// TIA Portal project "MSIL_TESTER_REV3_12JAN23" (V15)

(* hardware
DEVICE "S7-1200 station_1"  S7-1200 Station
   slot 0: "Rack_0"  S7-1200 Rack  Rack  V1.0
   slot 1: "PLC_1"  CPU 1214C DC/DC/DC  6ES7 214-1AG40-0XB0  V4.2
   slot 2: "DI 16/DQ 16x24VDC_1"  6ES7 223-1BL32-0XB0  V2.0
   slot 3: "DQ 8x24VDC _1"  SM 1222 DQ8 x 24VDC  6ES7 222-1BF32-0XB0  V2.0
DEVICE "GSD device_1"  GSD.Device.PN
   slot 0: "Rack"  Rack  V1.0
   slot 0: "cv-x400"  CV-X4XX  CV-X4XX  5.1
      slot 0: "CV-X4XX"  CV-X4XX  5.1
      slot 1: "Interface"  Interface
         slot 1: "Port 1"  Port 1
   slot 1: "Command and Result Status_1"  Command and Result Status
      slot 0: "Command and Result Status"  Command and Result Status
   slot 2: "Trg Ready Status_1"  Trg Ready Status
      slot 0: "Trg Ready Status"  Trg Ready Status
   slot 3: "Trg Ack Status_1"  Trg Ack Status
      slot 0: "Trg Ack Status"  Trg Ack Status
   slot 4: "Miscellaneous Status_1"  Miscellaneous Status
      slot 0: "Miscellaneous Status"  Miscellaneous Status
   slot 5: "Tool Judge Value_1"  Tool Judge Value
      slot 0: "Tool Judge Value"  Tool Judge Value
   slot 6: "Result Data 128Byte_1"  Result Data 128Byte
      slot 0: "Result Data 128Byte"  Result Data 128Byte
   slot 7: "Result Data 32Byte_1"  Result Data 32Byte
      slot 0: "Result Data 32Byte"  Result Data 32Byte
   slot 8: "Result Data 32Byte_2"  Result Data 32Byte
      slot 0: "Result Data 32Byte"  Result Data 32Byte
   slot 9: "Result Data 32Byte_3"  Result Data 32Byte
      slot 0: "Result Data 32Byte"  Result Data 32Byte
   slot 10: "Result Data 32Byte_4"  Result Data 32Byte
      slot 0: "Result Data 32Byte"  Result Data 32Byte
   slot 11: "Result Data 32Byte_5"  Result Data 32Byte
      slot 0: "Result Data 32Byte"  Result Data 32Byte
   slot 12: "Command and Result Control_1"  Command and Result Control
      slot 0: "Command and Result Control"  Command and Result Control
   slot 13: "Trg Control_1"  Trg Control
      slot 0: "Trg Control"  Trg Control
   slot 14: "Miscellaneous Control_1"  Miscellaneous Control
      slot 0: "Miscellaneous Control"  Miscellaneous Control
   slot 15: "Reserved Control_1"  Reserved Control
      slot 0: "Reserved Control"  Reserved Control
   slot 16: "Reserved Control_2"  Reserved Control
      slot 0: "Reserved Control"  Reserved Control
   slot 17: "Parameter 128Byte_1"  Parameter 128Byte
      slot 0: "Parameter 128Byte"  Parameter 128Byte
   slot 18: "Parameter 32Byte_1"  Parameter 32Byte
      slot 0: "Parameter 32Byte"  Parameter 32Byte
   slot 19: "Parameter 32Byte_2"  Parameter 32Byte
      slot 0: "Parameter 32Byte"  Parameter 32Byte
   slot 20: "Parameter 32Byte_3"  Parameter 32Byte
      slot 0: "Parameter 32Byte"  Parameter 32Byte
   slot 21: "Parameter 32Byte_4"  Parameter 32Byte
      slot 0: "Parameter 32Byte"  Parameter 32Byte
   slot 22: "Parameter 32Byte_5"  Parameter 32Byte
      slot 0: "Parameter 32Byte"  Parameter 32Byte
*)

// ===== PLC "PLC_1"  CPU 1214C DC/DC/DC =====

VAR_GLOBAL   // PLC tag table "Default tag table"
   "EMG" AT %I0.0 : Bool;
   "RESET" AT %I0.1 : Bool;
   "Tag_9" AT %I0.2 : Bool;
   "Tag_10" AT %I0.3 : Bool;
   "Tag_11" AT %I0.4 : Bool;
   "Tag_12" AT %I0.5 : Bool;
   "Tag_13" AT %I0.6 : Bool;
   "Tag_14" AT %I0.7 : Bool;
   "Tag_15" AT %I1.0 : Bool;
   "Tag_16" AT %I1.1 : Bool;
   "Tag_17" AT %I1.2 : Bool;
   "Tag_18" AT %I1.3 : Bool;
   "Tag_19" AT %I1.4 : Bool;
   "Tag_20" AT %I1.5 : Bool;
   "Tag_21" AT %I1.6 : Bool;
   "Tag_22" AT %I2.0 : Bool;
   "Tag_23" AT %I2.1 : Bool;
   "Tag_24" AT %I2.2 : Bool;
   "Tag_25" AT %I2.3 : Bool;
   "Tag_26" AT %I2.4 : Bool;
   "Tag_27" AT %I2.5 : Bool;
   "Tag_28" AT %I2.6 : Bool;
   "Tag_29" AT %I2.7 : Bool;
   "Tag_30" AT %I3.0 : Bool;
   "Tag_32" AT %I3.2 : Bool;
   "Tag_46" AT %I3.3 : Bool;
   "Tag_47" AT %I3.4 : Bool;
   "TEST_PART" AT %I1.7 : Bool;
   "Tag_53" AT %I3.5 : Bool;
   "Tag_60" AT %IB12 : Byte;
   "Tag_62" AT %I10.0 : Bool;
   "Tag_59" AT %I10.2 : Bool;
   "Tag_66" AT %IB76 : Byte;
   "Tag_69" AT %IW76 : Int;
   "Tag_75" AT %I10.5 : Bool;
   "rdy" AT %I5.5 : Bool;
   "Tag_76" AT %I3.1 : Bool;
   "Tag_77" AT %I3.6 : Bool;
   "Tag_78" AT %I3.7 : Bool;
   "Tag_3" AT %I13.0 : Bool;
   "Cmd Complete" AT %I20.0 : Bool;
   "Cmd Err" AT %I20.1 : Bool;
   "Cmd Ready" AT %I20.2 : Bool;
   "Result Ready" AT %I20.3 : Bool;
   "Result OR" AT %I20.4 : Bool;
   "res1" AT %I20.5 : Bool;
   "res2" AT %I20.6 : Bool;
   "res3" AT %I20.7 : Bool;
   "READY1" AT %I6.0 : Bool;
   "READY2" AT %I6.1 : Bool;
   "READY3" AT %I6.2 : Bool;
   "READY4" AT %I6.3 : Bool;
   "res4" AT %I6.4 : Bool;
   "res5" AT %I6.5 : Bool;
   "res6" AT %I6.6 : Bool;
   "res7" AT %I6.7 : Bool;
   "BUSY" AT %I7.0 : Bool;
   "ERROR" AT %I7.1 : Bool;
   "res8" AT %I7.2 : Bool;
   "RUN" AT %I7.3 : Bool;
   "res9" AT %I7.4 : Bool;
   "res10" AT %I7.5 : Bool;
   "OUTPUT_IMG_BUSY" AT %I7.6 : Bool;
   "OUTPUT_IMG_STATUS" AT %I7.7 : Bool;
   "res" AT %I8.0 : Bool;
   "res11" AT %I8.1 : Bool;
   "res12" AT %I8.2 : Bool;
   "res13" AT %I8.3 : Bool;
   "res14" AT %I8.4 : Bool;
   "res15" AT %I8.5 : Bool;
   "res16" AT %I8.6 : Bool;
   "res17" AT %I8.7 : Bool;
   "LOGO_RSLT_OK" AT %I68.0 : Bool;
   "LOGO_RSLT_NG" AT %I68.1 : Bool;
   "LED_RSLT_OK" AT %I68.2 : Bool;
   "LED_RSLT_NG" AT %I68.3 : Bool;
   "Tool Judge Value4" AT %I452.4 : Bool;
   "Tag_83" AT %I15.0 : Bool;
   "Tag_1" AT %Q2.5 : Bool;
   "Tag_2" AT %Q3.0 : Bool;
   "Tag_4" AT %Q2.0 : Bool;
   "Tag_5" AT %Q0.1 : Bool;
   "Tag_7" AT %Q0.2 : Bool;
   "Tag_8" AT %Q0.3 : Bool;
   "Tag_33" AT %Q0.5 : Bool;
   "Tag_34" AT %Q0.6 : Bool;
   "Tag_35" AT %Q0.7 : Bool;
   "Tag_36" AT %Q1.0 : Bool;
   "Tag_37" AT %Q1.1 : Bool;
   "Tag_38" AT %Q2.1 : Bool;
   "Tag_39" AT %Q2.2 : Bool;
   "Tag_40" AT %Q2.3 : Bool;
   "Tag_41" AT %Q3.1 : Bool;
   "Tag_42" AT %Q3.2 : Bool;
   "Tag_43" AT %Q3.3 : Bool;
   "Tag_44" AT %Q2.6 : Bool;
   "Tag_45" AT %Q2.7 : Bool;
   "Tag_48" AT %Q3.4 : Bool;
   "Tag_49" AT %Q3.5 : Bool;
   "Tag_50" AT %Q3.6 : Bool;
   "Tag_51" AT %Q3.7 : Bool;
   "Tag_52" AT %Q2.4 : Bool;
   "Tag_58" AT %QB12 : Byte;
   "Tag_56" AT %QB6 : Byte;
   "Tag_64" AT %QB8 : Byte;
   "Tag_65" AT %Q500.5 : Bool;
   "Tag_67" AT %QW504 : Int;
   "Tag_68" AT %QW76 : Int;
   "Tag_71" AT %Q500.0 : Bool;
   "Tag_72" AT %Q500.2 : Bool;
   "Tag_61" AT %Q4.0 : Bool;
   "Tag_63" AT %Q4.1 : Bool;
   "Tag_73" AT %Q4.2 : Bool;
   "Tag_74" AT %Q4.3 : Bool;
   "Tag_79" AT %Q4.4 : Bool;
   "Tag_80" AT %Q4.5 : Bool;
   "Tag_81" AT %Q0.0 : Bool;
   "Tag_6" AT %Q0.4 : Bool;
   "Tag_82" AT %Q6.0 : Bool;
   "Tag_86" AT %Q601.0 : Bool;
   "Tag_87" AT %Q50.0 : Bool;
   "Tag_88" AT %Q51.0 : Bool;
   "Tag_89" AT %Q52.0 : Bool;
   "Tag_90" AT %Q31.0 : Bool;
   "Tag_91" AT %Q5.0 : Bool;
   "Tag_31" AT %Q6.1 : Bool;
   "cam_reset" AT %Q7.0 : Bool;
   "Cam_Ext" AT %Q7.1 : Bool;
   "Tag_54" AT %QW2 : Int;
   "Tag_55" AT %QW21 : Int;
   "Tag_57" AT %QW24 : Word;
   "Tag_70" AT %QW29 : Word;
   "command" AT %QW78 : Int;
   "SD_CardNo" AT %QD80 : DInt;
   "Program_Number" AT %QD84 : DInt;
   "TAG 1" AT %M1.0 : Bool;
   "SHORT_CT" AT %M1.1 : Bool;
   "OK" AT %M1.2 : Bool;
   "NG" AT %M1.3 : Bool;
   "CONTINUITY" AT %M1.4 : Bool;
   "DIELECTRIC" AT %M1.5 : Bool;
   "TAG 2" AT %M1.6 : Bool;
   "SEQ_1" AT %MB2 : Byte;
   "RED_LED" AT %M1.7 : Bool;
   "AMBER_LED" AT %M3.0 : Bool;
   "GREEN_LED" AT %M3.1 : Bool;
   "TAG 3" AT %M3.2 : Bool;
   "TAG 4" AT %M3.3 : Bool;
   "TEST" AT %M3.4 : Bool;
   "MAIN SEQ" AT %MW4 : Int;
   "BLUE LED" AT %M3.5 : Bool;
   "GROUND" AT %M3.6 : Bool;
   "RED LED" AT %M3.7 : Bool;
   "GREEN LED" AT %M6.0 : Bool;
   "SEQ_MAIN" AT %MW8 : Int;
   "RED" AT %M6.1 : Bool;
   "BLUE" AT %M6.2 : Bool;
   "GREEN" AT %M6.3 : Bool;
   "COMMON" AT %M6.4 : Bool;
   "TEST 3" AT %M6.5 : Bool;
   "TEST 4" AT %M6.6 : Bool;
   "TEST 5" AT %M6.7 : Bool;
   "TRG" AT %M7.0 : Bool;
   "INC" AT %MD10 : DInt;
   "P_TRG" AT %M7.1 : Bool;
   "INC`1" AT %MD14 : DInt;
   "TEST_START" AT %M7.2 : Bool;
   "TEST_6" AT %M7.3 : Bool;
   "CON_TRG" AT %M7.4 : Bool;
   "DIE_TRG" AT %M7.5 : Bool;
   "SHORT_TRG" AT %M7.6 : Bool;
   "BIT 1" AT %M7.7 : Bool;
   "BIT 2" AT %M18.0 : Bool;
   "TRG1" AT %M18.1 : Bool;
   "TRG 2" AT %M18.2 : Bool;
   "TRG 3" AT %M18.3 : Bool;
   "TRG 4" AT %M18.4 : Bool;
   "TRG5" AT %M18.5 : Bool;
   "TRG 6" AT %M18.6 : Bool;
   "TEST_SEQ" AT %MW20 : Int;
   "TEST 7" AT %M18.7 : Bool;
   "VISION_OK" AT %M19.0 : Bool;
   "VISION_NG" AT %M19.1 : Bool;
   "TRG 7" AT %M19.2 : Bool;
   "TRG 8" AT %M19.3 : Bool;
   "FGH" AT %MD22 : DInt;
   "TEST_RESET" AT %M19.4 : Bool;
   "test 10" AT %M19.5 : Bool;
   "TRG 9" AT %M19.6 : Bool;
   "test_print" AT %M19.7 : Bool;
   "FWD_TEST" AT %M26.0 : Bool;
   "X2" AT %M26.1 : Bool;
   "X3" AT %M26.2 : Bool;
   "CL" AT %M26.3 : Bool;
   "TEST_BUZ" AT %M26.4 : Bool;
   "System_Byte" AT %MB200 : Byte;
   "FirstScan" AT %M200.0 : Bool;
   "DiagStatusUpdate" AT %M200.1 : Bool;
   "AlwaysTRUE" AT %M200.2 : Bool;
   "AlwaysFALSE" AT %M200.3 : Bool;
   "Clock_Byte" AT %MB202 : Byte;
   "Clock_10Hz" AT %M202.0 : Bool;
   "Clock_5Hz" AT %M202.1 : Bool;
   "Clock_2.5Hz" AT %M202.2 : Bool;
   "Clock_2Hz" AT %M202.3 : Bool;
   "Clock_1.25Hz" AT %M202.4 : Bool;
   "Clock_1Hz" AT %M202.5 : Bool;
   "Clock_0.625Hz" AT %M202.6 : Bool;
   "Clock_0.5Hz" AT %M202.7 : Bool;
   "System_Byte(3)" AT %MB200 : Byte;
   "OK_TEST" AT %M26.5 : Bool;
   "NG_TEST" AT %M26.6 : Bool;
   "SCN_OK" AT %M26.7 : Bool;
   "TRG10" AT %M27.0 : Bool;
   "GROUND_TEST" AT %M27.1 : Bool;
   "TEST_GREEN" AT %M27.2 : Bool;
   "TEST_BLUE" AT %M27.3 : Bool;
   "TEST_RED" AT %M27.4 : Bool;
   "Manual" AT %M27.5 : Bool;
   "TRG11" AT %M27.6 : Bool;
   "TRG12" AT %M27.7 : Bool;
   "PROGRAM_TRG" AT %M28.0 : Bool;
   "BREAK" AT %M28.1 : Bool;
   "CAM_TRG" AT %M28.2 : Bool;
   "TRG 11" AT %M28.3 : Bool;
   "TRG 12" AT %M28.4 : Bool;
   "BUFF_CLR" AT %M28.5 : Bool;
   "TRG13" AT %M28.6 : Bool;
   "TRG14" AT %M28.7 : Bool;
   "TRG 15" AT %M29.0 : Bool;
   "TRG 16" AT %M29.1 : Bool;
   "TEST_CLEAR" AT %M29.2 : Bool;
   "TRG15" AT %M29.3 : Bool;
   "TRG_16" AT %M29.4 : Bool;
   "TRG17" AT %M29.5 : Bool;
   "BREAK 2" AT %M29.6 : Bool;
   "BREAK 3" AT %M29.7 : Bool;
   "break 4" AT %M30.0 : Bool;
   "break 5" AT %M30.1 : Bool;
   "break 6" AT %M30.2 : Bool;
   "break 9" AT %M30.3 : Bool;
   "break 10" AT %M30.4 : Bool;
   "TRG20" AT %M30.5 : Bool;
   "TRG 17" AT %M30.6 : Bool;
   "TRG 20" AT %M30.7 : Bool;
   "break 11" AT %M31.0 : Bool;
   "REJECTION_ERROR_SET" AT %M31.1 : Bool;
   "BREAK 15" AT %M31.2 : Bool;
   "assembly bar code" AT %M31.3 : Bool;
   "POT_TEST" AT %M31.4 : Bool;
   "POT_TEST_GREEN" AT %M0.0 : Bool;
   "POT_TEST_BLUE" AT %M0.1 : Bool;
   "SCAN_BYP" AT %M0.2 : Bool;
   "test16" AT %M0.3 : Bool;
   "BUFF_CLR_10" AT %M0.4 : Bool;
   "trg18" AT %M0.5 : Bool;
   "trg19" AT %M0.6 : Bool;
   "buff_clr_11" AT %M0.7 : Bool;
   "CAM_2ND_TRG" AT %M31.5 : Bool;
   "TRG25" AT %M31.6 : Bool;
   "START" AT %M31.7 : Bool;
   "EL_GOOD" AT %MD32 : DInt;
   "EL_BAD" AT %MD36 : DInt;
   "VISION_CAL_OFF" AT %M40.0 : Bool;
   "LOGO_CAL_OFF" AT %M40.1 : Bool;
   "LED_CALI_OFF" AT %M40.2 : Bool;
   "ELEC_CAL_OFF" AT %M40.3 : Bool;
   "TEST 17" AT %M40.4 : Bool;
   "TEST 18" AT %M40.5 : Bool;
   "TEST 19" AT %M40.6 : Bool;
   "TEST 20" AT %M40.7 : Bool;
   "TEST 21" AT %M41.0 : Bool;
   "TEST 22" AT %M41.1 : Bool;
   "TEST 23" AT %M41.2 : Bool;
   "TEST 24" AT %M41.3 : Bool;
   "Tag_84" AT %M50.0 : Bool;
   "Tag_85" AT %M51.0 : Bool;
   "BREAK_1" AT %M41.4 : Bool;
   "ext" AT %M41.5 : Bool;
   "Cmd_rqt" AT %M41.6 : Bool;
   "TEST 25" AT %M41.7 : Bool;
   "Program_no" AT %MW42 : Word;
   "TEST6" AT %M44.0 : Bool;
   "TEMP" AT %M44.1 : Bool;
   "READ_TRIG" AT %M44.2 : Bool;
   "VISION TEST RUN_TIG" AT %M44.3 : Bool;
   "ELE_OK" AT %M44.4 : Bool;
END_VAR

DATA_BLOCK "MAIN_SEQ_DB"   // DB1
{ S7_Optimized_Access := 'TRUE' }
VERSION : 0.1
// stored: InstanceOfName MAIN_SEQ
"MAIN_SEQ"
BEGIN
END_DATA_BLOCK

DATA_BLOCK "UI"   // DB4
{ S7_Optimized_Access := 'FALSE' }
VERSION : 0.1
   VAR
      status : Int;
      ELECTRICAL_TEST_RSLT : Int;
      L0GO_RSLT : Int;
      AMBER_LED_RSLT : Int;
      STATUS_VISION : Int;
      RED_LED_RSLT : Int;
      BLUE_LED_RSLT : Int;
      GREEN_LED_RSLT : Int;
      TEST : Int;
      SCAN_RESULT : Int;
      "Print / fail" : Int;
      VALUE_RESET_BIT : Int;
      "Part Id" : String;
      "STOP&CON" : Bool;
      OUT : Bool;
      "STOP/CON" : Bool;
      CONVEYER_FB : Bool;
      REJ_FB : Bool;
      CALIBRATION : Bool;
      "ASSEMBLY SCANNER" : Bool;
      calib : Int;
      print : Bool;
      TRACEBILITY_BYPASS : Bool;
   END_VAR
BEGIN
END_DATA_BLOCK

DATA_BLOCK "TESTING_SEQ"   // DB5
{ S7_Optimized_Access := 'TRUE' }
VERSION : 0.1
// stored: InstanceOfName TESTING_SEQUENCE
"TESTING_SEQUENCE"
BEGIN
END_DATA_BLOCK

DATA_BLOCK "HMI INTERFACE"   // DB24
{ S7_Optimized_Access := 'FALSE' }
VERSION : 0.1
   VAR
      START : Bool;
      MANUAL : Bool;
      ELEC_PART_LOAD : Bool;
      VISION_PART_LOAD : Bool;
      SC_OK : Bool;
      SC_NG : Bool;
      CON_OK : Bool;
      CON_NG : Bool;
      DIE_OK : Bool;
      RESET : Bool;
      LCK1 : Bool;
      LCK2 : Bool;
      LCK3 : Bool;
      LH_BOTTOM_CYL_UP : Bool;
      LH_BOTTOM_CYL_DWN : Bool;
      RH_BOTTOM_CYL_UP : Bool;
      RH_BOTTOM_CYL_DWN : Bool;
      "PUNCH 1" : Bool;
      "PUNCH 2" : Bool;
      CONVEYER_REV : Bool;
      CON_FWD : Bool;
      MC_LIGHT : Bool;
      ERROR : Int;
      ERROR_POPUP : Bool;
      MC_STATUS : Int;
      COUNT_RST : Bool;
      REJECTION_POPUP : Bool;
      "TEST PASS POPUP" : Bool;
      CALIBRATION : Bool;
      PRESSURE_DROP_POPUP : Bool;
      "MC LIGHT 2" : Bool;
      BLUE_LIGHT_ON : Bool;
      "ELECTRICAL CALIBRATION" : Bool;
      "VIASION CALIBRATION" : Bool;
      "LOGO CALIBRATION" : Bool;
      "LED CALIBRATION" : Bool;
      LED_ON : Int;
      LOGO_LOCK : Bool;
      RECEIVER_MOVE : Bool;
      TRACEBILITY_BYPASS : Bool;
   END_VAR
BEGIN
END_DATA_BLOCK

DATA_BLOCK "INPUTS"   // DB28
{ S7_Optimized_Access := 'TRUE' }
VERSION : 0.1
   VAR
      KEY_SWITCH : Bool;
      RESET_PB : Bool;
      EMG_PB : Bool;
      LOCK1_REV : Bool;
      LOCK1_FWD : Bool;
      LOCK2_REV : Bool;
      LOCK2_FWD : Bool;
      LOCK3_REV : Bool;
      LOCK3_FWD : Bool;
      LH_BOTTOM_CYL_DOWN : Bool;
      LH_BOTTOM_CYL_UP : Bool;
      RH_BOTTOM_CYL_DOWN : Bool;
      RH_BOTTOM_CYL_UP : Bool;
      PUNCH_CYL1_REV : Bool;
      PUNCH_CYL1_FWD : Bool;
      PUNCH_CYL2_REV : Bool;
      PUNCH_CYL2_FWD : Bool;
      OPTICAL_SENSOR1 : Bool;
      OPTICAL_SENSOR2 : Bool;
      OPTICAL_SENSOR3 : Bool;
      ADAPTRONICS_OK_FB : Bool;
      ADAPTRONICS_NG_FB : Bool;
      ADAPTRONICS_SEGMENT : Bool;
      REJECTION_THROUGH_BEAM : Bool;
      GOOD_THROUGH_BEAM : Bool;
      PRESSURE_SENSOR : Bool;
      "CHARGING CYL_FWD" : Bool;
      "CHARGING CYL_REV" : Bool;
      "LOGO LCK_REV" : Bool;
      "LOGO LCK_FWD" : Bool;
      "LOGO OPTIC_SENSR" : Bool;
   END_VAR
BEGIN
END_DATA_BLOCK

DATA_BLOCK "OUTPUTS"   // DB29
{ S7_Optimized_Access := 'TRUE' }
VERSION : 0.1
   VAR
      TOWER_BUZZER : Bool;
      GREEN_ILLU : Bool;
      MACHINE_LIGHT : Bool;
      LOCK1 : Bool;
      LOCK2 : Bool;
      LOCK3 : Bool;
      PUNCH1 : Bool;
      PUNCH2 : Bool;
      LH_BOTTOM_CYL : Bool;
      RH_BOTTOM_CYL : Bool;
      ADAPTRONICS_START : Bool;
      ADAPTRONICS_ABORT : Bool;
      ADAPTRONICS_CONTINUE : Bool;
      RED : Bool;
      BLUE : Bool;
      GREEN : Bool;
      GROUND : Bool;
      TOWER_RED : Bool;
      TOWER_AMBER : Bool;
      TOWER_GREEN : Bool;
      CON_FWD : Bool;
      CON_REV : Bool;
      "LOGO CYL_ON" : Bool;
      "CHARGING CYL_ON" : Bool;
      "RELAY 5" : Bool;
      "RELAY 6" : Bool;
      "RELAY 7" : Bool;
      "RELAY 8" : Bool;
      "RELAY 9" : Bool;
      AMBER : Bool;
      "RED LIGHT" : Bool;
      "GREEN LIGHT" : Bool;
      RED_LED_ON : Bool;
      AMBER_LED_ON : Bool;
      BLUE_LED_ON : Bool;
      GREEN_LED_ON : Bool;
   END_VAR
BEGIN
END_DATA_BLOCK

DATA_BLOCK "BITS"   // DB30
{ S7_Optimized_Access := 'TRUE' }
VERSION : 0.1
   VAR
      ELECRICAL_PART_LOADED : Bool;
      VISION_PART_LOADED : Bool;
      ELECTRICAL_TEST_START : Bool;
      ELECTRICAL_TEST_COMPLETED : Bool;
      VISION_TEST_COMPLETED : Bool;
      VISION_TEST_START : Bool;
      ELEC_GOOD_FB : Bool;
      ELEC_BAD_FB : Bool;
      AMBER_LED_ON : Bool;
      RED_LED_ON : Bool;
      BLUE_LED_ON : Bool;
      GREEN_LED_ON : Bool;
   END_VAR
BEGIN
END_DATA_BLOCK

DATA_BLOCK "CAMERA_DB"   // DB33
{ S7_Optimized_Access := 'TRUE' }
VERSION : 0.1
   VAR
      RED_LED : Bool;
      GREEN_LED : Bool;
      BLUE_LED : Bool;
      CAMERA_1_TRG : Bool;
      LOGO_RSLT_OK : Bool;
      LOGO_RSLT_NG : Bool;
      LED_RSLT_OK : Bool;
      LED_RSLT_NG : Bool;
      PROGRAM_NO : Int;
      PROG_EN : Bool;
      LOGO_TEST_START : Bool;
      LOGO_TEST_CMPLT : Bool;
      CAMERA_2_TRG : Bool;
   END_VAR
BEGIN
END_DATA_BLOCK

DATA_BLOCK "cAM_MAN_DATA"   // DB40
{ S7_Optimized_Access := 'FALSE' }
VERSION : 0.1
   VAR
      Part : Int;
      Program_number : Int;
      Program_Change : Bool;
      Cam_trig : Bool;
      Program_trig : Bool;
      buffer_clear : Bool;
      Red : Bool;
      Blue : Bool;
      Green : Bool;
      cam_good : Bool;
      cam_bad : Bool;
   END_VAR
BEGIN
END_DATA_BLOCK

DATA_BLOCK "RETENTIVE_VALUES"   // DB63
{ S7_Optimized_Access := 'FALSE' }
VERSION : 0.1
   VAR
      GOOD_COUNT : Int;
      BAD_COUNT : Int;
   END_VAR
BEGIN
END_DATA_BLOCK

DATA_BLOCK "CVX 300 DB"   // DB78
{ S7_Optimized_Access := 'FALSE' }
VERSION : 0.1
   VAR
      "CAM READY" : Bool;
      "CAM GOOD" : Bool;
      "CAM BAD" : Bool;
      "CAM TRG" : Bool;
      RESET : Bool;
   END_VAR
BEGIN
END_DATA_BLOCK

DATA_BLOCK "HMI_CAMERA"   // DB79
{ S7_Optimized_Access := 'FALSE' }
VERSION : 0.1
   VAR
      LOGO_CAM_TRG : Bool;
      LED_CAM_TRG : Bool;
      LOGO_CAM_OK : Bool;
      LOGO_CAM_NG : Bool;
      LED_CAM_OK : Bool;
      LED_CAM_NG : Bool;
      RESET : Bool;
   END_VAR
BEGIN
END_DATA_BLOCK

// folder: System blocks/Program resources

DATA_BLOCK "IEC_Timer_0_DB"   // DB2
{ S7_Optimized_Access := 'TRUE' }
AUTHOR : Simatic
FAMILY : IEC
NAME : IEC_TMR
VERSION : 1.0
// stored: InstanceOfName IEC_TIMER
"IEC_TIMER"
BEGIN
END_DATA_BLOCK

DATA_BLOCK "IEC_Timer_0_DB_5"   // DB3
{ S7_Optimized_Access := 'TRUE' }
AUTHOR : Simatic
FAMILY : IEC
NAME : IEC_TMR
VERSION : 1.0
// stored: InstanceOfName IEC_TIMER
"IEC_TIMER"
BEGIN
END_DATA_BLOCK

DATA_BLOCK "IEC_Timer_0_DB_6"   // DB6
{ S7_Optimized_Access := 'TRUE' }
AUTHOR : Simatic
FAMILY : IEC
NAME : IEC_TMR
VERSION : 1.0
// stored: InstanceOfName IEC_TIMER
"IEC_TIMER"
BEGIN
END_DATA_BLOCK

DATA_BLOCK "IEC_Timer_0_DB_1"   // DB7
{ S7_Optimized_Access := 'TRUE' }
AUTHOR : Simatic
FAMILY : IEC
NAME : IEC_TMR
VERSION : 1.0
// stored: InstanceOfName IEC_TIMER
"IEC_TIMER"
BEGIN
END_DATA_BLOCK

DATA_BLOCK "IEC_Timer_0_DB_2"   // DB8
{ S7_Optimized_Access := 'TRUE' }
AUTHOR : Simatic
FAMILY : IEC
NAME : IEC_TMR
VERSION : 1.0
// stored: InstanceOfName IEC_TIMER
"IEC_TIMER"
BEGIN
END_DATA_BLOCK

DATA_BLOCK "IEC_Timer_0_DB_3"   // DB9
{ S7_Optimized_Access := 'TRUE' }
AUTHOR : Simatic
FAMILY : IEC
NAME : IEC_TMR
VERSION : 1.0
// stored: InstanceOfName IEC_TIMER
"IEC_TIMER"
BEGIN
END_DATA_BLOCK

DATA_BLOCK "IEC_Timer_0_DB_4"   // DB10
{ S7_Optimized_Access := 'TRUE' }
AUTHOR : Simatic
FAMILY : IEC
NAME : IEC_TMR
VERSION : 1.0
// stored: InstanceOfName IEC_TIMER
"IEC_TIMER"
BEGIN
END_DATA_BLOCK

DATA_BLOCK "IEC_Timer_0_DB_18"   // DB11
{ S7_Optimized_Access := 'TRUE' }
AUTHOR : Simatic
FAMILY : IEC
NAME : IEC_TMR
VERSION : 1.0
// stored: InstanceOfName IEC_TIMER
"IEC_TIMER"
BEGIN
END_DATA_BLOCK

DATA_BLOCK "IEC_Timer_0_DB_19"   // DB12
{ S7_Optimized_Access := 'TRUE' }
AUTHOR : Simatic
FAMILY : IEC
NAME : IEC_TMR
VERSION : 1.0
// stored: InstanceOfName IEC_TIMER
"IEC_TIMER"
BEGIN
END_DATA_BLOCK

DATA_BLOCK "IEC_Timer_0_DB_52"   // DB13
{ S7_Optimized_Access := 'TRUE' }
AUTHOR : Simatic
FAMILY : IEC
NAME : IEC_TMR
VERSION : 1.0
// stored: InstanceOfName IEC_TIMER
"IEC_TIMER"
BEGIN
END_DATA_BLOCK

DATA_BLOCK "IEC_Timer_0_DB_7"   // DB14
{ S7_Optimized_Access := 'TRUE' }
AUTHOR : Simatic
FAMILY : IEC
NAME : IEC_TMR
VERSION : 1.0
// stored: InstanceOfName IEC_TIMER
"IEC_TIMER"
BEGIN
END_DATA_BLOCK

DATA_BLOCK "IEC_Timer_0_DB_9"   // DB15
{ S7_Optimized_Access := 'TRUE' }
AUTHOR : Simatic
FAMILY : IEC
NAME : IEC_TMR
VERSION : 1.0
// stored: InstanceOfName IEC_TIMER
"IEC_TIMER"
BEGIN
END_DATA_BLOCK

DATA_BLOCK "IEC_Timer_0_DB_10"   // DB16
{ S7_Optimized_Access := 'TRUE' }
AUTHOR : Simatic
FAMILY : IEC
NAME : IEC_TMR
VERSION : 1.0
// stored: InstanceOfName IEC_TIMER
"IEC_TIMER"
BEGIN
END_DATA_BLOCK

DATA_BLOCK "IEC_Timer_0_DB_11"   // DB17
{ S7_Optimized_Access := 'TRUE' }
AUTHOR : Simatic
FAMILY : IEC
NAME : IEC_TMR
VERSION : 1.0
// stored: InstanceOfName IEC_TIMER
"IEC_TIMER"
BEGIN
END_DATA_BLOCK

DATA_BLOCK "IEC_Timer_0_DB_12"   // DB18
{ S7_Optimized_Access := 'TRUE' }
AUTHOR : Simatic
FAMILY : IEC
NAME : IEC_TMR
VERSION : 1.0
// stored: InstanceOfName IEC_TIMER
"IEC_TIMER"
BEGIN
END_DATA_BLOCK

DATA_BLOCK "IEC_Timer_0_DB_13"   // DB19
{ S7_Optimized_Access := 'TRUE' }
AUTHOR : Simatic
FAMILY : IEC
NAME : IEC_TMR
VERSION : 1.0
// stored: InstanceOfName IEC_TIMER
"IEC_TIMER"
BEGIN
END_DATA_BLOCK

DATA_BLOCK "IEC_Timer_0_DB_14"   // DB20
{ S7_Optimized_Access := 'TRUE' }
AUTHOR : Simatic
FAMILY : IEC
NAME : IEC_TMR
VERSION : 1.0
// stored: InstanceOfName IEC_TIMER
"IEC_TIMER"
BEGIN
END_DATA_BLOCK

DATA_BLOCK "IEC_Timer_0_DB_15"   // DB21
{ S7_Optimized_Access := 'TRUE' }
AUTHOR : Simatic
FAMILY : IEC
NAME : IEC_TMR
VERSION : 1.0
// stored: InstanceOfName IEC_TIMER
"IEC_TIMER"
BEGIN
END_DATA_BLOCK

DATA_BLOCK "IEC_Timer_0_DB_16"   // DB22
{ S7_Optimized_Access := 'TRUE' }
AUTHOR : Simatic
FAMILY : IEC
NAME : IEC_TMR
VERSION : 1.0
// stored: InstanceOfName IEC_TIMER
"IEC_TIMER"
BEGIN
END_DATA_BLOCK

DATA_BLOCK "IEC_Timer_0_DB_17"   // DB23
{ S7_Optimized_Access := 'TRUE' }
AUTHOR : Simatic
FAMILY : IEC
NAME : IEC_TMR
VERSION : 1.0
// stored: InstanceOfName IEC_TIMER
"IEC_TIMER"
BEGIN
END_DATA_BLOCK

DATA_BLOCK "IEC_Timer_0_DB_20"   // DB25
{ S7_Optimized_Access := 'TRUE' }
AUTHOR : Simatic
FAMILY : IEC
NAME : IEC_TMR
VERSION : 1.0
// stored: InstanceOfName IEC_TIMER
"IEC_TIMER"
BEGIN
END_DATA_BLOCK

DATA_BLOCK "IEC_Timer_0_DB_21"   // DB26
{ S7_Optimized_Access := 'TRUE' }
AUTHOR : Simatic
FAMILY : IEC
NAME : IEC_TMR
VERSION : 1.0
// stored: InstanceOfName IEC_TIMER
"IEC_TIMER"
BEGIN
END_DATA_BLOCK

DATA_BLOCK "IEC_Timer_0_DB_22"   // DB27
{ S7_Optimized_Access := 'TRUE' }
AUTHOR : Simatic
FAMILY : IEC
NAME : IEC_TMR
VERSION : 1.0
// stored: InstanceOfName IEC_TIMER
"IEC_TIMER"
BEGIN
END_DATA_BLOCK

DATA_BLOCK "IEC_Timer_0_DB_23"   // DB31
{ S7_Optimized_Access := 'TRUE' }
AUTHOR : Simatic
FAMILY : IEC
NAME : IEC_TMR
VERSION : 1.0
// stored: InstanceOfName IEC_TIMER
"IEC_TIMER"
BEGIN
END_DATA_BLOCK

DATA_BLOCK "IEC_Timer_0_DB_24"   // DB32
{ S7_Optimized_Access := 'TRUE' }
AUTHOR : Simatic
FAMILY : IEC
NAME : IEC_TMR
VERSION : 1.0
// stored: InstanceOfName IEC_TIMER
"IEC_TIMER"
BEGIN
END_DATA_BLOCK

DATA_BLOCK "IEC_Timer_0_DB_8"   // DB34
{ S7_Optimized_Access := 'TRUE' }
AUTHOR : Simatic
FAMILY : IEC
NAME : IEC_TMR
VERSION : 1.0
// stored: InstanceOfName IEC_TIMER
"IEC_TIMER"
BEGIN
END_DATA_BLOCK

DATA_BLOCK "IEC_Timer_0_DB_25"   // DB35
{ S7_Optimized_Access := 'TRUE' }
AUTHOR : Simatic
FAMILY : IEC
NAME : IEC_TMR
VERSION : 1.0
// stored: InstanceOfName IEC_TIMER
"IEC_TIMER"
BEGIN
END_DATA_BLOCK

DATA_BLOCK "IEC_Timer_0_DB_26"   // DB36
{ S7_Optimized_Access := 'TRUE' }
AUTHOR : Simatic
FAMILY : IEC
NAME : IEC_TMR
VERSION : 1.0
// stored: InstanceOfName IEC_TIMER
"IEC_TIMER"
BEGIN
END_DATA_BLOCK

DATA_BLOCK "IEC_Timer_0_DB_27"   // DB37
{ S7_Optimized_Access := 'TRUE' }
AUTHOR : Simatic
FAMILY : IEC
NAME : IEC_TMR
VERSION : 1.0
// stored: InstanceOfName IEC_TIMER
"IEC_TIMER"
BEGIN
END_DATA_BLOCK

DATA_BLOCK "IEC_Timer_0_DB_28"   // DB38
{ S7_Optimized_Access := 'TRUE' }
AUTHOR : Simatic
FAMILY : IEC
NAME : IEC_TMR
VERSION : 1.0
// stored: InstanceOfName IEC_TIMER
"IEC_TIMER"
BEGIN
END_DATA_BLOCK

DATA_BLOCK "IEC_Timer_0_DB_29"   // DB39
{ S7_Optimized_Access := 'TRUE' }
AUTHOR : Simatic
FAMILY : IEC
NAME : IEC_TMR
VERSION : 1.0
// stored: InstanceOfName IEC_TIMER
"IEC_TIMER"
BEGIN
END_DATA_BLOCK

DATA_BLOCK "IEC_Timer_0_DB_30"   // DB41
{ S7_Optimized_Access := 'TRUE' }
AUTHOR : Simatic
FAMILY : IEC
NAME : IEC_TMR
VERSION : 1.0
// stored: InstanceOfName IEC_TIMER
"IEC_TIMER"
BEGIN
END_DATA_BLOCK

DATA_BLOCK "IEC_Timer_0_DB_31"   // DB42
{ S7_Optimized_Access := 'TRUE' }
AUTHOR : Simatic
FAMILY : IEC
NAME : IEC_TMR
VERSION : 1.0
// stored: InstanceOfName IEC_TIMER
"IEC_TIMER"
BEGIN
END_DATA_BLOCK

DATA_BLOCK "IEC_Timer_0_DB_32"   // DB43
{ S7_Optimized_Access := 'TRUE' }
AUTHOR : Simatic
FAMILY : IEC
NAME : IEC_TMR
VERSION : 1.0
// stored: InstanceOfName IEC_TIMER
"IEC_TIMER"
BEGIN
END_DATA_BLOCK

DATA_BLOCK "IEC_Timer_0_DB_33"   // DB44
{ S7_Optimized_Access := 'TRUE' }
AUTHOR : Simatic
FAMILY : IEC
NAME : IEC_TMR
VERSION : 1.0
// stored: InstanceOfName IEC_TIMER
"IEC_TIMER"
BEGIN
END_DATA_BLOCK

DATA_BLOCK "IEC_Timer_0_DB_34"   // DB45
{ S7_Optimized_Access := 'TRUE' }
AUTHOR : Simatic
FAMILY : IEC
NAME : IEC_TMR
VERSION : 1.0
// stored: InstanceOfName IEC_TIMER
"IEC_TIMER"
BEGIN
END_DATA_BLOCK

DATA_BLOCK "IEC_Timer_0_DB_35"   // DB46
{ S7_Optimized_Access := 'TRUE' }
AUTHOR : Simatic
FAMILY : IEC
NAME : IEC_TMR
VERSION : 1.0
// stored: InstanceOfName IEC_TIMER
"IEC_TIMER"
BEGIN
END_DATA_BLOCK

DATA_BLOCK "IEC_Timer_0_DB_36"   // DB47
{ S7_Optimized_Access := 'TRUE' }
AUTHOR : Simatic
FAMILY : IEC
NAME : IEC_TMR
VERSION : 1.0
// stored: InstanceOfName IEC_TIMER
"IEC_TIMER"
BEGIN
END_DATA_BLOCK

DATA_BLOCK "LED_ON_DELAY"   // DB48
{ S7_Optimized_Access := 'TRUE' }
AUTHOR : Simatic
FAMILY : IEC
NAME : IEC_TMR
VERSION : 1.0
// stored: InstanceOfName IEC_TIMER
"IEC_TIMER"
BEGIN
END_DATA_BLOCK

DATA_BLOCK "TEST_ABORT"   // DB49
{ S7_Optimized_Access := 'TRUE' }
AUTHOR : Simatic
FAMILY : IEC
NAME : IEC_TMR
VERSION : 1.0
// stored: InstanceOfName IEC_TIMER
"IEC_TIMER"
BEGIN
END_DATA_BLOCK

DATA_BLOCK "IEC_Timer_0_DB_37"   // DB50
{ S7_Optimized_Access := 'TRUE' }
AUTHOR : Simatic
FAMILY : IEC
NAME : IEC_TMR
VERSION : 1.0
// stored: InstanceOfName IEC_TIMER
"IEC_TIMER"
BEGIN
END_DATA_BLOCK

DATA_BLOCK "IEC_Timer_0_DB_40"   // DB51
{ S7_Optimized_Access := 'TRUE' }
AUTHOR : Simatic
FAMILY : IEC
NAME : IEC_TMR
VERSION : 1.0
// stored: InstanceOfName IEC_TIMER
"IEC_TIMER"
BEGIN
END_DATA_BLOCK

DATA_BLOCK "IEC_Timer_0_DB_41"   // DB52
{ S7_Optimized_Access := 'TRUE' }
AUTHOR : Simatic
FAMILY : IEC
NAME : IEC_TMR
VERSION : 1.0
// stored: InstanceOfName IEC_TIMER
"IEC_TIMER"
BEGIN
END_DATA_BLOCK

DATA_BLOCK "IEC_Timer_0_DB_42"   // DB53
{ S7_Optimized_Access := 'TRUE' }
AUTHOR : Simatic
FAMILY : IEC
NAME : IEC_TMR
VERSION : 1.0
// stored: InstanceOfName IEC_TIMER
"IEC_TIMER"
BEGIN
END_DATA_BLOCK

DATA_BLOCK "IEC_Timer_0_DB_43"   // DB54
{ S7_Optimized_Access := 'TRUE' }
AUTHOR : Simatic
FAMILY : IEC
NAME : IEC_TMR
VERSION : 1.0
// stored: InstanceOfName IEC_TIMER
"IEC_TIMER"
BEGIN
END_DATA_BLOCK

DATA_BLOCK "IEC_Timer_0_DB_44"   // DB55
{ S7_Optimized_Access := 'TRUE' }
AUTHOR : Simatic
FAMILY : IEC
NAME : IEC_TMR
VERSION : 1.0
// stored: InstanceOfName IEC_TIMER
"IEC_TIMER"
BEGIN
END_DATA_BLOCK

DATA_BLOCK "IEC_Timer_0_DB_45"   // DB56
{ S7_Optimized_Access := 'TRUE' }
AUTHOR : Simatic
FAMILY : IEC
NAME : IEC_TMR
VERSION : 1.0
// stored: InstanceOfName IEC_TIMER
"IEC_TIMER"
BEGIN
END_DATA_BLOCK

DATA_BLOCK "IEC_Timer_0_DB_46"   // DB57
{ S7_Optimized_Access := 'TRUE' }
AUTHOR : Simatic
FAMILY : IEC
NAME : IEC_TMR
VERSION : 1.0
// stored: InstanceOfName IEC_TIMER
"IEC_TIMER"
BEGIN
END_DATA_BLOCK

DATA_BLOCK "IEC_Timer_0_DB_47"   // DB58
{ S7_Optimized_Access := 'TRUE' }
AUTHOR : Simatic
FAMILY : IEC
NAME : IEC_TMR
VERSION : 1.0
// stored: InstanceOfName IEC_TIMER
"IEC_TIMER"
BEGIN
END_DATA_BLOCK

DATA_BLOCK "IEC_Timer_0_DB_48"   // DB59
{ S7_Optimized_Access := 'TRUE' }
AUTHOR : Simatic
FAMILY : IEC
NAME : IEC_TMR
VERSION : 1.0
// stored: InstanceOfName IEC_TIMER
"IEC_TIMER"
BEGIN
END_DATA_BLOCK

DATA_BLOCK "IEC_Timer_0_DB_49"   // DB60
{ S7_Optimized_Access := 'TRUE' }
AUTHOR : Simatic
FAMILY : IEC
NAME : IEC_TMR
VERSION : 1.0
// stored: InstanceOfName IEC_TIMER
"IEC_TIMER"
BEGIN
END_DATA_BLOCK

DATA_BLOCK "IEC_Timer_0_DB_50"   // DB61
{ S7_Optimized_Access := 'TRUE' }
AUTHOR : Simatic
FAMILY : IEC
NAME : IEC_TMR
VERSION : 1.0
// stored: InstanceOfName IEC_TIMER
"IEC_TIMER"
BEGIN
END_DATA_BLOCK

DATA_BLOCK "IEC_Timer_0_DB_51"   // DB62
{ S7_Optimized_Access := 'TRUE' }
AUTHOR : Simatic
FAMILY : IEC
NAME : IEC_TMR
VERSION : 1.0
// stored: InstanceOfName IEC_TIMER
"IEC_TIMER"
BEGIN
END_DATA_BLOCK

DATA_BLOCK "IEC_Timer_0_DB_55"   // DB66
{ S7_Optimized_Access := 'TRUE' }
AUTHOR : Simatic
FAMILY : IEC
NAME : IEC_TMR
VERSION : 1.0
// stored: InstanceOfName IEC_TIMER
"IEC_TIMER"
BEGIN
END_DATA_BLOCK

DATA_BLOCK "IEC_Timer_0_DB_57"   // DB68
{ S7_Optimized_Access := 'TRUE' }
AUTHOR : Simatic
FAMILY : IEC
NAME : IEC_TMR
VERSION : 1.0
// stored: InstanceOfName IEC_TIMER
"IEC_TIMER"
BEGIN
END_DATA_BLOCK

DATA_BLOCK "IEC_Timer_0_DB_58"   // DB69
{ S7_Optimized_Access := 'TRUE' }
AUTHOR : Simatic
FAMILY : IEC
NAME : IEC_TMR
VERSION : 1.0
// stored: InstanceOfName IEC_TIMER
"IEC_TIMER"
BEGIN
END_DATA_BLOCK

DATA_BLOCK "IEC_Timer_0_DB_59"   // DB70
{ S7_Optimized_Access := 'TRUE' }
AUTHOR : Simatic
FAMILY : IEC
NAME : IEC_TMR
VERSION : 1.0
// stored: InstanceOfName IEC_TIMER
"IEC_TIMER"
BEGIN
END_DATA_BLOCK

DATA_BLOCK "IEC_Timer_0_DB_60"   // DB71
{ S7_Optimized_Access := 'TRUE' }
AUTHOR : Simatic
FAMILY : IEC
NAME : IEC_TMR
VERSION : 1.0
// stored: InstanceOfName IEC_TIMER
"IEC_TIMER"
BEGIN
END_DATA_BLOCK

DATA_BLOCK "IEC_Timer_0_DB_66"   // DB77
{ S7_Optimized_Access := 'TRUE' }
AUTHOR : Simatic
FAMILY : IEC
NAME : IEC_TMR
VERSION : 1.0
// stored: InstanceOfName IEC_TIMER
"IEC_TIMER"
BEGIN
END_DATA_BLOCK

DATA_BLOCK "IEC_Timer_0_DB_67"   // DB80
{ S7_Optimized_Access := 'TRUE' }
AUTHOR : Simatic
FAMILY : IEC
NAME : IEC_TMR
VERSION : 1.0
// stored: InstanceOfName IEC_TIMER
"IEC_TIMER"
BEGIN
END_DATA_BLOCK

DATA_BLOCK "IEC_Timer_0_DB_68"   // DB81
{ S7_Optimized_Access := 'TRUE' }
AUTHOR : Simatic
FAMILY : IEC
NAME : IEC_TMR
VERSION : 1.0
// stored: InstanceOfName IEC_TIMER
"IEC_TIMER"
BEGIN
END_DATA_BLOCK

DATA_BLOCK "IEC_Timer_0_DB_69"   // DB82
{ S7_Optimized_Access := 'TRUE' }
AUTHOR : Simatic
FAMILY : IEC
NAME : IEC_TMR
VERSION : 1.0
// stored: InstanceOfName IEC_TIMER
"IEC_TIMER"
BEGIN
END_DATA_BLOCK

DATA_BLOCK "IEC_Timer_0_DB_70"   // DB83
{ S7_Optimized_Access := 'TRUE' }
AUTHOR : Simatic
FAMILY : IEC
NAME : IEC_TMR
VERSION : 1.0
// stored: InstanceOfName IEC_TIMER
"IEC_TIMER"
BEGIN
END_DATA_BLOCK

DATA_BLOCK "IEC_Timer_0_DB_71"   // DB84
{ S7_Optimized_Access := 'TRUE' }
AUTHOR : Simatic
FAMILY : IEC
NAME : IEC_TMR
VERSION : 1.0
// stored: InstanceOfName IEC_TIMER
"IEC_TIMER"
BEGIN
END_DATA_BLOCK

DATA_BLOCK "IEC_Timer_0_DB_72"   // DB85
{ S7_Optimized_Access := 'TRUE' }
AUTHOR : Simatic
FAMILY : IEC
NAME : IEC_TMR
VERSION : 1.0
// stored: InstanceOfName IEC_TIMER
"IEC_TIMER"
BEGIN
END_DATA_BLOCK

DATA_BLOCK "IEC_Timer_0_DB_73"   // DB86
{ S7_Optimized_Access := 'TRUE' }
AUTHOR : Simatic
FAMILY : IEC
NAME : IEC_TMR
VERSION : 1.0
// stored: InstanceOfName IEC_TIMER
"IEC_TIMER"
BEGIN
END_DATA_BLOCK

DATA_BLOCK "IEC_Timer_0_DB_74"   // DB87
{ S7_Optimized_Access := 'TRUE' }
AUTHOR : Simatic
FAMILY : IEC
NAME : IEC_TMR
VERSION : 1.0
// stored: InstanceOfName IEC_TIMER
"IEC_TIMER"
BEGIN
END_DATA_BLOCK

DATA_BLOCK "IEC_Timer_0_DB_75"   // DB88
{ S7_Optimized_Access := 'TRUE' }
AUTHOR : Simatic
FAMILY : IEC
NAME : IEC_TMR
VERSION : 1.0
// stored: InstanceOfName IEC_TIMER
"IEC_TIMER"
BEGIN
END_DATA_BLOCK

DATA_BLOCK "IEC_Timer_0_DB_76"   // DB89
{ S7_Optimized_Access := 'TRUE' }
AUTHOR : Simatic
FAMILY : IEC
NAME : IEC_TMR
VERSION : 1.0
// stored: InstanceOfName IEC_TIMER
"IEC_TIMER"
BEGIN
END_DATA_BLOCK

DATA_BLOCK "IEC_Timer_0_DB_77"   // DB90
{ S7_Optimized_Access := 'TRUE' }
AUTHOR : Simatic
FAMILY : IEC
NAME : IEC_TMR
VERSION : 1.0
// stored: InstanceOfName IEC_TIMER
"IEC_TIMER"
BEGIN
END_DATA_BLOCK

DATA_BLOCK "IEC_Timer_0_DB_78"   // DB91
{ S7_Optimized_Access := 'TRUE' }
AUTHOR : Simatic
FAMILY : IEC
NAME : IEC_TMR
VERSION : 1.0
// stored: InstanceOfName IEC_TIMER
"IEC_TIMER"
BEGIN
END_DATA_BLOCK

DATA_BLOCK "IEC_Timer_0_DB_79"   // DB92
{ S7_Optimized_Access := 'TRUE' }
AUTHOR : Simatic
FAMILY : IEC
NAME : IEC_TMR
VERSION : 1.0
// stored: InstanceOfName IEC_TIMER
"IEC_TIMER"
BEGIN
END_DATA_BLOCK

DATA_BLOCK "IEC_Timer_0_DB_80"   // DB93
{ S7_Optimized_Access := 'TRUE' }
AUTHOR : Simatic
FAMILY : IEC
NAME : IEC_TMR
VERSION : 1.0
// stored: InstanceOfName IEC_TIMER
"IEC_TIMER"
BEGIN
END_DATA_BLOCK

// folder: (top level)

FUNCTION_BLOCK "TESTING_SEQUENCE"   // FB1, LAD
{ S7_Optimized_Access := 'TRUE' }
VERSION : 0.1
   VAR_INPUT
      start : Bool;
      "ELECTRICAL PART LOAD" : Bool;
      "VISION TEST PART LOADED" : Bool;
      RESET : Bool;
      ELECTRICAL_TEST_START : Bool;
      ELEC_OK : Bool;
      ELEC_NG : Bool;
      NG_BIT : Bool;
      LOCK3_HOME : Bool;
      LOCK3_FEED : Bool;
      LOGO_TEST_START : Bool;
      LOGO_RSLT_OK : Bool;
      LOGO_RSLT_NG : Bool;
      LED_RSLT_OK : Bool;
      LED_RSLT_NG : Bool;
   END_VAR
   VAR_OUTPUT
      ELECTRICAL_TEST_COMPLETED : Bool;
      VISION_TEST_COMPLETED : Bool;
      CAM_TRG : Bool;
      TEST_ABORT : Bool;
      LOGO_TEST_COMPLETED : Bool;
      PROGRAM_NO : Int;
      CAM1_TRG : Bool;
      CAM2_TRG : Bool;
      GREEN_LED_ON : Bool;
      RED_LED_ON : Bool;
      BLUE_LED_ON : Bool;
      AMBER_LED_ON : Bool;
      PROGRAM_TRIGGER : Bool;
   END_VAR
   VAR_IN_OUT
      ELEC_SEQ : Int;
      TEST_SEQ : Int;
   END_VAR
   VAR
      "START BIT" : Bool;
      LOGO_TRG : Bool;
      GREEN_TRG : Bool;
      RED_TRG : Bool;
      BLUE_TRG : Bool;
      prog_trg5 : Bool;
      AMBER_TRG : Bool;
      "PROG_TRG 4" : Bool;
      CAM_TRG1 : Bool;
      CAM_TRG2 : Bool;
      CAM_TRG3 : Bool;
   END_VAR
   VAR_TEMP
      PRG0_TRG : Bool;
      PRG1_TRG : Bool;
      PRG2_TRG : Bool;
      PRG3_TRG : Bool;
      BUFF_CLR1 : Bool;
      BUFF_CLR2 : Bool;
      BUFF_CLR3 : Bool;
      BUFF_CLR4 : Bool;
      BUFF_CLR5 : Bool;
      BUFF_CLR6 : Bool;
      BUFF_CLR7 : Bool;
      BUFF_CLR8 : Bool;
      CAM2_TRG0 : Bool;
      CAM2_TRG1 : Bool;
      CAM2_TRG2 : Bool;
      CAM2_TRG3 : Bool;
      CAM1_TRG1 : Bool;
   END_VAR
   VAR_TEMP   // added for the SCL form of the ladder/FBD networks
      _w1 : Bool;
      _w2 : Bool;
      _w3 : Bool;
      _w4 : Bool;
      _w5 : Bool;
   END_VAR
BEGIN

REGION Network 1: LOGO_CHECKING_TRG
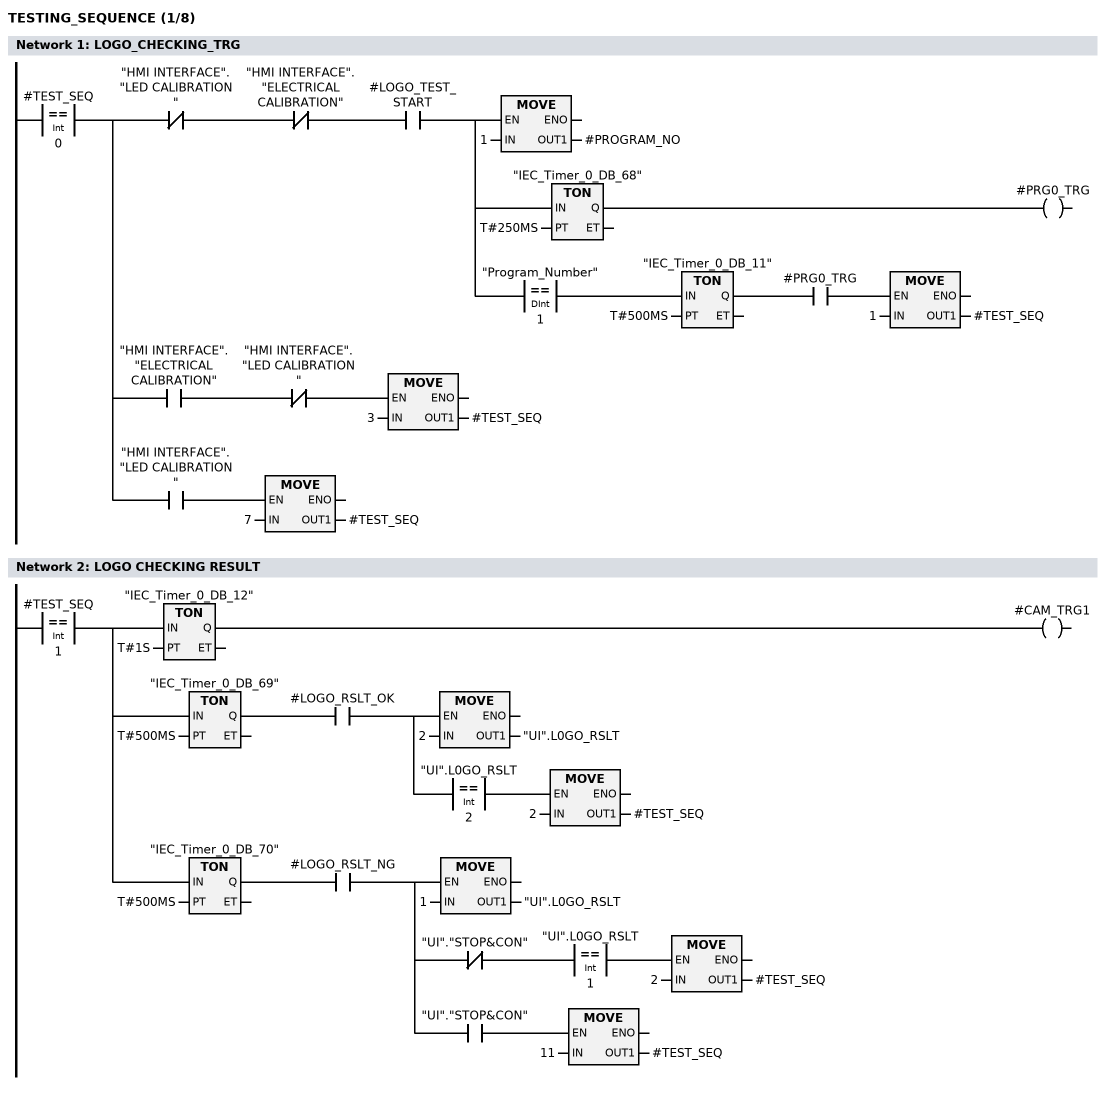
   #_w1 := #TEST_SEQ = 0;
   #_w2 := #_w1 AND NOT "HMI INTERFACE"."LED CALIBRATION" AND NOT "HMI INTERFACE"."ELECTRICAL CALIBRATION" AND #LOGO_TEST_START;
   IF #_w2 THEN #PROGRAM_NO := 1; END_IF;
   "IEC_Timer_0_DB_68".TON(IN := #_w2, PT := T#250MS);
   #PRG0_TRG := "IEC_Timer_0_DB_68".Q;
   "IEC_Timer_0_DB_11".TON(IN := #_w2 AND ("Program_Number" = 1), PT := T#500MS);
   IF "IEC_Timer_0_DB_11".Q AND #PRG0_TRG THEN #TEST_SEQ := 1; END_IF;
   IF #_w1 AND "HMI INTERFACE"."ELECTRICAL CALIBRATION" AND NOT "HMI INTERFACE"."LED CALIBRATION" THEN
       #TEST_SEQ := 3;
   END_IF;
   IF #_w1 AND "HMI INTERFACE"."LED CALIBRATION" THEN #TEST_SEQ := 7; END_IF;
END_REGION

REGION Network 2: LOGO CHECKING RESULT
   #_w1 := #TEST_SEQ = 1;
   "IEC_Timer_0_DB_12".TON(IN := #_w1, PT := T#1S);
   #CAM_TRG1 := "IEC_Timer_0_DB_12".Q;
   "IEC_Timer_0_DB_69".TON(IN := #_w1, PT := T#500MS);
   #_w2 := "IEC_Timer_0_DB_69".Q AND #LOGO_RSLT_OK;
   IF #_w2 THEN "UI".L0GO_RSLT := 2; END_IF;
   IF #_w2 AND ("UI".L0GO_RSLT = 2) THEN #TEST_SEQ := 2; END_IF;
   "IEC_Timer_0_DB_70".TON(IN := #_w1, PT := T#500MS);
   #_w3 := "IEC_Timer_0_DB_70".Q AND #LOGO_RSLT_NG;
   IF #_w3 THEN "UI".L0GO_RSLT := 1; END_IF;
   IF #_w3 AND NOT "UI"."STOP&CON" AND ("UI".L0GO_RSLT = 1) THEN #TEST_SEQ := 2; END_IF;
   IF #_w3 AND "UI"."STOP&CON" THEN #TEST_SEQ := 11; END_IF;
END_REGION

REGION Network 3: LOGO_TEST_COMPLETED
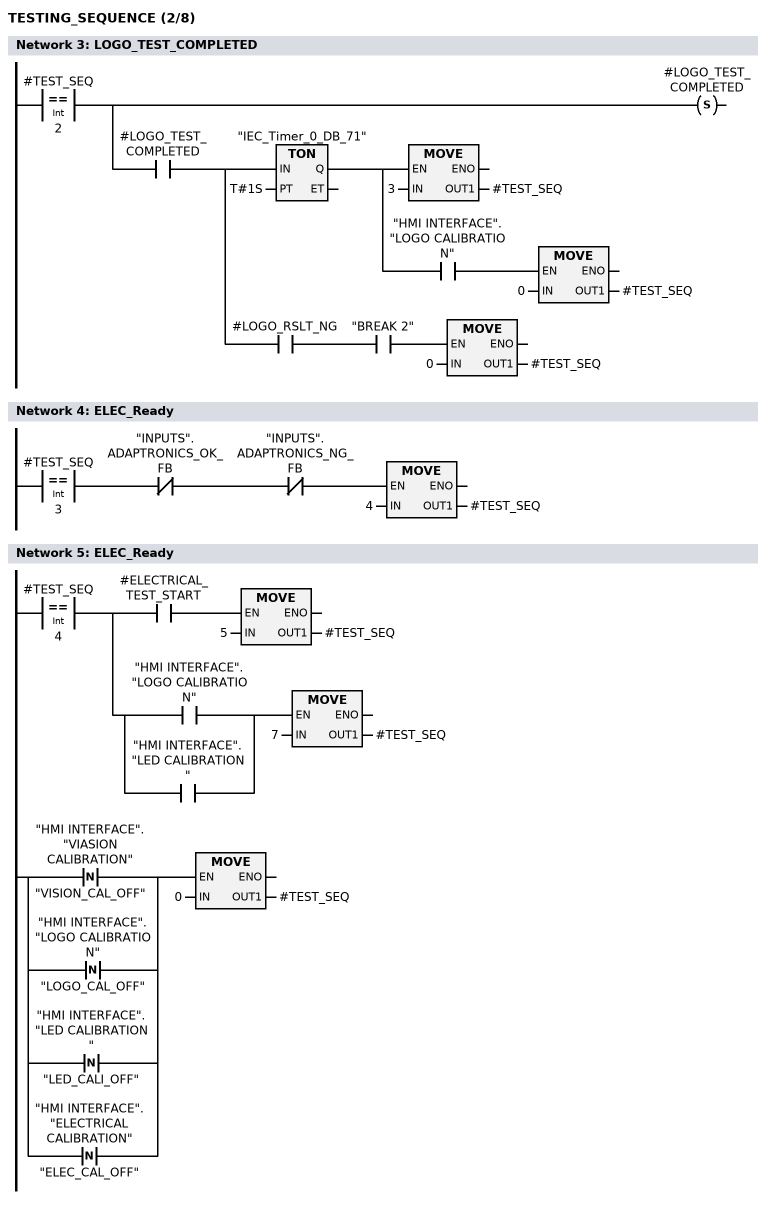
   #_w1 := #TEST_SEQ = 2;
   IF #_w1 THEN #LOGO_TEST_COMPLETED := TRUE; END_IF;
   #_w2 := #_w1 AND #LOGO_TEST_COMPLETED;
   "IEC_Timer_0_DB_71".TON(IN := #_w2, PT := T#1S);
   IF "IEC_Timer_0_DB_71".Q THEN #TEST_SEQ := 3; END_IF;
   IF "IEC_Timer_0_DB_71".Q AND "HMI INTERFACE"."LOGO CALIBRATION" THEN #TEST_SEQ := 0; END_IF;
   IF #_w2 AND #LOGO_RSLT_NG AND "BREAK 2" THEN #TEST_SEQ := 0; END_IF;
END_REGION

REGION Network 4: ELEC_Ready
   RUNG wire#powerrail
      { S7_Templates := "SrcType := Int" } EQ_Contact(in1 := #TEST_SEQ, in2 := 3)
      I_Contact( "INPUTS".ADAPTRONICS_OK_FB )
      I_Contact( "INPUTS".ADAPTRONICS_NG_FB )
      Move(in := 4, out1 => #TEST_SEQ)
   END_RUNG
   // the same network as SCL:
   IF (#TEST_SEQ = 3) AND NOT "INPUTS".ADAPTRONICS_OK_FB AND NOT "INPUTS".ADAPTRONICS_NG_FB THEN
       #TEST_SEQ := 4;
   END_IF;
END_REGION

REGION Network 5: ELEC_Ready
   RUNG wire#powerrail
      { S7_Templates := "SrcType := Int" } EQ_Contact(in1 := #TEST_SEQ, in2 := 4)
      wire#w1
      Contact( #ELECTRICAL_TEST_START )
      Move(in := 5, out1 => #TEST_SEQ)
   END_RUNG
   RUNG wire#w1
      Contact( "HMI INTERFACE"."LOGO CALIBRATION" )
      wire#w2
      Move(in := 7, out1 => #TEST_SEQ)
   END_RUNG
   RUNG wire#w1
      Contact( "HMI INTERFACE"."LED CALIBRATION" )
   END_RUNG wire#w2
   RUNG wire#powerrail
      N_Contact(operand := "HMI INTERFACE"."VIASION CALIBRATION", bit := "VISION_CAL_OFF")
      wire#w3
      Move(in := 0, out1 => #TEST_SEQ)
   END_RUNG
   RUNG wire#powerrail
      N_Contact(operand := "HMI INTERFACE"."LOGO CALIBRATION", bit := "LOGO_CAL_OFF")
   END_RUNG wire#w3
   RUNG wire#powerrail
      N_Contact(operand := "HMI INTERFACE"."LED CALIBRATION", bit := "LED_CALI_OFF")
   END_RUNG wire#w3
   RUNG wire#powerrail
      N_Contact(operand := "HMI INTERFACE"."ELECTRICAL CALIBRATION", bit := "ELEC_CAL_OFF")
   END_RUNG wire#w3
   // the same network as SCL:
   #_w1 := #TEST_SEQ = 4;
   IF #_w1 AND #ELECTRICAL_TEST_START THEN #TEST_SEQ := 5; END_IF;
   IF #_w1 AND ("HMI INTERFACE"."LOGO CALIBRATION" OR "HMI INTERFACE"."LED CALIBRATION") THEN
       #TEST_SEQ := 7;
   END_IF;
   #_w2 := NOT "HMI INTERFACE"."VIASION CALIBRATION" AND "VISION_CAL_OFF";   // falling edge of "HMI INTERFACE"."VIASION CALIBRATION"
   "VISION_CAL_OFF" := "HMI INTERFACE"."VIASION CALIBRATION";
   #_w3 := NOT "HMI INTERFACE"."LOGO CALIBRATION" AND "LOGO_CAL_OFF";   // falling edge of "HMI INTERFACE"."LOGO CALIBRATION"
   "LOGO_CAL_OFF" := "HMI INTERFACE"."LOGO CALIBRATION";
   #_w4 := NOT "HMI INTERFACE"."LED CALIBRATION" AND "LED_CALI_OFF";   // falling edge of "HMI INTERFACE"."LED CALIBRATION"
   "LED_CALI_OFF" := "HMI INTERFACE"."LED CALIBRATION";
   #_w5 := NOT "HMI INTERFACE"."ELECTRICAL CALIBRATION" AND "ELEC_CAL_OFF";   // falling edge of "HMI INTERFACE"."ELECTRICAL CALIBRATION"
   "ELEC_CAL_OFF" := "HMI INTERFACE"."ELECTRICAL CALIBRATION";
   IF #_w2 OR #_w3 OR #_w4 OR #_w5 THEN #TEST_SEQ := 0; END_IF;
END_REGION

REGION Network 6: ELECTRICAL_TEST
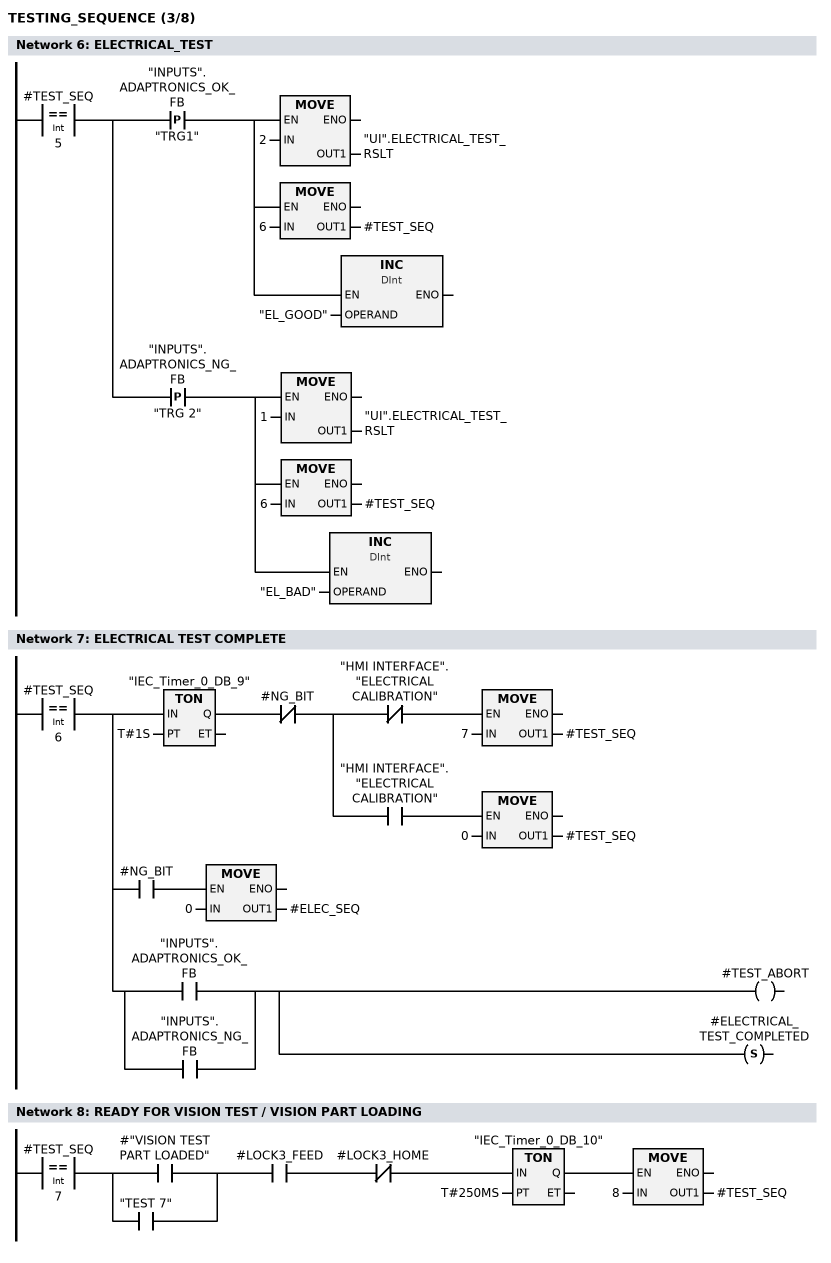
   RUNG wire#powerrail
      { S7_Templates := "SrcType := Int" } EQ_Contact(in1 := #TEST_SEQ, in2 := 5)
      wire#w1
      P_Contact(operand := "INPUTS".ADAPTRONICS_OK_FB, bit := "TRG1")
      wire#w2
      Move(in := 2, out1 => "UI".ELECTRICAL_TEST_RSLT)
   END_RUNG
   RUNG wire#w2
      Move(in := 6, out1 => #TEST_SEQ)
   END_RUNG
   RUNG wire#w2
      { S7_Templates := "DestType := DInt" } Inc( "EL_GOOD" )
   END_RUNG
   RUNG wire#w1
      P_Contact(operand := "INPUTS".ADAPTRONICS_NG_FB, bit := "TRG 2")
      wire#w3
      Move(in := 1, out1 => "UI".ELECTRICAL_TEST_RSLT)
   END_RUNG
   RUNG wire#w3
      Move(in := 6, out1 => #TEST_SEQ)
   END_RUNG
   RUNG wire#w3
      { S7_Templates := "DestType := DInt" } Inc( "EL_BAD" )
   END_RUNG
   // the same network as SCL:
   #_w1 := #TEST_SEQ = 5;
   #_w2 := #_w1 AND "INPUTS".ADAPTRONICS_OK_FB AND NOT "TRG1";   // rising edge of "INPUTS".ADAPTRONICS_OK_FB
   "TRG1" := "INPUTS".ADAPTRONICS_OK_FB;
   IF #_w2 THEN
       "UI".ELECTRICAL_TEST_RSLT := 2;
       #TEST_SEQ := 6;
       "EL_GOOD" := "EL_GOOD" + 1;
   END_IF;
   #_w3 := #_w1 AND "INPUTS".ADAPTRONICS_NG_FB AND NOT "TRG 2";   // rising edge of "INPUTS".ADAPTRONICS_NG_FB
   "TRG 2" := "INPUTS".ADAPTRONICS_NG_FB;
   IF #_w3 THEN
       "UI".ELECTRICAL_TEST_RSLT := 1;
       #TEST_SEQ := 6;
       "EL_BAD" := "EL_BAD" + 1;
   END_IF;
END_REGION

REGION Network 7: ELECTRICAL TEST COMPLETE
   #_w1 := #TEST_SEQ = 6;
   "IEC_Timer_0_DB_9".TON(IN := #_w1, PT := T#1S);
   #_w2 := "IEC_Timer_0_DB_9".Q AND NOT #NG_BIT;
   IF #_w2 AND NOT "HMI INTERFACE"."ELECTRICAL CALIBRATION" THEN #TEST_SEQ := 7; END_IF;
   IF #_w2 AND "HMI INTERFACE"."ELECTRICAL CALIBRATION" THEN #TEST_SEQ := 0; END_IF;
   IF #_w1 AND #NG_BIT THEN #ELEC_SEQ := 0; END_IF;
   #TEST_ABORT := #_w1 AND ("INPUTS".ADAPTRONICS_OK_FB OR "INPUTS".ADAPTRONICS_NG_FB);
   IF #TEST_ABORT THEN #ELECTRICAL_TEST_COMPLETED := TRUE; END_IF;
END_REGION

REGION Network 8: READY FOR VISION TEST / VISION PART LOADING
   "IEC_Timer_0_DB_10".TON(IN := (#TEST_SEQ = 7) AND (#"VISION TEST PART LOADED" OR "TEST 7") AND #LOCK3_FEED AND NOT #LOCK3_HOME,
                           PT := T#250MS);
   IF "IEC_Timer_0_DB_10".Q THEN #TEST_SEQ := 8; END_IF;
END_REGION

REGION Network 9: GREEN_LED_SWITCHING
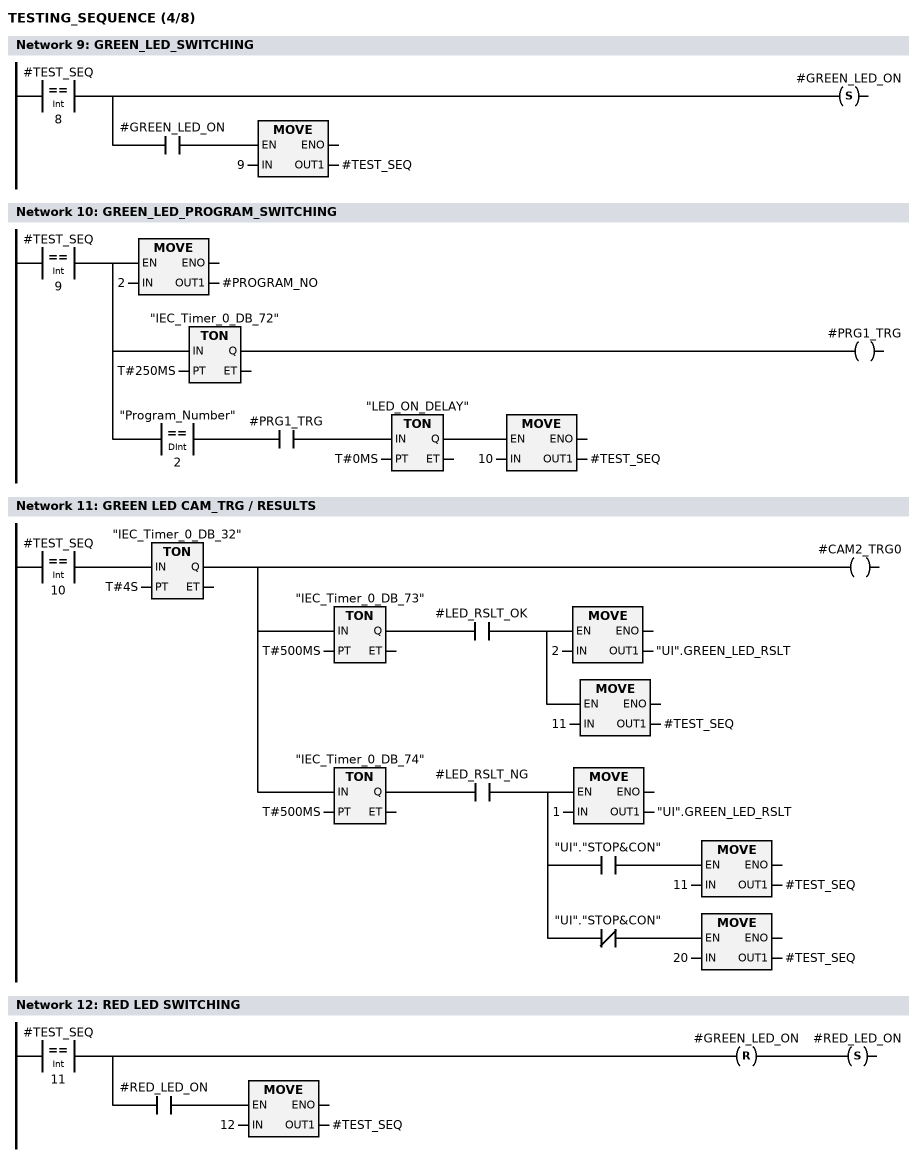
   RUNG wire#powerrail
      { S7_Templates := "SrcType := Int" } EQ_Contact(in1 := #TEST_SEQ, in2 := 8)
      wire#w1
      S_Coil( #GREEN_LED_ON )
   END_RUNG
   RUNG wire#w1
      Contact( #GREEN_LED_ON )
      Move(in := 9, out1 => #TEST_SEQ)
   END_RUNG
   // the same network as SCL:
   #_w1 := #TEST_SEQ = 8;
   IF #_w1 THEN #GREEN_LED_ON := TRUE; END_IF;
   IF #_w1 AND #GREEN_LED_ON THEN #TEST_SEQ := 9; END_IF;
END_REGION

REGION Network 10: GREEN_LED_PROGRAM_SWITCHING
   #_w1 := #TEST_SEQ = 9;
   IF #_w1 THEN #PROGRAM_NO := 2; END_IF;
   "IEC_Timer_0_DB_72".TON(IN := #_w1, PT := T#250MS);
   #PRG1_TRG := "IEC_Timer_0_DB_72".Q;
   "LED_ON_DELAY".TON(IN := #_w1 AND ("Program_Number" = 2) AND #PRG1_TRG, PT := T#0MS);
   IF "LED_ON_DELAY".Q THEN #TEST_SEQ := 10; END_IF;
END_REGION

REGION Network 11: GREEN LED CAM_TRG / RESULTS
   "IEC_Timer_0_DB_32".TON(IN := #TEST_SEQ = 10, PT := T#4S);
   #CAM2_TRG0 := "IEC_Timer_0_DB_32".Q;
   "IEC_Timer_0_DB_73".TON(IN := "IEC_Timer_0_DB_32".Q, PT := T#500MS);
   IF "IEC_Timer_0_DB_73".Q AND #LED_RSLT_OK THEN
       "UI".GREEN_LED_RSLT := 2;
       #TEST_SEQ := 11;
   END_IF;
   "IEC_Timer_0_DB_74".TON(IN := "IEC_Timer_0_DB_32".Q, PT := T#500MS);
   #_w1 := "IEC_Timer_0_DB_74".Q AND #LED_RSLT_NG;
   IF #_w1 THEN "UI".GREEN_LED_RSLT := 1; END_IF;
   IF #_w1 AND "UI"."STOP&CON" THEN #TEST_SEQ := 11; END_IF;
   IF #_w1 AND NOT "UI"."STOP&CON" THEN #TEST_SEQ := 20; END_IF;
END_REGION

REGION Network 12: RED LED SWITCHING
   RUNG wire#powerrail
      { S7_Templates := "SrcType := Int" } EQ_Contact(in1 := #TEST_SEQ, in2 := 11)
      wire#w1
      R_Coil( #GREEN_LED_ON )
      S_Coil( #RED_LED_ON )
   END_RUNG
   RUNG wire#w1
      Contact( #RED_LED_ON )
      Move(in := 12, out1 => #TEST_SEQ)
   END_RUNG
   // the same network as SCL:
   #_w1 := #TEST_SEQ = 11;
   IF #_w1 THEN
       #GREEN_LED_ON := FALSE;
       #RED_LED_ON := TRUE;
   END_IF;
   IF #_w1 AND #RED_LED_ON THEN #TEST_SEQ := 12; END_IF;
END_REGION

REGION Network 13: RED_LED_PROGRAM_SWITCHING
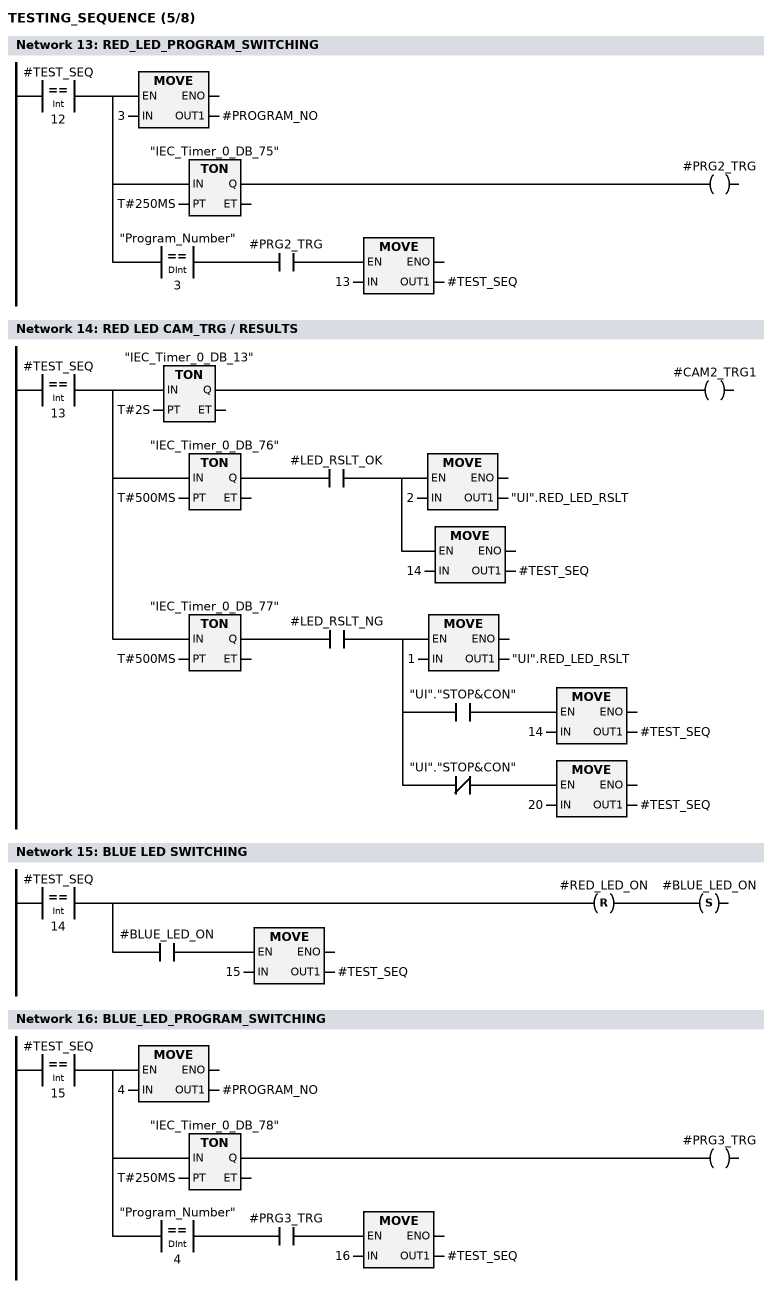
   #_w1 := #TEST_SEQ = 12;
   IF #_w1 THEN #PROGRAM_NO := 3; END_IF;
   "IEC_Timer_0_DB_75".TON(IN := #_w1, PT := T#250MS);
   #PRG2_TRG := "IEC_Timer_0_DB_75".Q;
   IF #_w1 AND ("Program_Number" = 3) AND #PRG2_TRG THEN #TEST_SEQ := 13; END_IF;
END_REGION

REGION Network 14: RED LED CAM_TRG / RESULTS
   #_w1 := #TEST_SEQ = 13;
   "IEC_Timer_0_DB_13".TON(IN := #_w1, PT := T#2S);
   #CAM2_TRG1 := "IEC_Timer_0_DB_13".Q;
   "IEC_Timer_0_DB_76".TON(IN := #_w1, PT := T#500MS);
   IF "IEC_Timer_0_DB_76".Q AND #LED_RSLT_OK THEN
       "UI".RED_LED_RSLT := 2;
       #TEST_SEQ := 14;
   END_IF;
   "IEC_Timer_0_DB_77".TON(IN := #_w1, PT := T#500MS);
   #_w2 := "IEC_Timer_0_DB_77".Q AND #LED_RSLT_NG;
   IF #_w2 THEN "UI".RED_LED_RSLT := 1; END_IF;
   IF #_w2 AND "UI"."STOP&CON" THEN #TEST_SEQ := 14; END_IF;
   IF #_w2 AND NOT "UI"."STOP&CON" THEN #TEST_SEQ := 20; END_IF;
END_REGION

REGION Network 15: BLUE LED SWITCHING
   RUNG wire#powerrail
      { S7_Templates := "SrcType := Int" } EQ_Contact(in1 := #TEST_SEQ, in2 := 14)
      wire#w1
      R_Coil( #RED_LED_ON )
      S_Coil( #BLUE_LED_ON )
   END_RUNG
   RUNG wire#w1
      Contact( #BLUE_LED_ON )
      Move(in := 15, out1 => #TEST_SEQ)
   END_RUNG
   // the same network as SCL:
   #_w1 := #TEST_SEQ = 14;
   IF #_w1 THEN
       #RED_LED_ON := FALSE;
       #BLUE_LED_ON := TRUE;
   END_IF;
   IF #_w1 AND #BLUE_LED_ON THEN #TEST_SEQ := 15; END_IF;
END_REGION

REGION Network 16: BLUE_LED_PROGRAM_SWITCHING
   #_w1 := #TEST_SEQ = 15;
   IF #_w1 THEN #PROGRAM_NO := 4; END_IF;
   "IEC_Timer_0_DB_78".TON(IN := #_w1, PT := T#250MS);
   #PRG3_TRG := "IEC_Timer_0_DB_78".Q;
   IF #_w1 AND ("Program_Number" = 4) AND #PRG3_TRG THEN #TEST_SEQ := 16; END_IF;
END_REGION

REGION Network 17: RED LED CAM_TRG / RESULTS
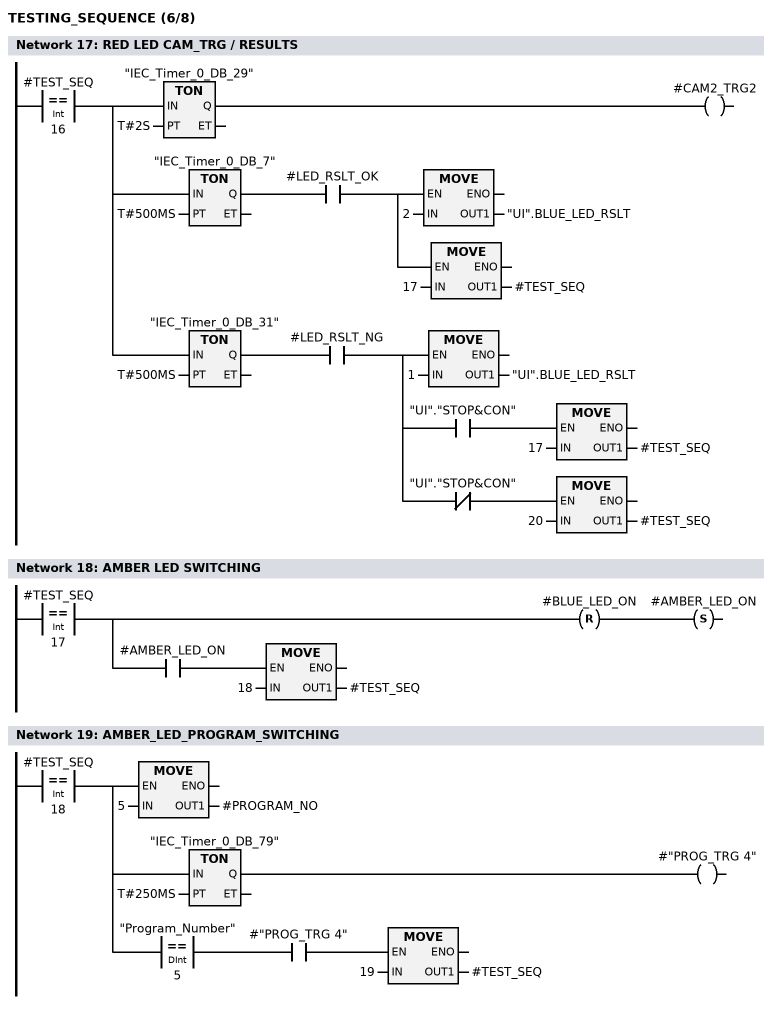
   #_w1 := #TEST_SEQ = 16;
   "IEC_Timer_0_DB_29".TON(IN := #_w1, PT := T#2S);
   #CAM2_TRG2 := "IEC_Timer_0_DB_29".Q;
   "IEC_Timer_0_DB_7".TON(IN := #_w1, PT := T#500MS);
   IF "IEC_Timer_0_DB_7".Q AND #LED_RSLT_OK THEN
       "UI".BLUE_LED_RSLT := 2;
       #TEST_SEQ := 17;
   END_IF;
   "IEC_Timer_0_DB_31".TON(IN := #_w1, PT := T#500MS);
   #_w2 := "IEC_Timer_0_DB_31".Q AND #LED_RSLT_NG;
   IF #_w2 THEN "UI".BLUE_LED_RSLT := 1; END_IF;
   IF #_w2 AND "UI"."STOP&CON" THEN #TEST_SEQ := 17; END_IF;
   IF #_w2 AND NOT "UI"."STOP&CON" THEN #TEST_SEQ := 20; END_IF;
END_REGION

REGION Network 18: AMBER LED SWITCHING
   RUNG wire#powerrail
      { S7_Templates := "SrcType := Int" } EQ_Contact(in1 := #TEST_SEQ, in2 := 17)
      wire#w1
      R_Coil( #BLUE_LED_ON )
      S_Coil( #AMBER_LED_ON )
   END_RUNG
   RUNG wire#w1
      Contact( #AMBER_LED_ON )
      Move(in := 18, out1 => #TEST_SEQ)
   END_RUNG
   // the same network as SCL:
   #_w1 := #TEST_SEQ = 17;
   IF #_w1 THEN
       #BLUE_LED_ON := FALSE;
       #AMBER_LED_ON := TRUE;
   END_IF;
   IF #_w1 AND #AMBER_LED_ON THEN #TEST_SEQ := 18; END_IF;
END_REGION

REGION Network 19: AMBER_LED_PROGRAM_SWITCHING
   #_w1 := #TEST_SEQ = 18;
   IF #_w1 THEN #PROGRAM_NO := 5; END_IF;
   "IEC_Timer_0_DB_79".TON(IN := #_w1, PT := T#250MS);
   #"PROG_TRG 4" := "IEC_Timer_0_DB_79".Q;
   IF #_w1 AND ("Program_Number" = 5) AND #"PROG_TRG 4" THEN #TEST_SEQ := 19; END_IF;
END_REGION

REGION Network 20: AMBER LED CAM_TRG / RESULTS
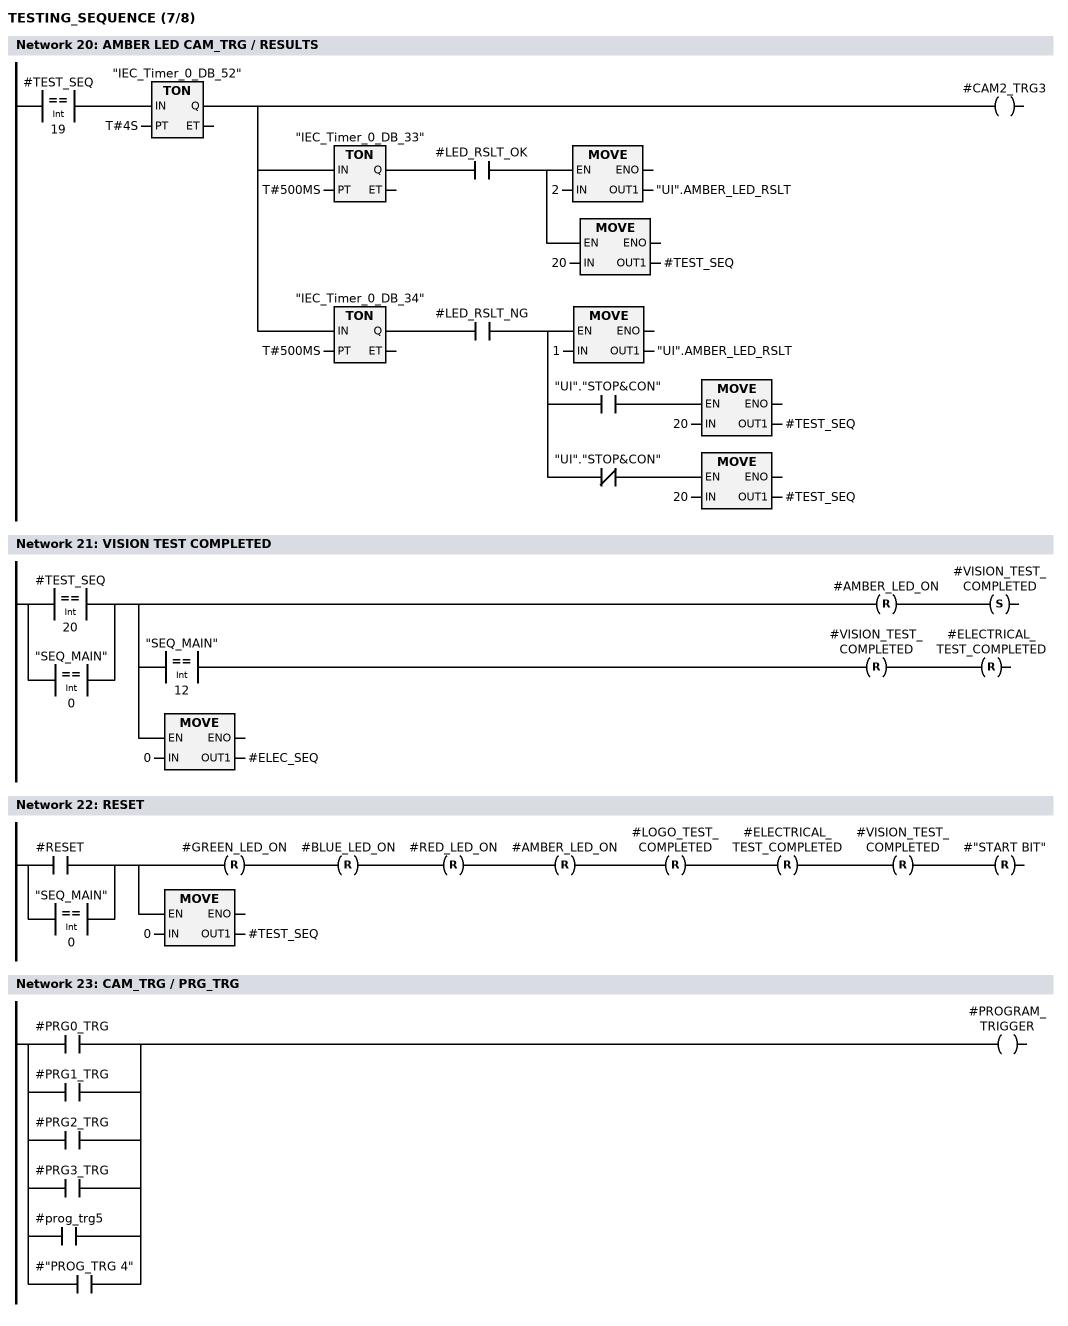
   "IEC_Timer_0_DB_52".TON(IN := #TEST_SEQ = 19, PT := T#4S);
   #CAM2_TRG3 := "IEC_Timer_0_DB_52".Q;
   "IEC_Timer_0_DB_33".TON(IN := "IEC_Timer_0_DB_52".Q, PT := T#500MS);
   IF "IEC_Timer_0_DB_33".Q AND #LED_RSLT_OK THEN
       "UI".AMBER_LED_RSLT := 2;
       #TEST_SEQ := 20;
   END_IF;
   "IEC_Timer_0_DB_34".TON(IN := "IEC_Timer_0_DB_52".Q, PT := T#500MS);
   #_w1 := "IEC_Timer_0_DB_34".Q AND #LED_RSLT_NG;
   IF #_w1 THEN "UI".AMBER_LED_RSLT := 1; END_IF;
   IF #_w1 AND "UI"."STOP&CON" THEN #TEST_SEQ := 20; END_IF;
   IF #_w1 AND NOT "UI"."STOP&CON" THEN #TEST_SEQ := 20; END_IF;
END_REGION

REGION Network 21: VISION TEST COMPLETED
   RUNG wire#powerrail
      { S7_Templates := "SrcType := Int" } EQ_Contact(in1 := #TEST_SEQ, in2 := 20)
      wire#w1
      R_Coil( #AMBER_LED_ON )
      S_Coil( #VISION_TEST_COMPLETED )
   END_RUNG
   RUNG wire#powerrail
      { S7_Templates := "SrcType := Int" } EQ_Contact(in1 := "SEQ_MAIN", in2 := 0)
   END_RUNG wire#w1
   RUNG wire#w1
      { S7_Templates := "SrcType := Int" } EQ_Contact(in1 := "SEQ_MAIN", in2 := 12)
      R_Coil( #VISION_TEST_COMPLETED )
      R_Coil( #ELECTRICAL_TEST_COMPLETED )
   END_RUNG
   RUNG wire#w1
      Move(in := 0, out1 => #ELEC_SEQ)
   END_RUNG
   // the same network as SCL:
   #_w1 := (#TEST_SEQ = 20) OR ("SEQ_MAIN" = 0);
   IF #_w1 THEN
       #AMBER_LED_ON := FALSE;
       #VISION_TEST_COMPLETED := TRUE;
   END_IF;
   IF #_w1 AND ("SEQ_MAIN" = 12) THEN
       #VISION_TEST_COMPLETED := FALSE;
       #ELECTRICAL_TEST_COMPLETED := FALSE;
   END_IF;
   IF #_w1 THEN #ELEC_SEQ := 0; END_IF;
END_REGION

REGION Network 22: RESET
   RUNG wire#powerrail
      Contact( #RESET )
      wire#w1
      R_Coil( #GREEN_LED_ON )
      R_Coil( #BLUE_LED_ON )
      R_Coil( #RED_LED_ON )
      R_Coil( #AMBER_LED_ON )
      R_Coil( #LOGO_TEST_COMPLETED )
      R_Coil( #ELECTRICAL_TEST_COMPLETED )
      R_Coil( #VISION_TEST_COMPLETED )
      R_Coil( #"START BIT" )
   END_RUNG
   RUNG wire#powerrail
      { S7_Templates := "SrcType := Int" } EQ_Contact(in1 := "SEQ_MAIN", in2 := 0)
   END_RUNG wire#w1
   RUNG wire#w1
      Move(in := 0, out1 => #TEST_SEQ)
   END_RUNG
   // the same network as SCL:
   IF #RESET OR ("SEQ_MAIN" = 0) THEN
       #GREEN_LED_ON := FALSE;
       #BLUE_LED_ON := FALSE;
       #RED_LED_ON := FALSE;
       #AMBER_LED_ON := FALSE;
       #LOGO_TEST_COMPLETED := FALSE;
       #ELECTRICAL_TEST_COMPLETED := FALSE;
       #VISION_TEST_COMPLETED := FALSE;
       #"START BIT" := FALSE;
       #TEST_SEQ := 0;
   END_IF;
END_REGION

REGION Network 23: CAM_TRG / PRG_TRG
   RUNG wire#powerrail
      Contact( #PRG0_TRG )
      wire#w1
      Coil( #PROGRAM_TRIGGER )
   END_RUNG
   RUNG wire#powerrail
      Contact( #PRG1_TRG )
   END_RUNG wire#w1
   RUNG wire#powerrail
      Contact( #PRG2_TRG )
   END_RUNG wire#w1
   RUNG wire#powerrail
      Contact( #PRG3_TRG )
   END_RUNG wire#w1
   RUNG wire#powerrail
      Contact( #prog_trg5 )
   END_RUNG wire#w1
   RUNG wire#powerrail
      Contact( #"PROG_TRG 4" )
   END_RUNG wire#w1
   // the same network as SCL:
   #PROGRAM_TRIGGER := #PRG0_TRG OR #PRG1_TRG OR #PRG2_TRG OR #PRG3_TRG OR #prog_trg5 OR #"PROG_TRG 4";
END_REGION

REGION Network 24: BUFFER_CLEAR
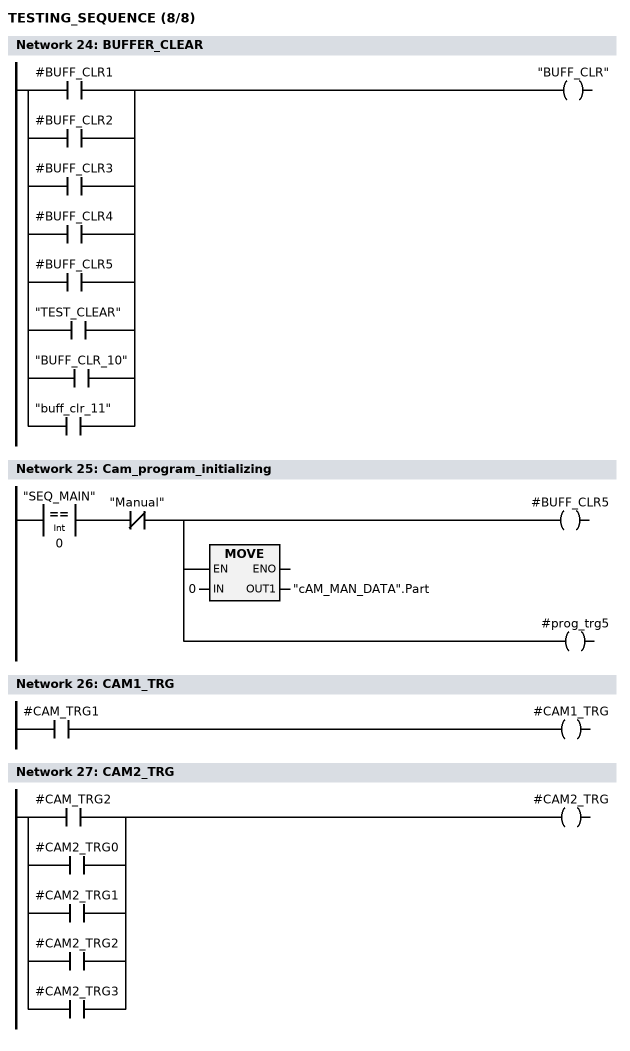
   RUNG wire#powerrail
      Contact( #BUFF_CLR1 )
      wire#w1
      Coil( "BUFF_CLR" )
   END_RUNG
   RUNG wire#powerrail
      Contact( #BUFF_CLR2 )
   END_RUNG wire#w1
   RUNG wire#powerrail
      Contact( #BUFF_CLR3 )
   END_RUNG wire#w1
   RUNG wire#powerrail
      Contact( #BUFF_CLR4 )
   END_RUNG wire#w1
   RUNG wire#powerrail
      Contact( #BUFF_CLR5 )
   END_RUNG wire#w1
   RUNG wire#powerrail
      Contact( "TEST_CLEAR" )
   END_RUNG wire#w1
   RUNG wire#powerrail
      Contact( "BUFF_CLR_10" )
   END_RUNG wire#w1
   RUNG wire#powerrail
      Contact( "buff_clr_11" )
   END_RUNG wire#w1
   // the same network as SCL:
   "BUFF_CLR" := #BUFF_CLR1 OR #BUFF_CLR2 OR #BUFF_CLR3 OR #BUFF_CLR4 OR #BUFF_CLR5 OR "TEST_CLEAR" OR "BUFF_CLR_10" OR "buff_clr_11";
END_REGION

REGION Network 25: Cam_program_initializing
   RUNG wire#powerrail
      { S7_Templates := "SrcType := Int" } EQ_Contact(in1 := "SEQ_MAIN", in2 := 0)
      I_Contact( "Manual" )
      wire#w1
      Coil( #BUFF_CLR5 )
   END_RUNG
   RUNG wire#w1
      Move(in := 0, out1 => "cAM_MAN_DATA".Part)
   END_RUNG
   RUNG wire#w1
      Coil( #prog_trg5 )
   END_RUNG
   // the same network as SCL:
   #BUFF_CLR5 := ("SEQ_MAIN" = 0) AND NOT "Manual";
   IF #BUFF_CLR5 THEN "cAM_MAN_DATA".Part := 0; END_IF;
   #prog_trg5 := #BUFF_CLR5;
END_REGION

REGION Network 26: CAM1_TRG
   RUNG wire#powerrail
      Contact( #CAM_TRG1 )
      Coil( #CAM1_TRG )
   END_RUNG
   // the same network as SCL:
   #CAM1_TRG := #CAM_TRG1;
END_REGION

REGION Network 27: CAM2_TRG
   RUNG wire#powerrail
      Contact( #CAM_TRG2 )
      wire#w1
      Coil( #CAM2_TRG )
   END_RUNG
   RUNG wire#powerrail
      Contact( #CAM2_TRG0 )
   END_RUNG wire#w1
   RUNG wire#powerrail
      Contact( #CAM2_TRG1 )
   END_RUNG wire#w1
   RUNG wire#powerrail
      Contact( #CAM2_TRG2 )
   END_RUNG wire#w1
   RUNG wire#powerrail
      Contact( #CAM2_TRG3 )
   END_RUNG wire#w1
   // the same network as SCL:
   #CAM2_TRG := #CAM_TRG2 OR #CAM2_TRG0 OR #CAM2_TRG1 OR #CAM2_TRG2 OR #CAM2_TRG3;
END_REGION
END_FUNCTION_BLOCK

FUNCTION_BLOCK "MAIN_SEQ"   // FB2, LAD
{ S7_Optimized_Access := 'TRUE' }
VERSION : 0.1
   VAR_INPUT
      "LCK1 REV" : Bool;
      "LCK1 FWD" : Bool;
      "LCK2 REV" : Bool;
      "LCK2 FWD" : Bool;
      "LCK3 REV" : Bool;
      "LCK3 FWD" : Bool;
      "PART1 PRESENCE" : Bool;
      "PART2 PRESENCE" : Bool;
      "PART3 PRESENCE" : Bool;
      LH_BOTTOM_CYL_DOWN : Bool;
      LH_BOTTOM_CYL_UP : Bool;
      RH_BOTTOM_CYL_DOWN : Bool;
      RH_BOTTOM_CYL_UP : Bool;
      START : Bool;
      "ELECTRICAL TEST COMPLETED" : Bool;
      VISION_TEST_COMPLETED : Bool;
      ADAPTRONICS_NG_FB : Bool;
      VISION_NG_FB : Bool;
      SCANNING_COMPLETED : Bool;
      MANUAL : Bool;
      SCAN_OK : Bool;
      CONVEYER_FB : Bool;
      REJECTION_FB : Bool;
      RESET : Bool;
      EMG : Bool;
      PUNCH1_FWD : Bool;
      PUNCH1_REV : Bool;
      PUNCH2_FWD : Bool;
      PUNCH2_REV : Bool;
      PRESSURE : Bool;
      "CHARGING CYL_FWD" : Bool;
      "CHARGING CYL_REV" : Bool;
      "LOGO LK_REV" : Bool;
      "LOGO LK_FWD" : Bool;
      "LOGO OPTIC_SENSR" : Bool;
      LOGO_TEST_CMPLTD : Bool;
      LOGO_RESULT_NG : Bool;
   END_VAR
   VAR_OUTPUT
      "LOCK 1" : Bool;
      "LOCK 2" : Bool;
      "LOCK 3" : Bool;
      "PUNCH 1" : Bool;
      "PUNCH 2" : Bool;
      LH_BOTTOM_DOWN : Bool;
      LH_BOTTOM_UP : Bool;
      RH_BOTTOM_DOWN : Bool;
      RH_BOTTOM_UP : Bool;
      ELECTRICAL_TEST_ABORT : Bool;
      ELECTRICAL_TEST_CONTINUE : Bool;
      "ELECTRICAL _TEST_START" : Bool;
      VISION_TEST_START : Bool;
      ELECTRICAL_PART_LOADED : Bool;
      VISION_PART_LOADED : Bool;
      RED_LED_ON : Bool;
      GREEN_LED_ON : Bool;
      BLUE_LED_ON : Bool;
      RED_BIT : Bool;
      GREEN_BIT : Bool;
      BLUE_BIT : Bool;
      GROUND_ON : Bool;
      TEST_RESULT : Int;
      NG_BIT : Bool;
      CAM_TRG : Bool;
      STATUS : Int;
      ELEC_CONTINUE : Bool;
      "VALUE RESET" : Int;
      BUZZ : Bool;
      conv_out : Bool;
      rej_out : Bool;
      GREEN_ILLU : Bool;
      TOWER_READY : Bool;
      TOWER_RUNNING : Bool;
      TOWER_STOP : Bool;
      "LOGO LK_ON" : Bool;
      "CHARGING CYL_ON" : Bool;
      LOGO_TEST_START : Bool;
   END_VAR
   VAR_IN_OUT
      SEQ : Int;
      RST_SEQ : Int;
      MOTOR_ON : Bool;
      "RELAY 5" : Bool;
      "RELAY 6" : Bool;
      "RELAY 7" : Bool;
      "RELAY 8" : Bool;
      "RELAY 9" : Bool;
      AMBER : Bool;
      REDLIGHT : Bool;
      "GREEN LIGHT" : Bool;
   END_VAR
   VAR
      START_BIT : Bool;
      "RESET BIT" : Bool;
      IEC_Timer_0_Instance : TON_TIME;
      "PASS ERROR BIT" : Bool;
      CONTINUE_MODE_NG : Bool;
      LOGO_NG_BIT : Bool;
      IEC_Timer_0_Instance_1 : TOF_TIME;
      "ELECTRICAL TEST _ABRT" : TOF_TIME;
   END_VAR
   VAR_TEMP
      HOME : Bool;
      SAFETY : Bool;
      PART2_BUZZ : Bool;
      PART1_BUZZ : Bool;
      PART3_BUZZ : Bool;
      REJ_BUZZ : Bool;
      GN_ILLU1 : Bool;
      GN_ILLU2 : Bool;
      LOGO_LCK_BUZZ : Bool;
   END_VAR
   VAR_TEMP   // added for the SCL form of the ladder/FBD networks
      _w1 : Bool;
      _w2 : Bool;
      _w3 : Bool;
      _w4 : Bool;
      _w5 : Bool;
      _w6 : Bool;
      _w7 : Bool;
      _w8 : Bool;
      _w9 : Bool;
   END_VAR
BEGIN

REGION Network 1: HOME
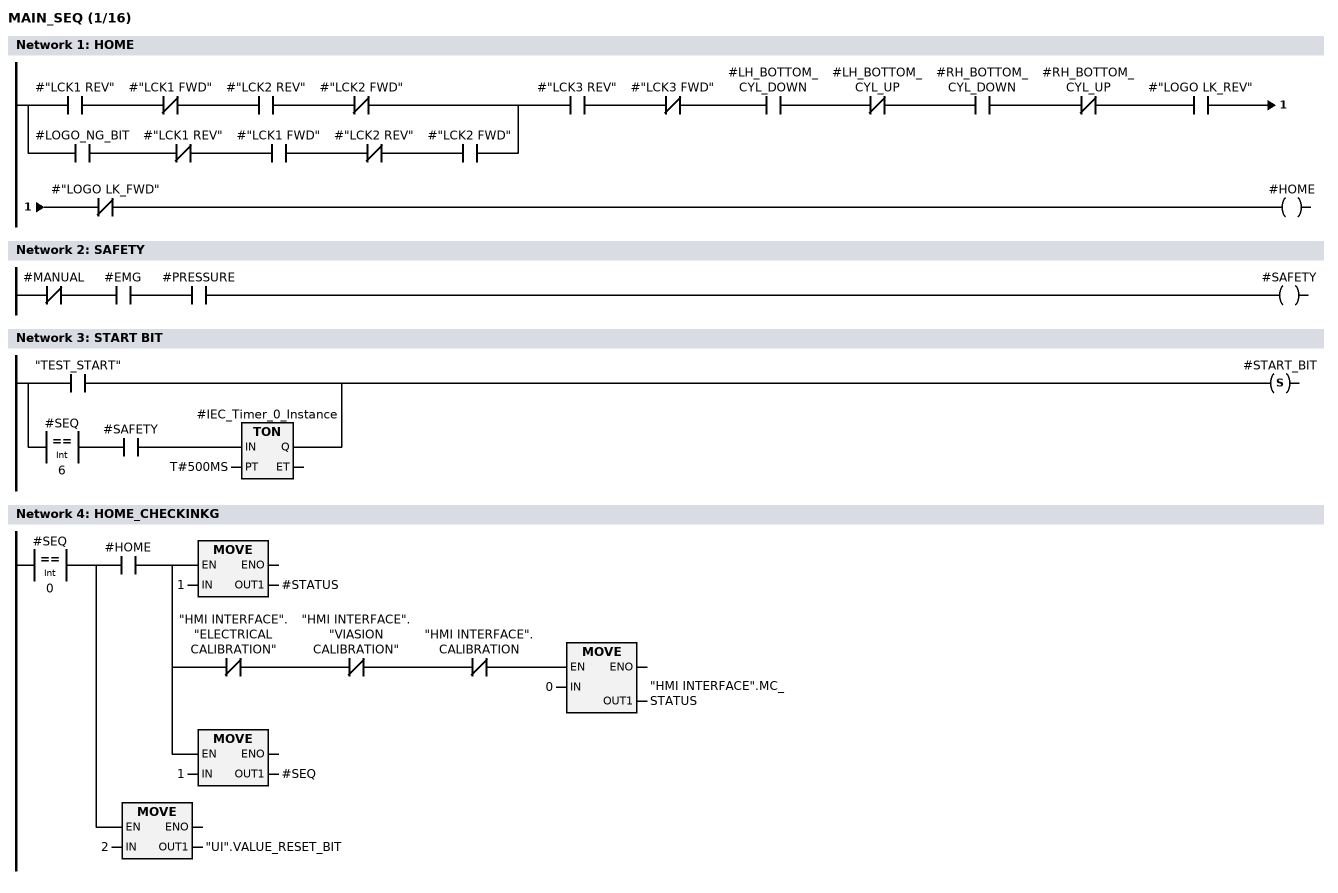
   RUNG wire#powerrail
      Contact( #"LCK1 REV" )
      I_Contact( #"LCK1 FWD" )
      Contact( #"LCK2 REV" )
      I_Contact( #"LCK2 FWD" )
      wire#w1
      Contact( #"LCK3 REV" )
      I_Contact( #"LCK3 FWD" )
      Contact( #LH_BOTTOM_CYL_DOWN )
      I_Contact( #LH_BOTTOM_CYL_UP )
      Contact( #RH_BOTTOM_CYL_DOWN )
      I_Contact( #RH_BOTTOM_CYL_UP )
      Contact( #"LOGO LK_REV" )
      I_Contact( #"LOGO LK_FWD" )
      Coil( #HOME )
   END_RUNG
   RUNG wire#powerrail
      Contact( #LOGO_NG_BIT )
      I_Contact( #"LCK1 REV" )
      Contact( #"LCK1 FWD" )
      I_Contact( #"LCK2 REV" )
      Contact( #"LCK2 FWD" )
   END_RUNG wire#w1
   // the same network as SCL:
   #HOME := ((#"LCK1 REV" AND NOT #"LCK1 FWD" AND #"LCK2 REV" AND NOT #"LCK2 FWD") OR (#LOGO_NG_BIT AND NOT #"LCK1 REV" AND #"LCK1 FWD" AND NOT #"LCK2 REV" AND #"LCK2 FWD")) AND #"LCK3 REV" AND NOT #"LCK3 FWD" AND #LH_BOTTOM_CYL_DOWN AND NOT #LH_BOTTOM_CYL_UP AND #RH_BOTTOM_CYL_DOWN AND NOT #RH_BOTTOM_CYL_UP AND #"LOGO LK_REV" AND NOT #"LOGO LK_FWD";
END_REGION

REGION Network 2: SAFETY
   RUNG wire#powerrail
      I_Contact( #MANUAL )
      Contact( #EMG )
      Contact( #PRESSURE )
      Coil( #SAFETY )
   END_RUNG
   // the same network as SCL:
   #SAFETY := NOT #MANUAL AND #EMG AND #PRESSURE;
END_REGION

REGION Network 3: START BIT
   #IEC_Timer_0_Instance(IN := (#SEQ = 6) AND #SAFETY, PT := T#500MS);   // TON
   IF "TEST_START" OR #IEC_Timer_0_Instance.Q THEN #START_BIT := TRUE; END_IF;
END_REGION

REGION Network 4: HOME_CHECKINKG
   RUNG wire#powerrail
      { S7_Templates := "SrcType := Int" } EQ_Contact(in1 := #SEQ, in2 := 0)
      wire#w1
      Contact( #HOME )
      wire#w2
      Move(in := 1, out1 => #STATUS)
   END_RUNG
   RUNG wire#w2
      I_Contact( "HMI INTERFACE"."ELECTRICAL CALIBRATION" )
      I_Contact( "HMI INTERFACE"."VIASION CALIBRATION" )
      I_Contact( "HMI INTERFACE".CALIBRATION )
      Move(in := 0, out1 => "HMI INTERFACE".MC_STATUS)
   END_RUNG
   RUNG wire#w2
      Move(in := 1, out1 => #SEQ)
   END_RUNG
   RUNG wire#w1
      Move(in := 2, out1 => "UI".VALUE_RESET_BIT)
   END_RUNG
   // the same network as SCL:
   #_w1 := #SEQ = 0;
   #_w2 := #_w1 AND #HOME;
   IF #_w2 THEN #STATUS := 1; END_IF;
   IF #_w2 AND NOT "HMI INTERFACE"."ELECTRICAL CALIBRATION" AND NOT "HMI INTERFACE"."VIASION CALIBRATION" AND NOT "HMI INTERFACE".CALIBRATION THEN
       "HMI INTERFACE".MC_STATUS := 0;
   END_IF;
   IF #_w2 THEN #SEQ := 1; END_IF;
   IF #_w1 THEN "UI".VALUE_RESET_BIT := 2; END_IF;
END_REGION

REGION Network 5: PART1_CHECKING
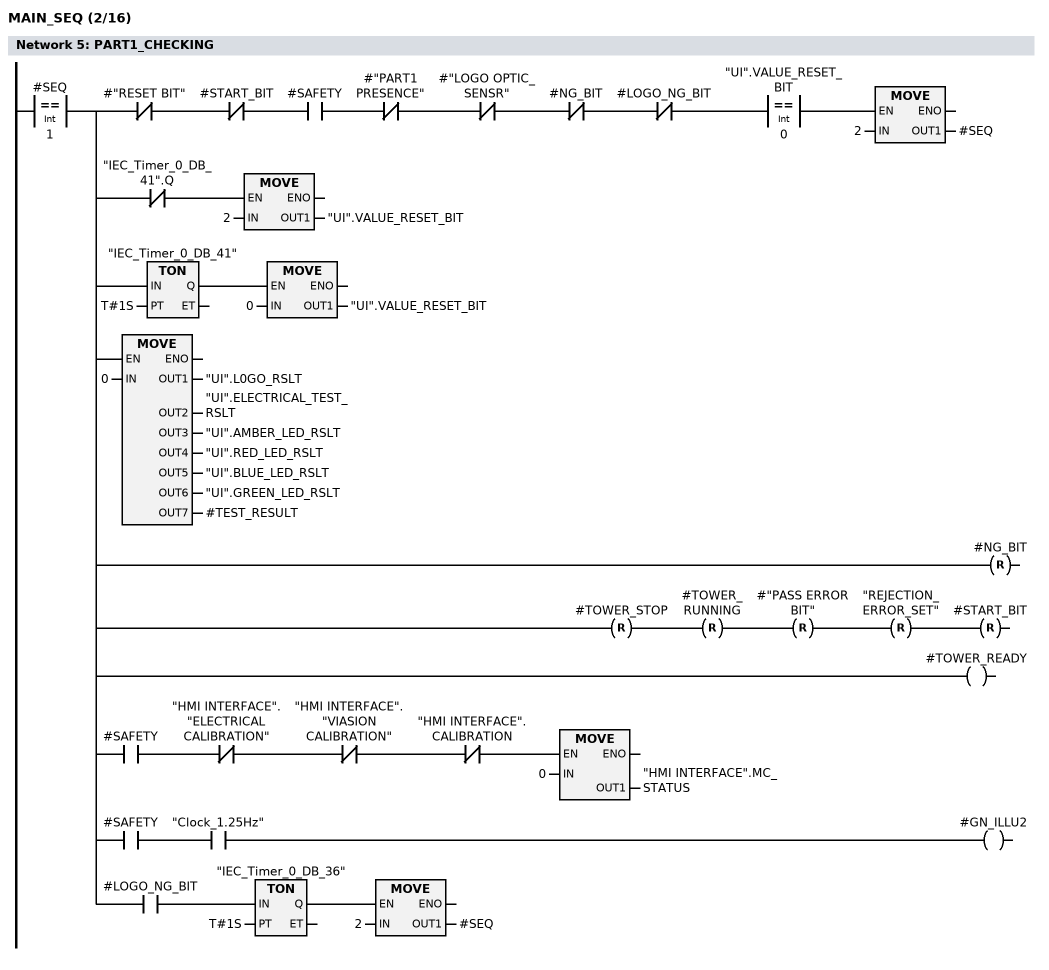
   #_w1 := #SEQ = 1;
   IF #_w1 AND NOT #"RESET BIT" AND NOT #START_BIT AND #SAFETY AND NOT #"PART1 PRESENCE" AND NOT #"LOGO OPTIC_SENSR" AND NOT #NG_BIT AND NOT #LOGO_NG_BIT AND ("UI".VALUE_RESET_BIT = 0) THEN
       #SEQ := 2;
   END_IF;
   IF #_w1 AND NOT "IEC_Timer_0_DB_41".Q THEN "UI".VALUE_RESET_BIT := 2; END_IF;
   "IEC_Timer_0_DB_41".TON(IN := #_w1, PT := T#1S);
   IF "IEC_Timer_0_DB_41".Q THEN "UI".VALUE_RESET_BIT := 0; END_IF;
   IF #_w1 THEN
       "UI".L0GO_RSLT := 0;
       "UI".ELECTRICAL_TEST_RSLT := 0;
       "UI".AMBER_LED_RSLT := 0;
       "UI".RED_LED_RSLT := 0;
       "UI".BLUE_LED_RSLT := 0;
       "UI".GREEN_LED_RSLT := 0;
       #TEST_RESULT := 0;
       #NG_BIT := FALSE;
       #TOWER_STOP := FALSE;
       #TOWER_RUNNING := FALSE;
       #"PASS ERROR BIT" := FALSE;
       "REJECTION_ERROR_SET" := FALSE;
       #START_BIT := FALSE;
   END_IF;
   #TOWER_READY := #_w1;
   IF #_w1 AND #SAFETY AND NOT "HMI INTERFACE"."ELECTRICAL CALIBRATION" AND NOT "HMI INTERFACE"."VIASION CALIBRATION" AND NOT "HMI INTERFACE".CALIBRATION THEN
       "HMI INTERFACE".MC_STATUS := 0;
   END_IF;
   #GN_ILLU2 := #_w1 AND #SAFETY AND "Clock_1.25Hz";
   "IEC_Timer_0_DB_36".TON(IN := #_w1 AND #LOGO_NG_BIT, PT := T#1S);
   IF "IEC_Timer_0_DB_36".Q THEN #SEQ := 2; END_IF;
END_REGION

REGION Network 6: PART1_LOCKING
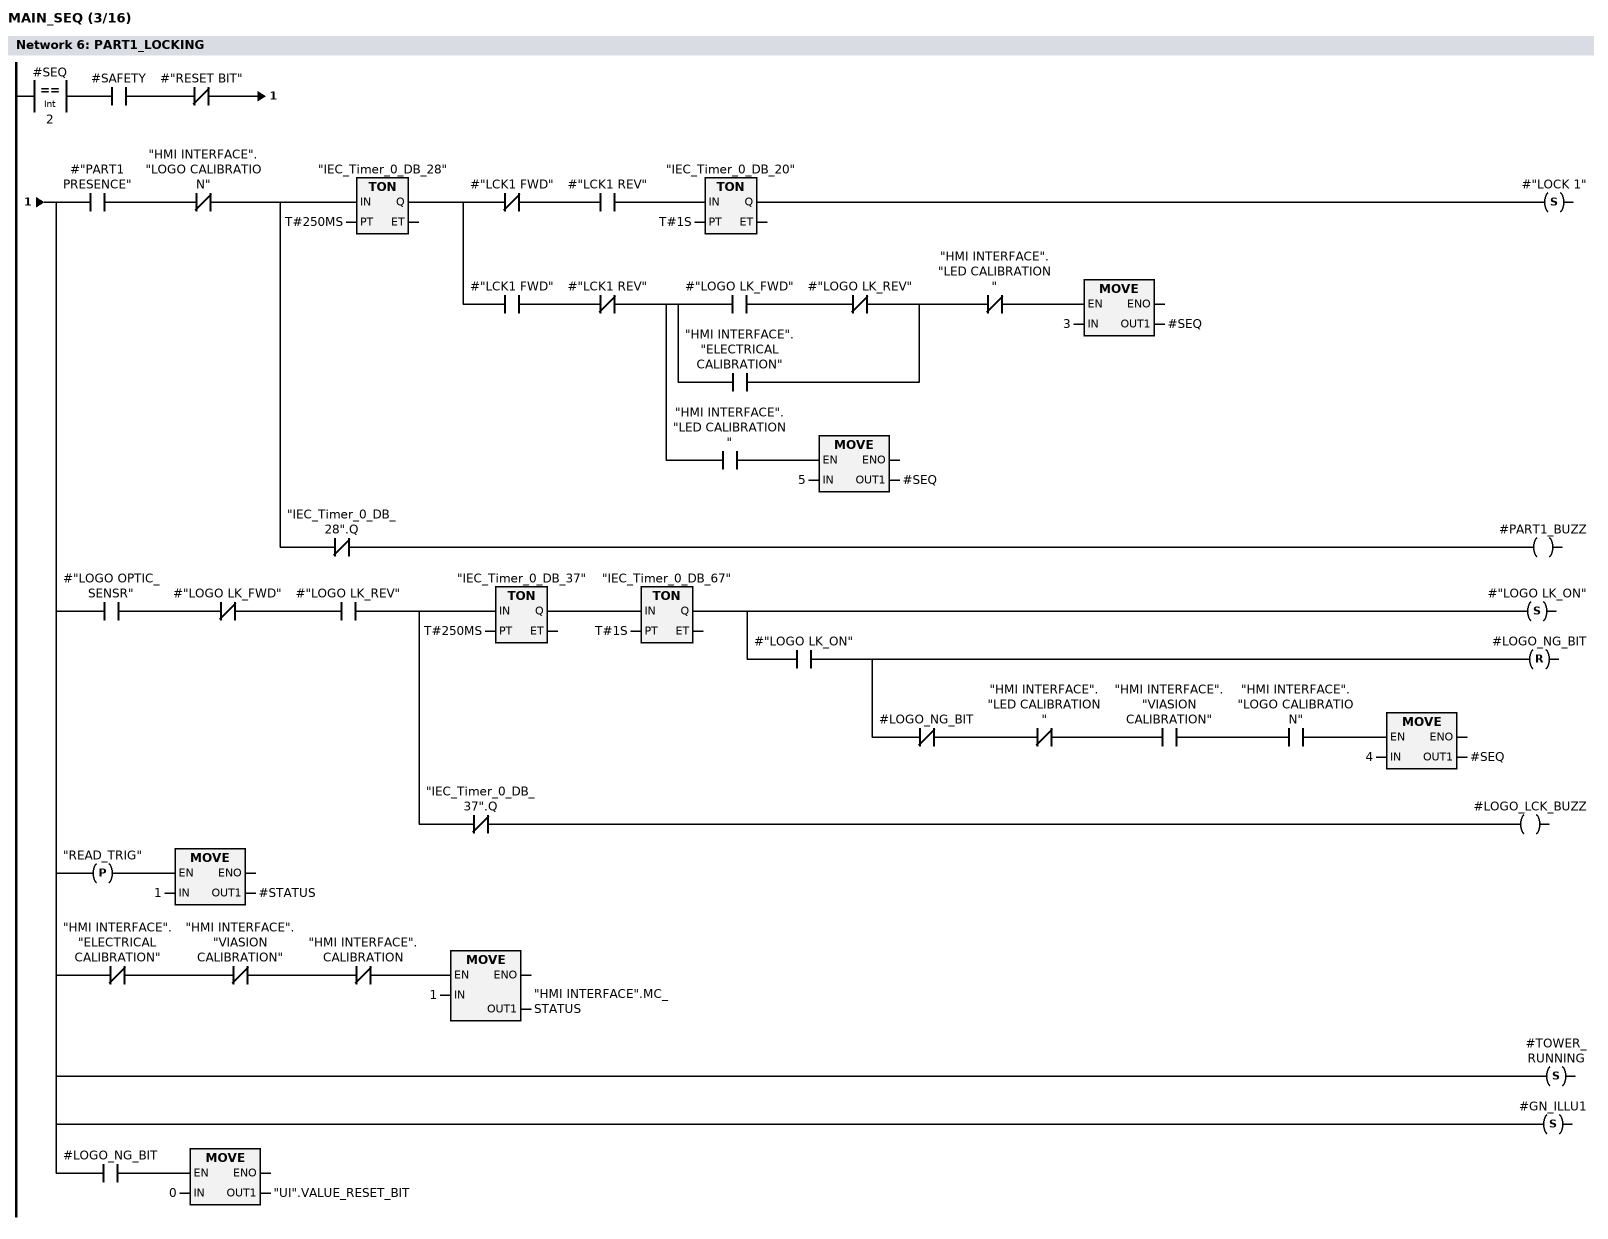
   #_w1 := (#SEQ = 2) AND #SAFETY AND NOT #"RESET BIT";
   #_w2 := #_w1 AND #"PART1 PRESENCE" AND NOT "HMI INTERFACE"."LOGO CALIBRATION";
   "IEC_Timer_0_DB_28".TON(IN := #_w2, PT := T#250MS);
   "IEC_Timer_0_DB_20".TON(IN := "IEC_Timer_0_DB_28".Q AND NOT #"LCK1 FWD" AND #"LCK1 REV", PT := T#1S);
   IF "IEC_Timer_0_DB_20".Q THEN #"LOCK 1" := TRUE; END_IF;
   #_w3 := "IEC_Timer_0_DB_28".Q AND #"LCK1 FWD" AND NOT #"LCK1 REV";
   IF #_w3 AND ((#"LOGO LK_FWD" AND NOT #"LOGO LK_REV") OR "HMI INTERFACE"."ELECTRICAL CALIBRATION") AND NOT "HMI INTERFACE"."LED CALIBRATION" THEN
       #SEQ := 3;
   END_IF;
   IF #_w3 AND "HMI INTERFACE"."LED CALIBRATION" THEN #SEQ := 5; END_IF;
   #PART1_BUZZ := #_w2 AND NOT "IEC_Timer_0_DB_28".Q;
   #_w4 := #_w1 AND #"LOGO OPTIC_SENSR" AND NOT #"LOGO LK_FWD" AND #"LOGO LK_REV";
   "IEC_Timer_0_DB_37".TON(IN := #_w4, PT := T#250MS);
   "IEC_Timer_0_DB_67".TON(IN := "IEC_Timer_0_DB_37".Q, PT := T#1S);
   IF "IEC_Timer_0_DB_67".Q THEN #"LOGO LK_ON" := TRUE; END_IF;
   #_w5 := "IEC_Timer_0_DB_67".Q AND #"LOGO LK_ON";
   IF #_w5 THEN #LOGO_NG_BIT := FALSE; END_IF;
   IF #_w5 AND NOT #LOGO_NG_BIT AND NOT "HMI INTERFACE"."LED CALIBRATION" AND "HMI INTERFACE"."VIASION CALIBRATION" AND "HMI INTERFACE"."LOGO CALIBRATION" THEN
       #SEQ := 4;
   END_IF;
   #LOGO_LCK_BUZZ := #_w4 AND NOT "IEC_Timer_0_DB_37".Q;
   #_w6 := #_w1 AND NOT "READ_TRIG";   // rising edge
   "READ_TRIG" := #_w1;
   IF #_w6 THEN #STATUS := 1; END_IF;
   IF #_w1 AND NOT "HMI INTERFACE"."ELECTRICAL CALIBRATION" AND NOT "HMI INTERFACE"."VIASION CALIBRATION" AND NOT "HMI INTERFACE".CALIBRATION THEN
       "HMI INTERFACE".MC_STATUS := 1;
   END_IF;
   IF #_w1 THEN
       #TOWER_RUNNING := TRUE;
       #GN_ILLU1 := TRUE;
   END_IF;
   IF #_w1 AND #LOGO_NG_BIT THEN "UI".VALUE_RESET_BIT := 0; END_IF;
END_REGION

REGION Network 7: PART2 CHECKING & LOCKING
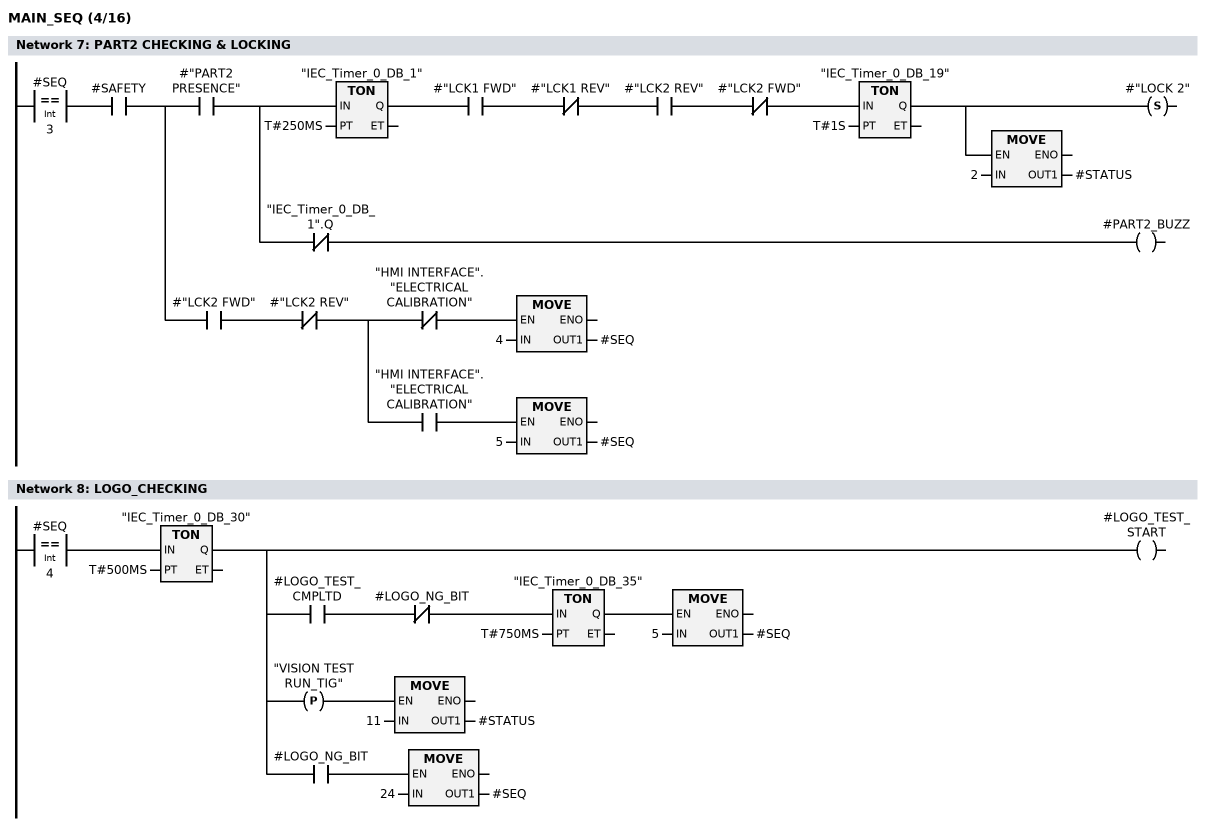
   #_w1 := (#SEQ = 3) AND #SAFETY;
   #_w2 := #_w1 AND #"PART2 PRESENCE";
   "IEC_Timer_0_DB_1".TON(IN := #_w2, PT := T#250MS);
   "IEC_Timer_0_DB_19".TON(IN := "IEC_Timer_0_DB_1".Q AND #"LCK1 FWD" AND NOT #"LCK1 REV" AND #"LCK2 REV" AND NOT #"LCK2 FWD",
                           PT := T#1S);
   IF "IEC_Timer_0_DB_19".Q THEN
       #"LOCK 2" := TRUE;
       #STATUS := 2;
   END_IF;
   #PART2_BUZZ := #_w2 AND NOT "IEC_Timer_0_DB_1".Q;
   #_w3 := #_w1 AND #"LCK2 FWD" AND NOT #"LCK2 REV";
   IF #_w3 AND NOT "HMI INTERFACE"."ELECTRICAL CALIBRATION" THEN #SEQ := 4; END_IF;
   IF #_w3 AND "HMI INTERFACE"."ELECTRICAL CALIBRATION" THEN #SEQ := 5; END_IF;
END_REGION

REGION Network 8: LOGO_CHECKING
   "IEC_Timer_0_DB_30".TON(IN := #SEQ = 4, PT := T#500MS);
   #LOGO_TEST_START := "IEC_Timer_0_DB_30".Q;
   "IEC_Timer_0_DB_35".TON(IN := "IEC_Timer_0_DB_30".Q AND #LOGO_TEST_CMPLTD AND NOT #LOGO_NG_BIT,
                           PT := T#750MS);
   IF "IEC_Timer_0_DB_35".Q THEN #SEQ := 5; END_IF;
   #_w1 := "IEC_Timer_0_DB_30".Q AND NOT "VISION TEST RUN_TIG";   // rising edge
   "VISION TEST RUN_TIG" := "IEC_Timer_0_DB_30".Q;
   IF #_w1 THEN #STATUS := 11; END_IF;
   IF "IEC_Timer_0_DB_30".Q AND #LOGO_NG_BIT THEN #SEQ := 24; END_IF;
END_REGION

REGION Network 9: BOTTOM CYLINDERS UP
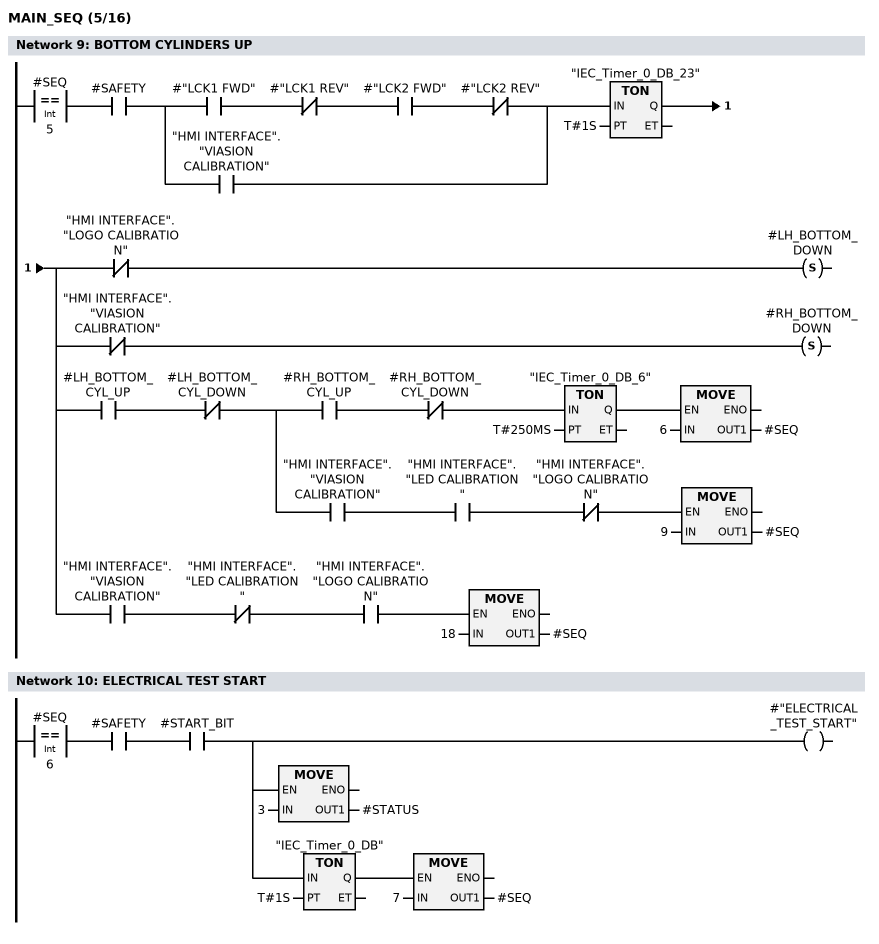
   "IEC_Timer_0_DB_23".TON(IN := (#SEQ = 5) AND #SAFETY AND ((#"LCK1 FWD" AND NOT #"LCK1 REV" AND #"LCK2 FWD" AND NOT #"LCK2 REV") OR "HMI INTERFACE"."VIASION CALIBRATION"),
                           PT := T#1S);
   IF "IEC_Timer_0_DB_23".Q AND NOT "HMI INTERFACE"."LOGO CALIBRATION" THEN #LH_BOTTOM_DOWN := TRUE; END_IF;
   IF "IEC_Timer_0_DB_23".Q AND NOT "HMI INTERFACE"."VIASION CALIBRATION" THEN
       #RH_BOTTOM_DOWN := TRUE;
   END_IF;
   #_w1 := "IEC_Timer_0_DB_23".Q AND #LH_BOTTOM_CYL_UP AND NOT #LH_BOTTOM_CYL_DOWN;
   "IEC_Timer_0_DB_6".TON(IN := #_w1 AND #RH_BOTTOM_CYL_UP AND NOT #RH_BOTTOM_CYL_DOWN, PT := T#250MS);
   IF "IEC_Timer_0_DB_6".Q THEN #SEQ := 6; END_IF;
   IF #_w1 AND "HMI INTERFACE"."VIASION CALIBRATION" AND "HMI INTERFACE"."LED CALIBRATION" AND NOT "HMI INTERFACE"."LOGO CALIBRATION" THEN
       #SEQ := 9;
   END_IF;
   IF "IEC_Timer_0_DB_23".Q AND "HMI INTERFACE"."VIASION CALIBRATION" AND NOT "HMI INTERFACE"."LED CALIBRATION" AND "HMI INTERFACE"."LOGO CALIBRATION" THEN
       #SEQ := 18;
   END_IF;
END_REGION

REGION Network 10: ELECTRICAL TEST START
   #"ELECTRICAL _TEST_START" := (#SEQ = 6) AND #SAFETY AND #START_BIT;
   IF #"ELECTRICAL _TEST_START" THEN #STATUS := 3; END_IF;
   "IEC_Timer_0_DB".TON(IN := #"ELECTRICAL _TEST_START", PT := T#1S);
   IF "IEC_Timer_0_DB".Q THEN #SEQ := 7; END_IF;
END_REGION

REGION Network 11: LOCK 2 RELEASING
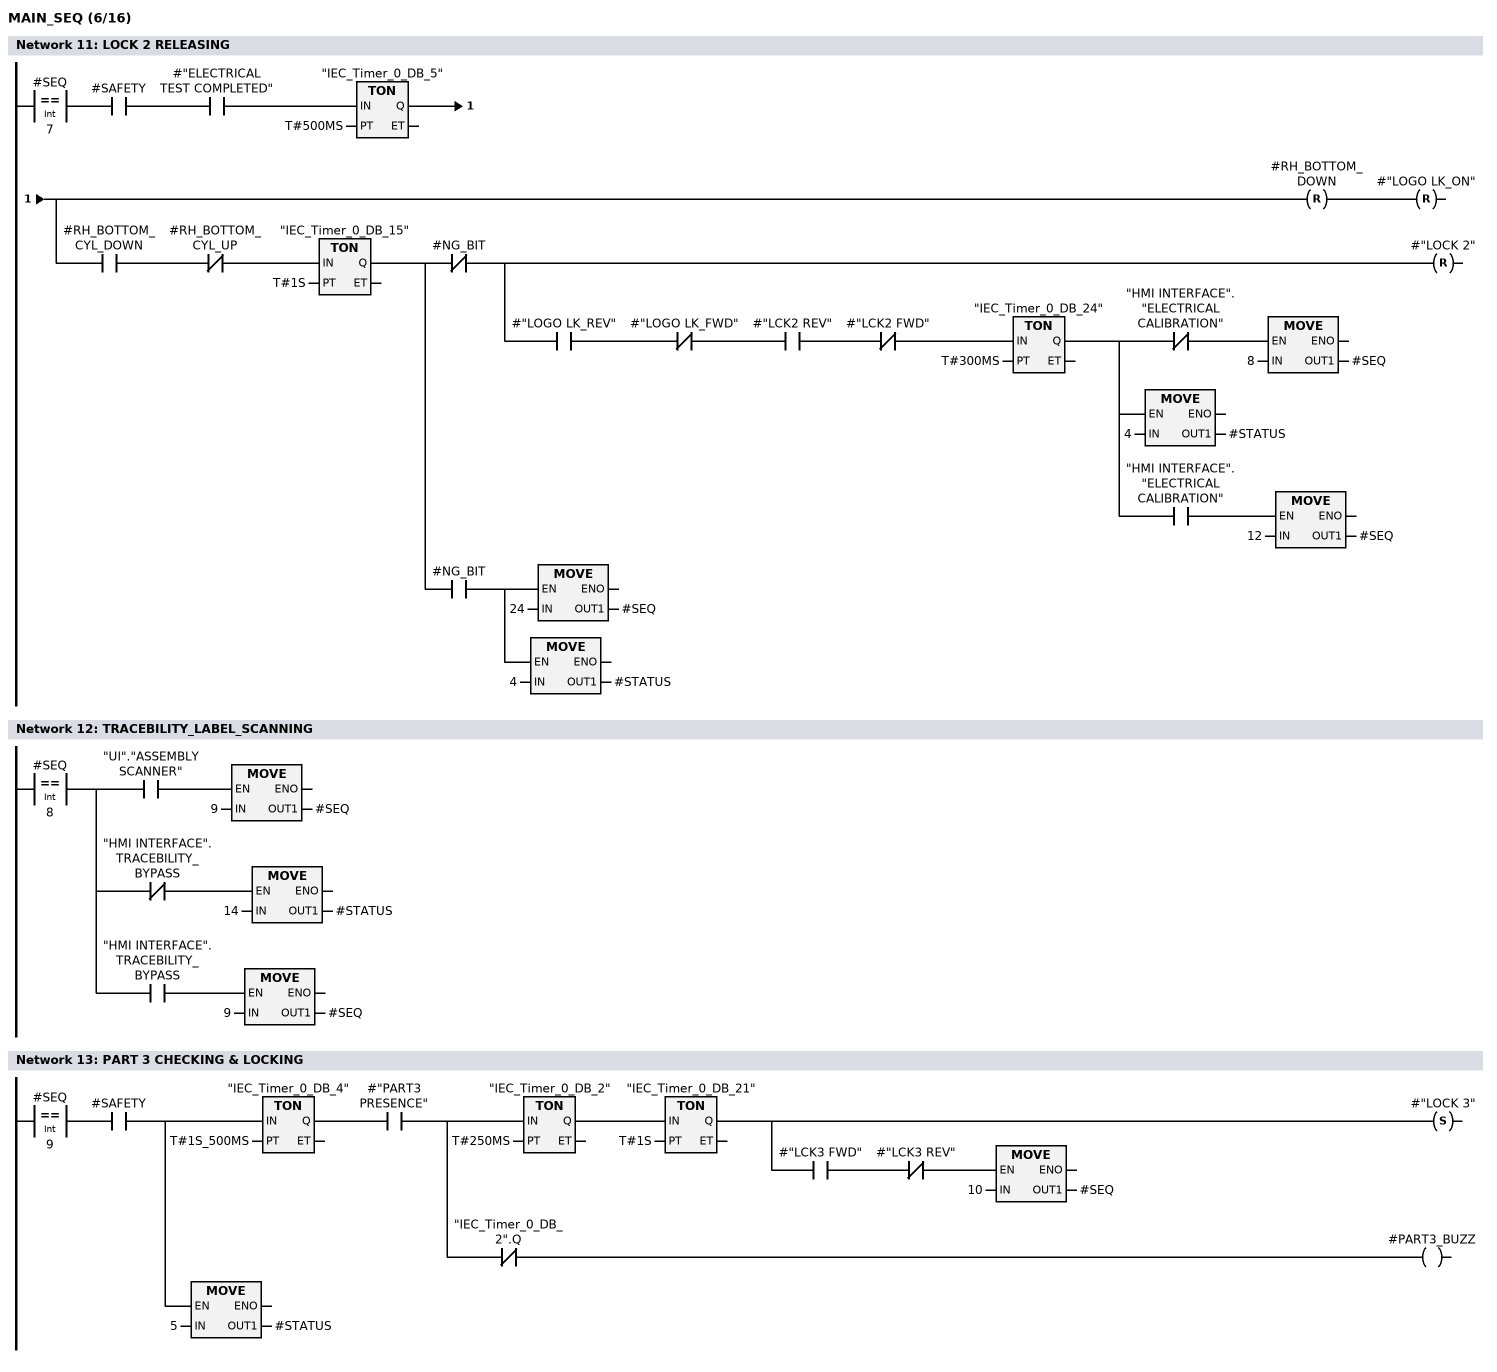
   "IEC_Timer_0_DB_5".TON(IN := (#SEQ = 7) AND #SAFETY AND #"ELECTRICAL TEST COMPLETED", PT := T#500MS);
   IF "IEC_Timer_0_DB_5".Q THEN
       #RH_BOTTOM_DOWN := FALSE;
       #"LOGO LK_ON" := FALSE;
   END_IF;
   "IEC_Timer_0_DB_15".TON(IN := "IEC_Timer_0_DB_5".Q AND #RH_BOTTOM_CYL_DOWN AND NOT #RH_BOTTOM_CYL_UP,
                           PT := T#1S);
   #_w1 := "IEC_Timer_0_DB_15".Q AND NOT #NG_BIT;
   IF #_w1 THEN #"LOCK 2" := FALSE; END_IF;
   "IEC_Timer_0_DB_24".TON(IN := #_w1 AND #"LOGO LK_REV" AND NOT #"LOGO LK_FWD" AND #"LCK2 REV" AND NOT #"LCK2 FWD",
                           PT := T#300MS);
   IF "IEC_Timer_0_DB_24".Q AND NOT "HMI INTERFACE"."ELECTRICAL CALIBRATION" THEN #SEQ := 8; END_IF;
   IF "IEC_Timer_0_DB_24".Q THEN #STATUS := 4; END_IF;
   IF "IEC_Timer_0_DB_24".Q AND "HMI INTERFACE"."ELECTRICAL CALIBRATION" THEN #SEQ := 12; END_IF;
   IF "IEC_Timer_0_DB_15".Q AND #NG_BIT THEN
       #SEQ := 24;
       #STATUS := 4;
   END_IF;
END_REGION

REGION Network 12: TRACEBILITY_LABEL_SCANNING
   RUNG wire#powerrail
      { S7_Templates := "SrcType := Int" } EQ_Contact(in1 := #SEQ, in2 := 8)
      wire#w1
      Contact( "UI"."ASSEMBLY SCANNER" )
      Move(in := 9, out1 => #SEQ)
   END_RUNG
   RUNG wire#w1
      I_Contact( "HMI INTERFACE".TRACEBILITY_BYPASS )
      Move(in := 14, out1 => #STATUS)
   END_RUNG
   RUNG wire#w1
      Contact( "HMI INTERFACE".TRACEBILITY_BYPASS )
      Move(in := 9, out1 => #SEQ)
   END_RUNG
   // the same network as SCL:
   #_w1 := #SEQ = 8;
   IF #_w1 AND "UI"."ASSEMBLY SCANNER" THEN #SEQ := 9; END_IF;
   IF #_w1 AND NOT "HMI INTERFACE".TRACEBILITY_BYPASS THEN #STATUS := 14; END_IF;
   IF #_w1 AND "HMI INTERFACE".TRACEBILITY_BYPASS THEN #SEQ := 9; END_IF;
END_REGION

REGION Network 13: PART 3 CHECKING & LOCKING
   #_w1 := (#SEQ = 9) AND #SAFETY;
   "IEC_Timer_0_DB_4".TON(IN := #_w1, PT := T#1S_500MS);
   #_w2 := "IEC_Timer_0_DB_4".Q AND #"PART3 PRESENCE";
   "IEC_Timer_0_DB_2".TON(IN := #_w2, PT := T#250MS);
   "IEC_Timer_0_DB_21".TON(IN := "IEC_Timer_0_DB_2".Q, PT := T#1S);
   IF "IEC_Timer_0_DB_21".Q THEN #"LOCK 3" := TRUE; END_IF;
   IF "IEC_Timer_0_DB_21".Q AND #"LCK3 FWD" AND NOT #"LCK3 REV" THEN #SEQ := 10; END_IF;
   #PART3_BUZZ := #_w2 AND NOT "IEC_Timer_0_DB_2".Q;
   IF #_w1 THEN #STATUS := 5; END_IF;
END_REGION

REGION Network 14: VISION TEST START
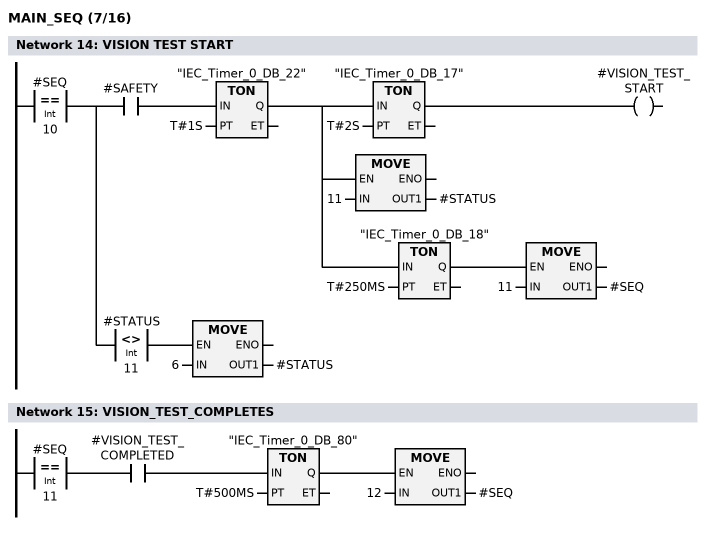
   #_w1 := #SEQ = 10;
   "IEC_Timer_0_DB_22".TON(IN := #_w1 AND #SAFETY, PT := T#1S);
   "IEC_Timer_0_DB_17".TON(IN := "IEC_Timer_0_DB_22".Q, PT := T#2S);
   #VISION_TEST_START := "IEC_Timer_0_DB_17".Q;
   IF "IEC_Timer_0_DB_22".Q THEN #STATUS := 11; END_IF;
   "IEC_Timer_0_DB_18".TON(IN := "IEC_Timer_0_DB_22".Q, PT := T#250MS);
   IF "IEC_Timer_0_DB_18".Q THEN #SEQ := 11; END_IF;
   IF #_w1 AND (#STATUS <> 11) THEN #STATUS := 6; END_IF;
END_REGION

REGION Network 15: VISION_TEST_COMPLETES
   "IEC_Timer_0_DB_80".TON(IN := (#SEQ = 11) AND #VISION_TEST_COMPLETED, PT := T#500MS);
   IF "IEC_Timer_0_DB_80".Q THEN #SEQ := 12; END_IF;
END_REGION

REGION Network 16: LOCK 1 RELEASE
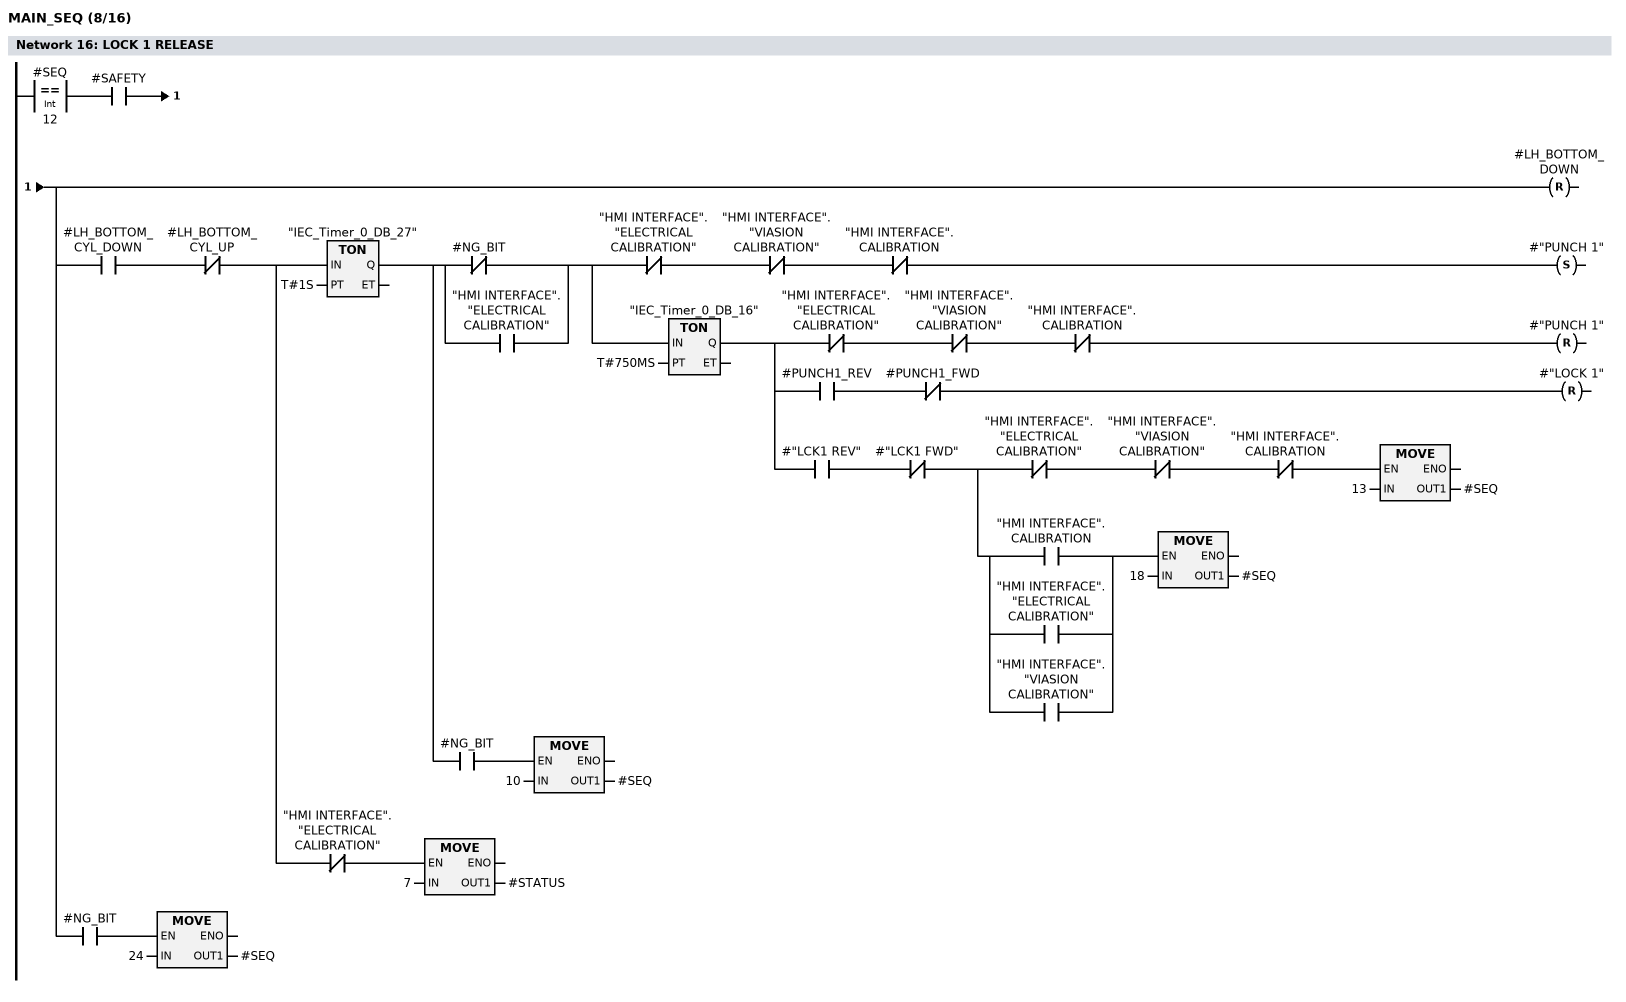
   #_w1 := (#SEQ = 12) AND #SAFETY;
   IF #_w1 THEN #LH_BOTTOM_DOWN := FALSE; END_IF;
   #_w2 := #_w1 AND #LH_BOTTOM_CYL_DOWN AND NOT #LH_BOTTOM_CYL_UP;
   "IEC_Timer_0_DB_27".TON(IN := #_w2, PT := T#1S);
   #_w3 := "IEC_Timer_0_DB_27".Q AND (NOT #NG_BIT OR "HMI INTERFACE"."ELECTRICAL CALIBRATION");
   IF #_w3 AND NOT "HMI INTERFACE"."ELECTRICAL CALIBRATION" AND NOT "HMI INTERFACE"."VIASION CALIBRATION" AND NOT "HMI INTERFACE".CALIBRATION THEN
       #"PUNCH 1" := TRUE;
   END_IF;
   "IEC_Timer_0_DB_16".TON(IN := #_w3, PT := T#750MS);
   IF "IEC_Timer_0_DB_16".Q AND NOT "HMI INTERFACE"."ELECTRICAL CALIBRATION" AND NOT "HMI INTERFACE"."VIASION CALIBRATION" AND NOT "HMI INTERFACE".CALIBRATION THEN
       #"PUNCH 1" := FALSE;
   END_IF;
   IF "IEC_Timer_0_DB_16".Q AND #PUNCH1_REV AND NOT #PUNCH1_FWD THEN #"LOCK 1" := FALSE; END_IF;
   #_w4 := "IEC_Timer_0_DB_16".Q AND #"LCK1 REV" AND NOT #"LCK1 FWD";
   IF #_w4 AND NOT "HMI INTERFACE"."ELECTRICAL CALIBRATION" AND NOT "HMI INTERFACE"."VIASION CALIBRATION" AND NOT "HMI INTERFACE".CALIBRATION THEN
       #SEQ := 13;
   END_IF;
   IF #_w4 AND ("HMI INTERFACE".CALIBRATION OR "HMI INTERFACE"."ELECTRICAL CALIBRATION" OR "HMI INTERFACE"."VIASION CALIBRATION") THEN
       #SEQ := 18;
   END_IF;
   IF "IEC_Timer_0_DB_27".Q AND #NG_BIT THEN #SEQ := 10; END_IF;
   IF #_w2 AND NOT "HMI INTERFACE"."ELECTRICAL CALIBRATION" THEN #STATUS := 7; END_IF;
   IF #_w1 AND #NG_BIT THEN #SEQ := 24; END_IF;
END_REGION

REGION Network 17: TEST_STATUS
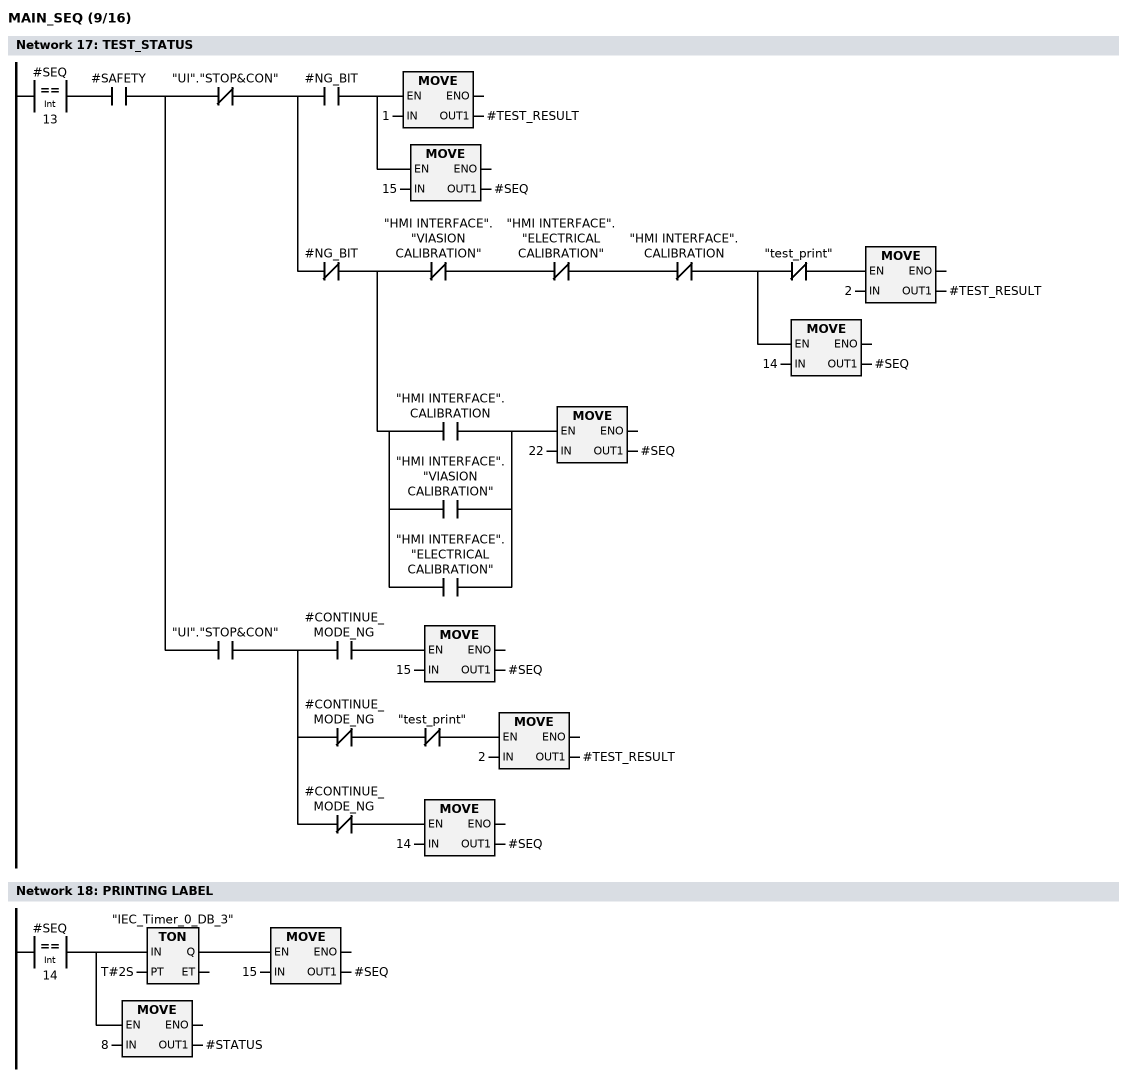
   RUNG wire#powerrail
      { S7_Templates := "SrcType := Int" } EQ_Contact(in1 := #SEQ, in2 := 13)
      Contact( #SAFETY )
      wire#w1
      I_Contact( "UI"."STOP&CON" )
      wire#w2
      Contact( #NG_BIT )
      wire#w3
      Move(in := 1, out1 => #TEST_RESULT)
   END_RUNG
   RUNG wire#w3
      Move(in := 15, out1 => #SEQ)
   END_RUNG
   RUNG wire#w2
      I_Contact( #NG_BIT )
      wire#w4
      I_Contact( "HMI INTERFACE"."VIASION CALIBRATION" )
      I_Contact( "HMI INTERFACE"."ELECTRICAL CALIBRATION" )
      I_Contact( "HMI INTERFACE".CALIBRATION )
      wire#w5
      I_Contact( "test_print" )
      Move(in := 2, out1 => #TEST_RESULT)
   END_RUNG
   RUNG wire#w5
      Move(in := 14, out1 => #SEQ)
   END_RUNG
   RUNG wire#w4
      Contact( "HMI INTERFACE".CALIBRATION )
      wire#w6
      Move(in := 22, out1 => #SEQ)
   END_RUNG
   RUNG wire#w4
      Contact( "HMI INTERFACE"."VIASION CALIBRATION" )
   END_RUNG wire#w6
   RUNG wire#w4
      Contact( "HMI INTERFACE"."ELECTRICAL CALIBRATION" )
   END_RUNG wire#w6
   RUNG wire#w1
      Contact( "UI"."STOP&CON" )
      wire#w7
      Contact( #CONTINUE_MODE_NG )
      Move(in := 15, out1 => #SEQ)
   END_RUNG
   RUNG wire#w7
      I_Contact( #CONTINUE_MODE_NG )
      I_Contact( "test_print" )
      Move(in := 2, out1 => #TEST_RESULT)
   END_RUNG
   RUNG wire#w7
      I_Contact( #CONTINUE_MODE_NG )
      Move(in := 14, out1 => #SEQ)
   END_RUNG
   // the same network as SCL:
   #_w1 := (#SEQ = 13) AND #SAFETY;
   #_w2 := #_w1 AND NOT "UI"."STOP&CON";
   IF #_w2 AND #NG_BIT THEN
       #TEST_RESULT := 1;
       #SEQ := 15;
   END_IF;
   #_w3 := #_w2 AND NOT #NG_BIT;
   #_w4 := #_w3 AND NOT "HMI INTERFACE"."VIASION CALIBRATION" AND NOT "HMI INTERFACE"."ELECTRICAL CALIBRATION" AND NOT "HMI INTERFACE".CALIBRATION;
   IF #_w4 AND NOT "test_print" THEN #TEST_RESULT := 2; END_IF;
   IF #_w4 THEN #SEQ := 14; END_IF;
   IF #_w3 AND ("HMI INTERFACE".CALIBRATION OR "HMI INTERFACE"."VIASION CALIBRATION" OR "HMI INTERFACE"."ELECTRICAL CALIBRATION") THEN
       #SEQ := 22;
   END_IF;
   #_w5 := #_w1 AND "UI"."STOP&CON";
   IF #_w5 AND #CONTINUE_MODE_NG THEN #SEQ := 15; END_IF;
   IF #_w5 AND NOT #CONTINUE_MODE_NG AND NOT "test_print" THEN #TEST_RESULT := 2; END_IF;
   IF #_w5 AND NOT #CONTINUE_MODE_NG THEN #SEQ := 14; END_IF;
END_REGION

REGION Network 18: PRINTING LABEL
   #_w1 := #SEQ = 14;
   "IEC_Timer_0_DB_3".TON(IN := #_w1, PT := T#2S);
   IF "IEC_Timer_0_DB_3".Q THEN #SEQ := 15; END_IF;
   IF #_w1 THEN #STATUS := 8; END_IF;
END_REGION

REGION Network 19: SCANNING
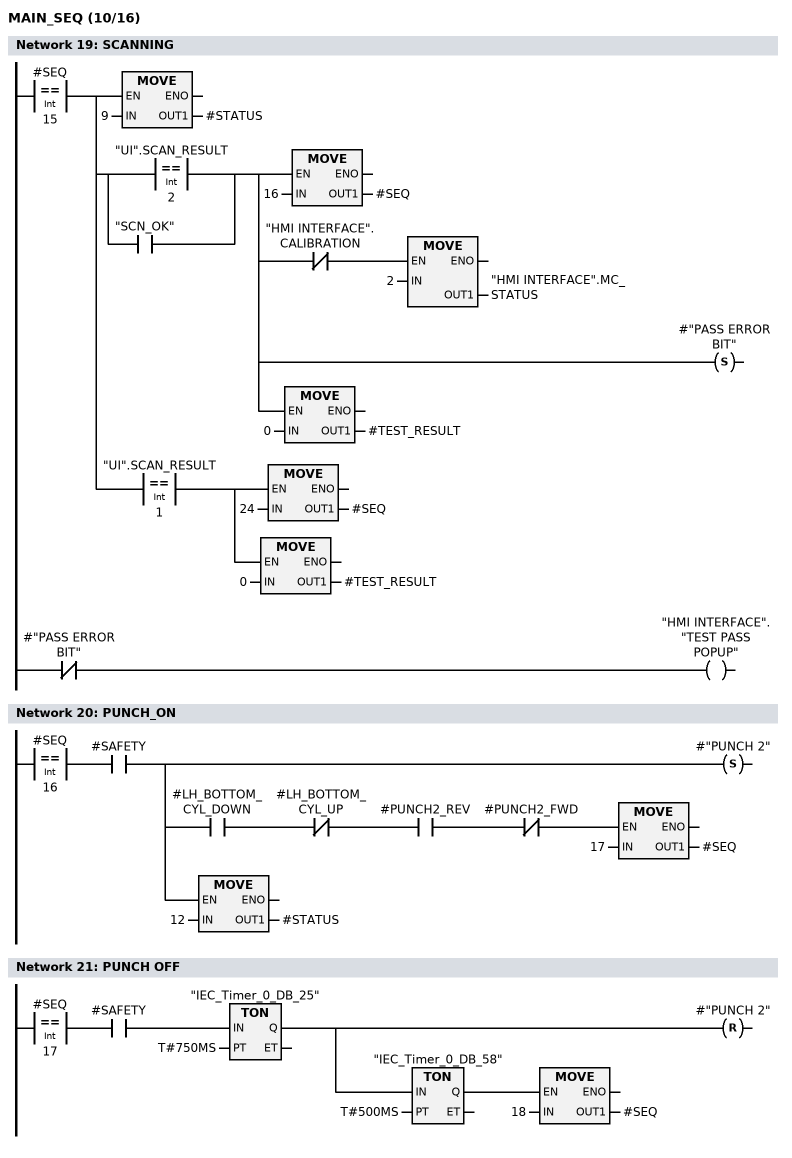
   RUNG wire#powerrail
      { S7_Templates := "SrcType := Int" } EQ_Contact(in1 := #SEQ, in2 := 15)
      wire#w1
      Move(in := 9, out1 => #STATUS)
   END_RUNG
   RUNG wire#w1
      { S7_Templates := "SrcType := Int" } EQ_Contact(in1 := "UI".SCAN_RESULT, in2 := 2)
      wire#w2
      Move(in := 16, out1 => #SEQ)
   END_RUNG
   RUNG wire#w1
      Contact( "SCN_OK" )
   END_RUNG wire#w2
   RUNG wire#w2
      I_Contact( "HMI INTERFACE".CALIBRATION )
      Move(in := 2, out1 => "HMI INTERFACE".MC_STATUS)
   END_RUNG
   RUNG wire#w2
      S_Coil( #"PASS ERROR BIT" )
   END_RUNG
   RUNG wire#w2
      Move(in := 0, out1 => #TEST_RESULT)
   END_RUNG
   RUNG wire#w1
      { S7_Templates := "SrcType := Int" } EQ_Contact(in1 := "UI".SCAN_RESULT, in2 := 1)
      wire#w3
      Move(in := 24, out1 => #SEQ)
   END_RUNG
   RUNG wire#w3
      Move(in := 0, out1 => #TEST_RESULT)
   END_RUNG
   RUNG wire#powerrail
      I_Contact( #"PASS ERROR BIT" )
      Coil( "HMI INTERFACE"."TEST PASS POPUP" )
   END_RUNG
   // the same network as SCL:
   #_w1 := #SEQ = 15;
   IF #_w1 THEN #STATUS := 9; END_IF;
   #_w2 := #_w1 AND (("UI".SCAN_RESULT = 2) OR "SCN_OK");
   IF #_w2 THEN #SEQ := 16; END_IF;
   IF #_w2 AND NOT "HMI INTERFACE".CALIBRATION THEN "HMI INTERFACE".MC_STATUS := 2; END_IF;
   IF #_w2 THEN
       #"PASS ERROR BIT" := TRUE;
       #TEST_RESULT := 0;
   END_IF;
   IF #_w1 AND ("UI".SCAN_RESULT = 1) THEN
       #SEQ := 24;
       #TEST_RESULT := 0;
   END_IF;
   "HMI INTERFACE"."TEST PASS POPUP" := NOT #"PASS ERROR BIT";
END_REGION

REGION Network 20: PUNCH_ON
   RUNG wire#powerrail
      { S7_Templates := "SrcType := Int" } EQ_Contact(in1 := #SEQ, in2 := 16)
      Contact( #SAFETY )
      wire#w1
      S_Coil( #"PUNCH 2" )
   END_RUNG
   RUNG wire#w1
      Contact( #LH_BOTTOM_CYL_DOWN )
      I_Contact( #LH_BOTTOM_CYL_UP )
      Contact( #PUNCH2_REV )
      I_Contact( #PUNCH2_FWD )
      Move(in := 17, out1 => #SEQ)
   END_RUNG
   RUNG wire#w1
      Move(in := 12, out1 => #STATUS)
   END_RUNG
   // the same network as SCL:
   #_w1 := (#SEQ = 16) AND #SAFETY;
   IF #_w1 THEN #"PUNCH 2" := TRUE; END_IF;
   IF #_w1 AND #LH_BOTTOM_CYL_DOWN AND NOT #LH_BOTTOM_CYL_UP AND #PUNCH2_REV AND NOT #PUNCH2_FWD THEN
       #SEQ := 17;
   END_IF;
   IF #_w1 THEN #STATUS := 12; END_IF;
END_REGION

REGION Network 21: PUNCH OFF
   "IEC_Timer_0_DB_25".TON(IN := (#SEQ = 17) AND #SAFETY, PT := T#750MS);
   IF "IEC_Timer_0_DB_25".Q THEN #"PUNCH 2" := FALSE; END_IF;
   "IEC_Timer_0_DB_58".TON(IN := "IEC_Timer_0_DB_25".Q, PT := T#500MS);
   IF "IEC_Timer_0_DB_58".Q THEN #SEQ := 18; END_IF;
END_REGION

REGION Network 22: LOCK 3 RELEASE / COUNT
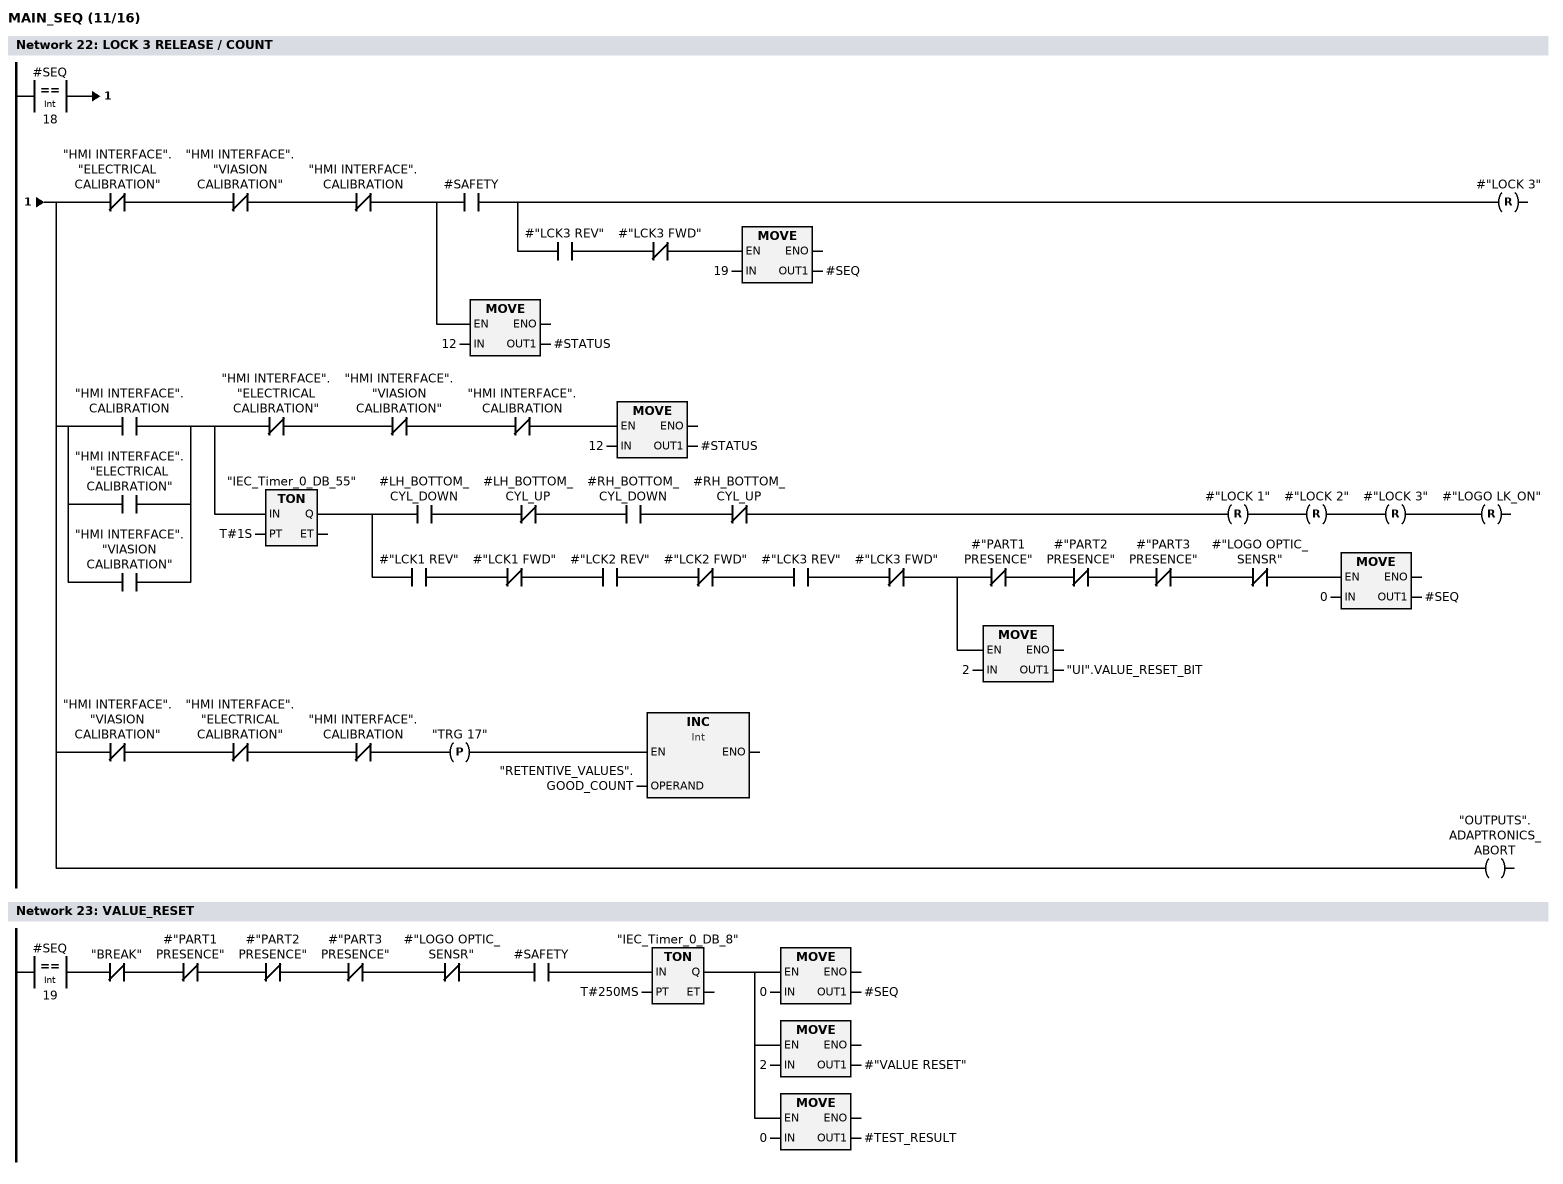
   #_w1 := #SEQ = 18;
   #_w2 := #_w1 AND NOT "HMI INTERFACE"."ELECTRICAL CALIBRATION" AND NOT "HMI INTERFACE"."VIASION CALIBRATION" AND NOT "HMI INTERFACE".CALIBRATION;
   #_w3 := #_w2 AND #SAFETY;
   IF #_w3 THEN #"LOCK 3" := FALSE; END_IF;
   IF #_w3 AND #"LCK3 REV" AND NOT #"LCK3 FWD" THEN #SEQ := 19; END_IF;
   IF #_w2 THEN #STATUS := 12; END_IF;
   #_w4 := #_w1 AND ("HMI INTERFACE".CALIBRATION OR "HMI INTERFACE"."ELECTRICAL CALIBRATION" OR "HMI INTERFACE"."VIASION CALIBRATION");
   IF #_w4 AND NOT "HMI INTERFACE"."ELECTRICAL CALIBRATION" AND NOT "HMI INTERFACE"."VIASION CALIBRATION" AND NOT "HMI INTERFACE".CALIBRATION THEN
       #STATUS := 12;
   END_IF;
   "IEC_Timer_0_DB_55".TON(IN := #_w4, PT := T#1S);
   IF "IEC_Timer_0_DB_55".Q AND #LH_BOTTOM_CYL_DOWN AND NOT #LH_BOTTOM_CYL_UP AND #RH_BOTTOM_CYL_DOWN AND NOT #RH_BOTTOM_CYL_UP THEN
       #"LOCK 1" := FALSE;
       #"LOCK 2" := FALSE;
       #"LOCK 3" := FALSE;
       #"LOGO LK_ON" := FALSE;
   END_IF;
   #_w5 := "IEC_Timer_0_DB_55".Q AND #"LCK1 REV" AND NOT #"LCK1 FWD" AND #"LCK2 REV" AND NOT #"LCK2 FWD" AND #"LCK3 REV" AND NOT #"LCK3 FWD";
   IF #_w5 AND NOT #"PART1 PRESENCE" AND NOT #"PART2 PRESENCE" AND NOT #"PART3 PRESENCE" AND NOT #"LOGO OPTIC_SENSR" THEN
       #SEQ := 0;
   END_IF;
   IF #_w5 THEN "UI".VALUE_RESET_BIT := 2; END_IF;
   #_w6 := #_w1 AND NOT "HMI INTERFACE"."VIASION CALIBRATION" AND NOT "HMI INTERFACE"."ELECTRICAL CALIBRATION" AND NOT "HMI INTERFACE".CALIBRATION;
   #_w7 := #_w6 AND NOT "TRG 17";   // rising edge
   "TRG 17" := #_w6;
   IF #_w7 THEN "RETENTIVE_VALUES".GOOD_COUNT := "RETENTIVE_VALUES".GOOD_COUNT + 1; END_IF;
   "OUTPUTS".ADAPTRONICS_ABORT := #_w1;
END_REGION

REGION Network 23: VALUE_RESET
   "IEC_Timer_0_DB_8".TON(IN := (#SEQ = 19) AND NOT "BREAK" AND NOT #"PART1 PRESENCE" AND NOT #"PART2 PRESENCE" AND NOT #"PART3 PRESENCE" AND NOT #"LOGO OPTIC_SENSR" AND #SAFETY,
                          PT := T#250MS);
   IF "IEC_Timer_0_DB_8".Q THEN
       #SEQ := 0;
       #"VALUE RESET" := 2;
       #TEST_RESULT := 0;
   END_IF;
END_REGION

REGION Network 24: REJECTION
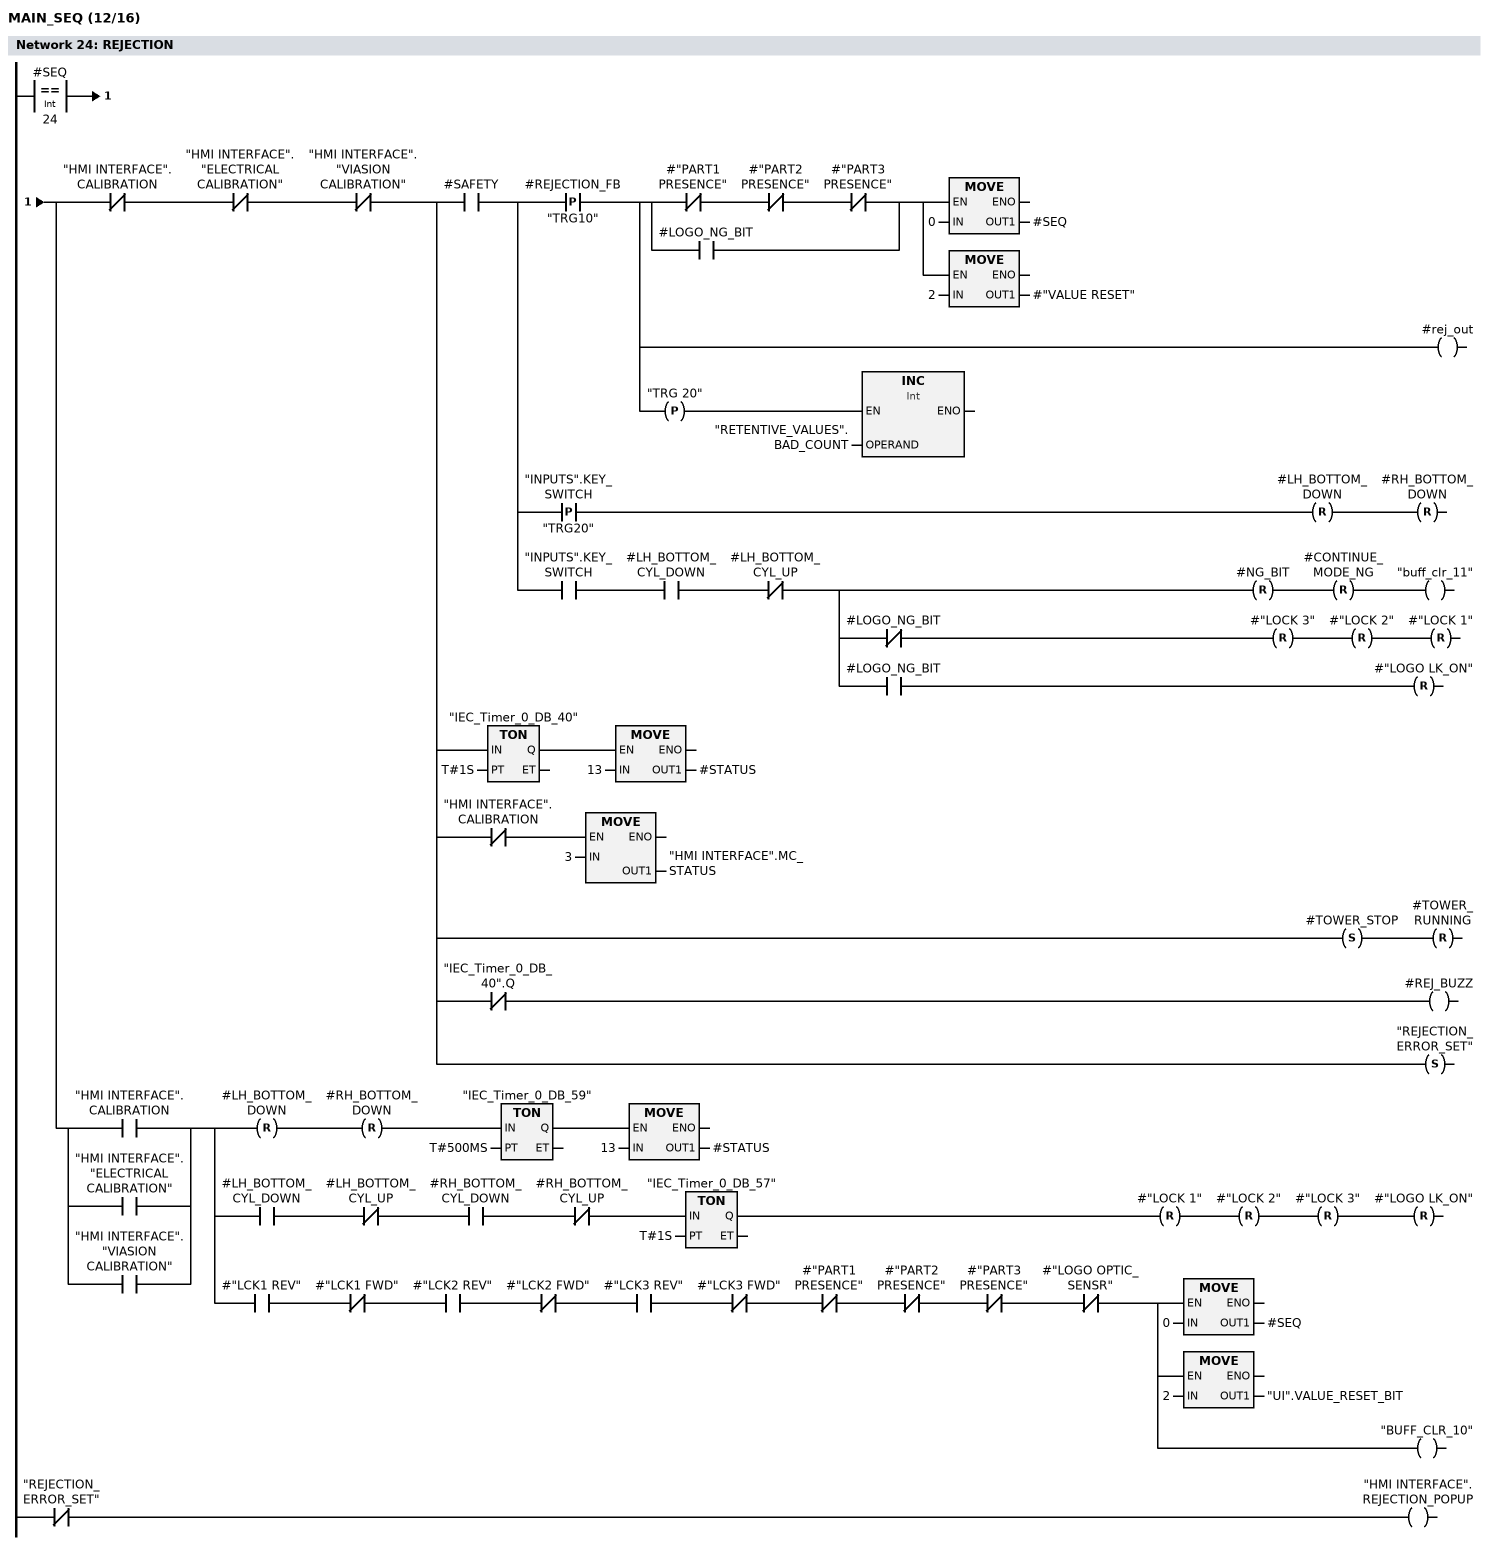
   #_w1 := #SEQ = 24;
   #_w2 := #_w1 AND NOT "HMI INTERFACE".CALIBRATION AND NOT "HMI INTERFACE"."ELECTRICAL CALIBRATION" AND NOT "HMI INTERFACE"."VIASION CALIBRATION";
   #_w3 := #_w2 AND #SAFETY;
   #_w4 := #_w3 AND #REJECTION_FB AND NOT "TRG10";   // rising edge of #REJECTION_FB
   "TRG10" := #REJECTION_FB;
   IF #_w4 AND ((NOT #"PART1 PRESENCE" AND NOT #"PART2 PRESENCE" AND NOT #"PART3 PRESENCE") OR #LOGO_NG_BIT) THEN
       #SEQ := 0;
       #"VALUE RESET" := 2;
   END_IF;
   #rej_out := #_w4;
   #_w5 := #_w4 AND NOT "TRG 20";   // rising edge
   "TRG 20" := #_w4;
   IF #_w5 THEN "RETENTIVE_VALUES".BAD_COUNT := "RETENTIVE_VALUES".BAD_COUNT + 1; END_IF;
   #_w6 := #_w3 AND "INPUTS".KEY_SWITCH AND NOT "TRG20";   // rising edge of "INPUTS".KEY_SWITCH
   "TRG20" := "INPUTS".KEY_SWITCH;
   IF #_w6 THEN
       #LH_BOTTOM_DOWN := FALSE;
       #RH_BOTTOM_DOWN := FALSE;
   END_IF;
   #_w7 := #_w3 AND "INPUTS".KEY_SWITCH AND #LH_BOTTOM_CYL_DOWN AND NOT #LH_BOTTOM_CYL_UP;
   IF #_w7 THEN
       #NG_BIT := FALSE;
       #CONTINUE_MODE_NG := FALSE;
   END_IF;
   "buff_clr_11" := #_w7;
   IF #_w7 AND NOT #LOGO_NG_BIT THEN
       #"LOCK 3" := FALSE;
       #"LOCK 2" := FALSE;
       #"LOCK 1" := FALSE;
   END_IF;
   IF #_w7 AND #LOGO_NG_BIT THEN #"LOGO LK_ON" := FALSE; END_IF;
   "IEC_Timer_0_DB_40".TON(IN := #_w2, PT := T#1S);
   IF "IEC_Timer_0_DB_40".Q THEN #STATUS := 13; END_IF;
   IF #_w2 AND NOT "HMI INTERFACE".CALIBRATION THEN "HMI INTERFACE".MC_STATUS := 3; END_IF;
   IF #_w2 THEN
       #TOWER_STOP := TRUE;
       #TOWER_RUNNING := FALSE;
   END_IF;
   #REJ_BUZZ := #_w2 AND NOT "IEC_Timer_0_DB_40".Q;
   IF #_w2 THEN "REJECTION_ERROR_SET" := TRUE; END_IF;
   #_w8 := #_w1 AND ("HMI INTERFACE".CALIBRATION OR "HMI INTERFACE"."ELECTRICAL CALIBRATION" OR "HMI INTERFACE"."VIASION CALIBRATION");
   IF #_w8 THEN
       #LH_BOTTOM_DOWN := FALSE;
       #RH_BOTTOM_DOWN := FALSE;
   END_IF;
   "IEC_Timer_0_DB_59".TON(IN := #_w8, PT := T#500MS);
   IF "IEC_Timer_0_DB_59".Q THEN #STATUS := 13; END_IF;
   "IEC_Timer_0_DB_57".TON(IN := #_w8 AND #LH_BOTTOM_CYL_DOWN AND NOT #LH_BOTTOM_CYL_UP AND #RH_BOTTOM_CYL_DOWN AND NOT #RH_BOTTOM_CYL_UP,
                           PT := T#1S);
   IF "IEC_Timer_0_DB_57".Q THEN
       #"LOCK 1" := FALSE;
       #"LOCK 2" := FALSE;
       #"LOCK 3" := FALSE;
       #"LOGO LK_ON" := FALSE;
   END_IF;
   #_w9 := #_w8 AND #"LCK1 REV" AND NOT #"LCK1 FWD" AND #"LCK2 REV" AND NOT #"LCK2 FWD" AND #"LCK3 REV" AND NOT #"LCK3 FWD" AND NOT #"PART1 PRESENCE" AND NOT #"PART2 PRESENCE" AND NOT #"PART3 PRESENCE" AND NOT #"LOGO OPTIC_SENSR";
   IF #_w9 THEN
       #SEQ := 0;
       "UI".VALUE_RESET_BIT := 2;
   END_IF;
   "BUFF_CLR_10" := #_w9;
   "HMI INTERFACE".REJECTION_POPUP := NOT "REJECTION_ERROR_SET";
END_REGION

REGION Network 25: ELECTRICAL_PARTLOADED_BIT
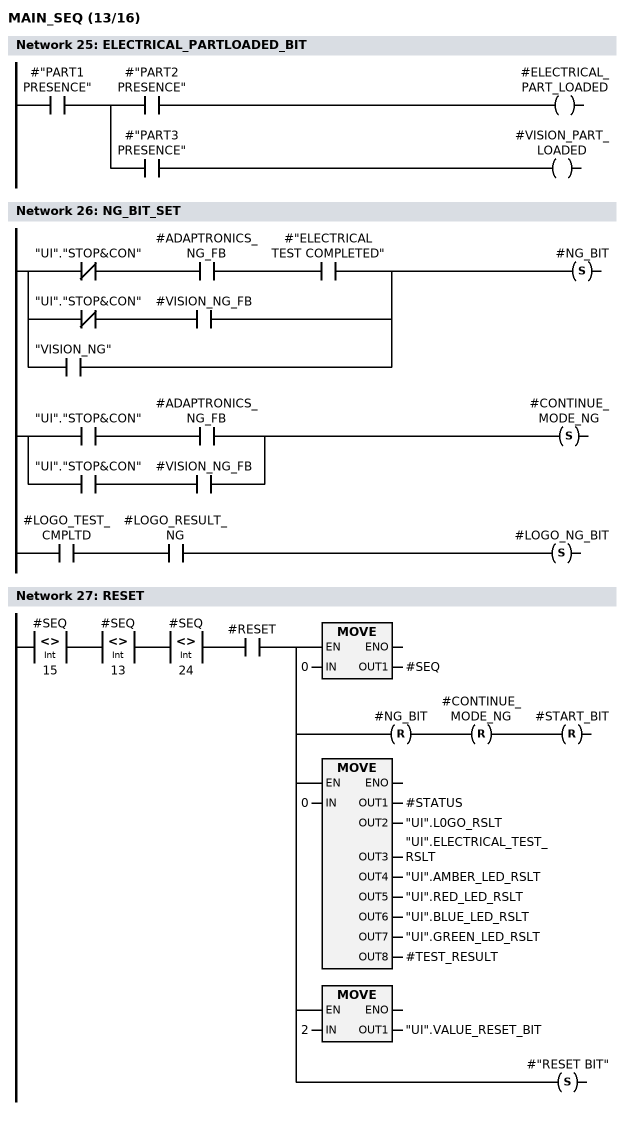
   RUNG wire#powerrail
      Contact( #"PART1 PRESENCE" )
      wire#w1
      Contact( #"PART2 PRESENCE" )
      Coil( #ELECTRICAL_PART_LOADED )
   END_RUNG
   RUNG wire#w1
      Contact( #"PART3 PRESENCE" )
      Coil( #VISION_PART_LOADED )
   END_RUNG
   // the same network as SCL:
   #ELECTRICAL_PART_LOADED := #"PART1 PRESENCE" AND #"PART2 PRESENCE";
   #VISION_PART_LOADED := #"PART1 PRESENCE" AND #"PART3 PRESENCE";
END_REGION

REGION Network 26: NG_BIT_SET
   RUNG wire#powerrail
      I_Contact( "UI"."STOP&CON" )
      Contact( #ADAPTRONICS_NG_FB )
      Contact( #"ELECTRICAL TEST COMPLETED" )
      wire#w1
      S_Coil( #NG_BIT )
   END_RUNG
   RUNG wire#powerrail
      I_Contact( "UI"."STOP&CON" )
      Contact( #VISION_NG_FB )
   END_RUNG wire#w1
   RUNG wire#powerrail
      Contact( "VISION_NG" )
   END_RUNG wire#w1
   RUNG wire#powerrail
      Contact( "UI"."STOP&CON" )
      Contact( #ADAPTRONICS_NG_FB )
      wire#w2
      S_Coil( #CONTINUE_MODE_NG )
   END_RUNG
   RUNG wire#powerrail
      Contact( "UI"."STOP&CON" )
      Contact( #VISION_NG_FB )
   END_RUNG wire#w2
   RUNG wire#powerrail
      Contact( #LOGO_TEST_CMPLTD )
      Contact( #LOGO_RESULT_NG )
      S_Coil( #LOGO_NG_BIT )
   END_RUNG
   // the same network as SCL:
   IF (NOT "UI"."STOP&CON" AND #ADAPTRONICS_NG_FB AND #"ELECTRICAL TEST COMPLETED") OR (NOT "UI"."STOP&CON" AND #VISION_NG_FB) OR "VISION_NG" THEN
       #NG_BIT := TRUE;
   END_IF;
   IF ("UI"."STOP&CON" AND #ADAPTRONICS_NG_FB) OR ("UI"."STOP&CON" AND #VISION_NG_FB) THEN
       #CONTINUE_MODE_NG := TRUE;
   END_IF;
   IF #LOGO_TEST_CMPLTD AND #LOGO_RESULT_NG THEN #LOGO_NG_BIT := TRUE; END_IF;
END_REGION

REGION Network 27: RESET
   RUNG wire#powerrail
      { S7_Templates := "SrcType := Int" } NE_Contact(in1 := #SEQ, in2 := 15)
      { S7_Templates := "SrcType := Int" } NE_Contact(in1 := #SEQ, in2 := 13)
      { S7_Templates := "SrcType := Int" } NE_Contact(in1 := #SEQ, in2 := 24)
      Contact( #RESET )
      wire#w1
      Move(in := 0, out1 => #SEQ)
   END_RUNG
   RUNG wire#w1
      R_Coil( #NG_BIT )
      R_Coil( #CONTINUE_MODE_NG )
      R_Coil( #START_BIT )
   END_RUNG
   RUNG wire#w1
      Move(in := 0, out1 => #STATUS, out2 => "UI".L0GO_RSLT, out3 => "UI".ELECTRICAL_TEST_RSLT, out4 => "UI".AMBER_LED_RSLT, out5 => "UI".RED_LED_RSLT, out6 => "UI".BLUE_LED_RSLT, out7 => "UI".GREEN_LED_RSLT, out8 => #TEST_RESULT)
   END_RUNG
   RUNG wire#w1
      Move(in := 2, out1 => "UI".VALUE_RESET_BIT)
   END_RUNG
   RUNG wire#w1
      S_Coil( #"RESET BIT" )
   END_RUNG
   // the same network as SCL:
   #_w1 := (#SEQ <> 15) AND (#SEQ <> 13) AND (#SEQ <> 24) AND #RESET;
   IF #_w1 THEN
       #SEQ := 0;
       #NG_BIT := FALSE;
       #CONTINUE_MODE_NG := FALSE;
       #START_BIT := FALSE;
       #STATUS := 0;
       "UI".L0GO_RSLT := 0;
       "UI".ELECTRICAL_TEST_RSLT := 0;
       "UI".AMBER_LED_RSLT := 0;
       "UI".RED_LED_RSLT := 0;
       "UI".BLUE_LED_RSLT := 0;
       "UI".GREEN_LED_RSLT := 0;
       #TEST_RESULT := 0;
       "UI".VALUE_RESET_BIT := 2;
       #"RESET BIT" := TRUE;
   END_IF;
END_REGION

REGION Network 28: RESET
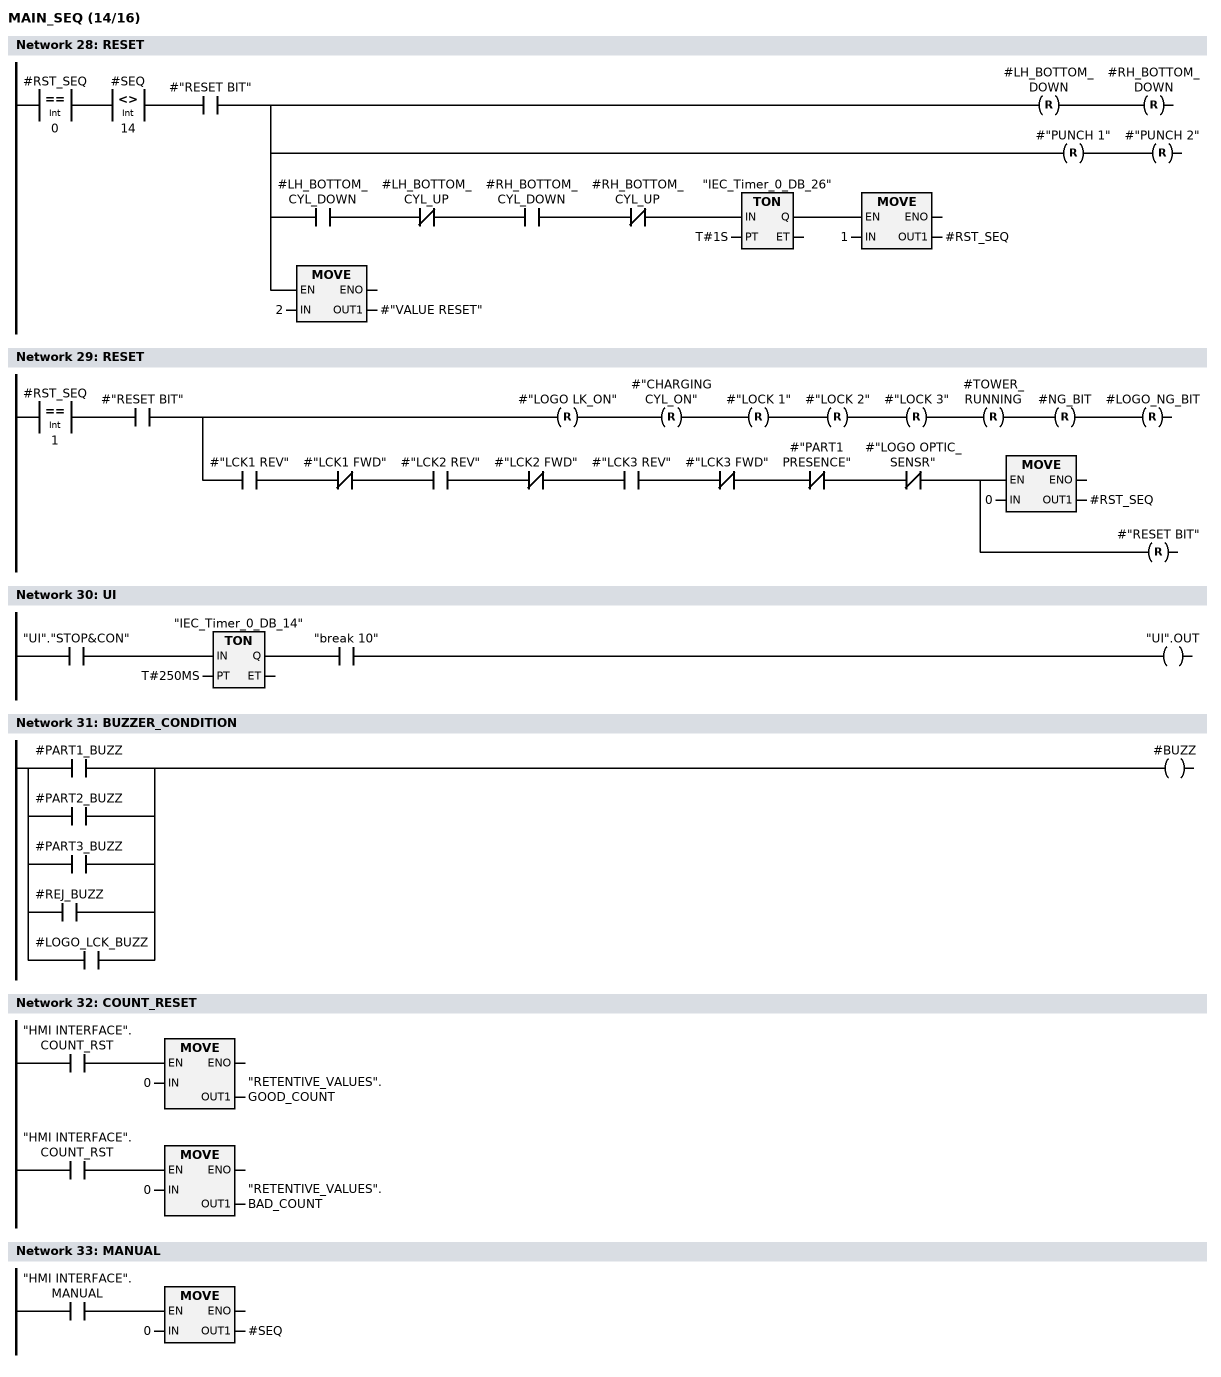
   #_w1 := (#RST_SEQ = 0) AND (#SEQ <> 14) AND #"RESET BIT";
   IF #_w1 THEN
       #LH_BOTTOM_DOWN := FALSE;
       #RH_BOTTOM_DOWN := FALSE;
       #"PUNCH 1" := FALSE;
       #"PUNCH 2" := FALSE;
   END_IF;
   "IEC_Timer_0_DB_26".TON(IN := #_w1 AND #LH_BOTTOM_CYL_DOWN AND NOT #LH_BOTTOM_CYL_UP AND #RH_BOTTOM_CYL_DOWN AND NOT #RH_BOTTOM_CYL_UP,
                           PT := T#1S);
   IF "IEC_Timer_0_DB_26".Q THEN #RST_SEQ := 1; END_IF;
   IF #_w1 THEN #"VALUE RESET" := 2; END_IF;
END_REGION

REGION Network 29: RESET
   RUNG wire#powerrail
      { S7_Templates := "SrcType := Int" } EQ_Contact(in1 := #RST_SEQ, in2 := 1)
      Contact( #"RESET BIT" )
      wire#w1
      R_Coil( #"LOGO LK_ON" )
      R_Coil( #"CHARGING CYL_ON" )
      R_Coil( #"LOCK 1" )
      R_Coil( #"LOCK 2" )
      R_Coil( #"LOCK 3" )
      R_Coil( #TOWER_RUNNING )
      R_Coil( #NG_BIT )
      R_Coil( #LOGO_NG_BIT )
   END_RUNG
   RUNG wire#w1
      Contact( #"LCK1 REV" )
      I_Contact( #"LCK1 FWD" )
      Contact( #"LCK2 REV" )
      I_Contact( #"LCK2 FWD" )
      Contact( #"LCK3 REV" )
      I_Contact( #"LCK3 FWD" )
      I_Contact( #"PART1 PRESENCE" )
      I_Contact( #"LOGO OPTIC_SENSR" )
      wire#w2
      Move(in := 0, out1 => #RST_SEQ)
   END_RUNG
   RUNG wire#w2
      R_Coil( #"RESET BIT" )
   END_RUNG
   // the same network as SCL:
   #_w1 := (#RST_SEQ = 1) AND #"RESET BIT";
   IF #_w1 THEN
       #"LOGO LK_ON" := FALSE;
       #"CHARGING CYL_ON" := FALSE;
       #"LOCK 1" := FALSE;
       #"LOCK 2" := FALSE;
       #"LOCK 3" := FALSE;
       #TOWER_RUNNING := FALSE;
       #NG_BIT := FALSE;
       #LOGO_NG_BIT := FALSE;
   END_IF;
   IF #_w1 AND #"LCK1 REV" AND NOT #"LCK1 FWD" AND #"LCK2 REV" AND NOT #"LCK2 FWD" AND #"LCK3 REV" AND NOT #"LCK3 FWD" AND NOT #"PART1 PRESENCE" AND NOT #"LOGO OPTIC_SENSR" THEN
       #RST_SEQ := 0;
       #"RESET BIT" := FALSE;
   END_IF;
END_REGION

REGION Network 30: UI
   "IEC_Timer_0_DB_14".TON(IN := "UI"."STOP&CON", PT := T#250MS);
   "UI".OUT := "IEC_Timer_0_DB_14".Q AND "break 10";
END_REGION

REGION Network 31: BUZZER_CONDITION
   RUNG wire#powerrail
      Contact( #PART1_BUZZ )
      wire#w1
      Coil( #BUZZ )
   END_RUNG
   RUNG wire#powerrail
      Contact( #PART2_BUZZ )
   END_RUNG wire#w1
   RUNG wire#powerrail
      Contact( #PART3_BUZZ )
   END_RUNG wire#w1
   RUNG wire#powerrail
      Contact( #REJ_BUZZ )
   END_RUNG wire#w1
   RUNG wire#powerrail
      Contact( #LOGO_LCK_BUZZ )
   END_RUNG wire#w1
   // the same network as SCL:
   #BUZZ := #PART1_BUZZ OR #PART2_BUZZ OR #PART3_BUZZ OR #REJ_BUZZ OR #LOGO_LCK_BUZZ;
END_REGION

REGION Network 32: COUNT_RESET
   RUNG wire#powerrail
      Contact( "HMI INTERFACE".COUNT_RST )
      Move(in := 0, out1 => "RETENTIVE_VALUES".GOOD_COUNT)
   END_RUNG
   RUNG wire#powerrail
      Contact( "HMI INTERFACE".COUNT_RST )
      Move(in := 0, out1 => "RETENTIVE_VALUES".BAD_COUNT)
   END_RUNG
   // the same network as SCL:
   IF "HMI INTERFACE".COUNT_RST THEN
       "RETENTIVE_VALUES".GOOD_COUNT := 0;
       "RETENTIVE_VALUES".BAD_COUNT := 0;
   END_IF;
END_REGION

REGION Network 33: MANUAL
   RUNG wire#powerrail
      Contact( "HMI INTERFACE".MANUAL )
      Move(in := 0, out1 => #SEQ)
   END_RUNG
   // the same network as SCL:
   IF "HMI INTERFACE".MANUAL THEN #SEQ := 0; END_IF;
END_REGION

REGION Network 34: SAFETY_ERROR
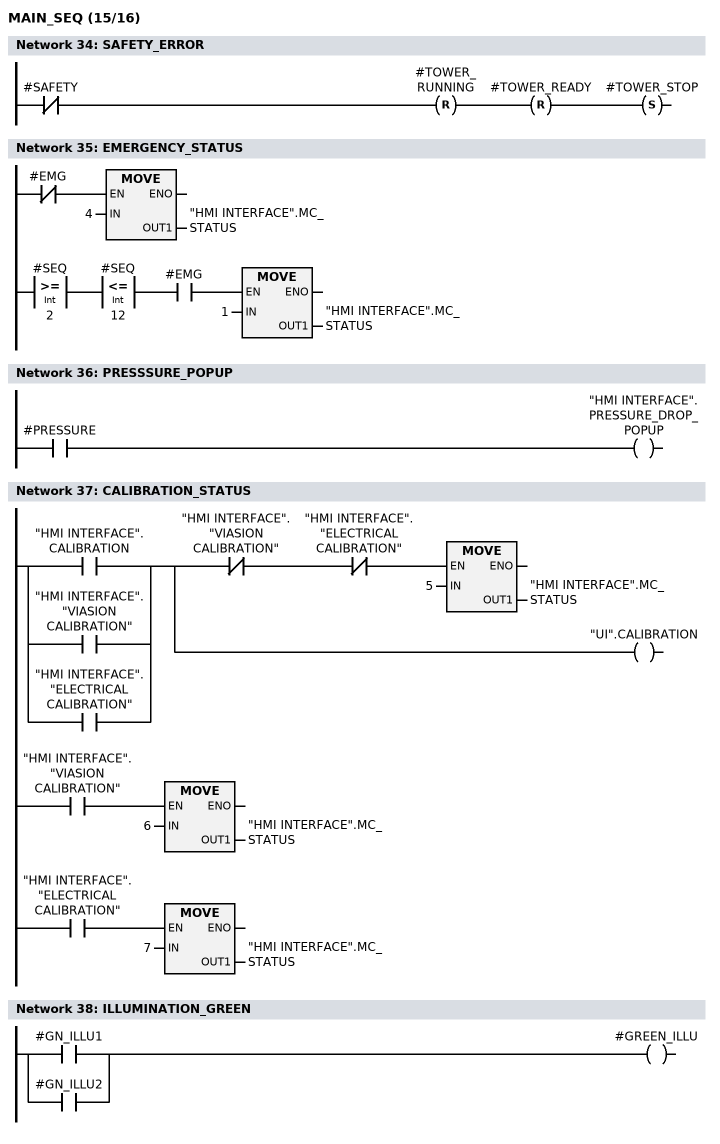
   RUNG wire#powerrail
      I_Contact( #SAFETY )
      R_Coil( #TOWER_RUNNING )
      R_Coil( #TOWER_READY )
      S_Coil( #TOWER_STOP )
   END_RUNG
   // the same network as SCL:
   IF NOT #SAFETY THEN
       #TOWER_RUNNING := FALSE;
       #TOWER_READY := FALSE;
       #TOWER_STOP := TRUE;
   END_IF;
END_REGION

REGION Network 35: EMERGENCY_STATUS
   RUNG wire#powerrail
      I_Contact( #EMG )
      Move(in := 4, out1 => "HMI INTERFACE".MC_STATUS)
   END_RUNG
   RUNG wire#powerrail
      { S7_Templates := "SrcType := Int" } GE_Contact(in1 := #SEQ, in2 := 2)
      { S7_Templates := "SrcType := Int" } LE_Contact(in1 := #SEQ, in2 := 12)
      Contact( #EMG )
      Move(in := 1, out1 => "HMI INTERFACE".MC_STATUS)
   END_RUNG
   // the same network as SCL:
   IF NOT #EMG THEN "HMI INTERFACE".MC_STATUS := 4; END_IF;
   IF (#SEQ >= 2) AND (#SEQ <= 12) AND #EMG THEN "HMI INTERFACE".MC_STATUS := 1; END_IF;
END_REGION

REGION Network 36: PRESSSURE_POPUP
   RUNG wire#powerrail
      Contact( #PRESSURE )
      Coil( "HMI INTERFACE".PRESSURE_DROP_POPUP )
   END_RUNG
   // the same network as SCL:
   "HMI INTERFACE".PRESSURE_DROP_POPUP := #PRESSURE;
END_REGION

REGION Network 37: CALIBRATION_STATUS
   RUNG wire#powerrail
      Contact( "HMI INTERFACE".CALIBRATION )
      wire#w1
      I_Contact( "HMI INTERFACE"."VIASION CALIBRATION" )
      I_Contact( "HMI INTERFACE"."ELECTRICAL CALIBRATION" )
      Move(in := 5, out1 => "HMI INTERFACE".MC_STATUS)
   END_RUNG
   RUNG wire#powerrail
      Contact( "HMI INTERFACE"."VIASION CALIBRATION" )
   END_RUNG wire#w1
   RUNG wire#powerrail
      Contact( "HMI INTERFACE"."ELECTRICAL CALIBRATION" )
   END_RUNG wire#w1
   RUNG wire#w1
      Coil( "UI".CALIBRATION )
   END_RUNG
   RUNG wire#powerrail
      Contact( "HMI INTERFACE"."VIASION CALIBRATION" )
      Move(in := 6, out1 => "HMI INTERFACE".MC_STATUS)
   END_RUNG
   RUNG wire#powerrail
      Contact( "HMI INTERFACE"."ELECTRICAL CALIBRATION" )
      Move(in := 7, out1 => "HMI INTERFACE".MC_STATUS)
   END_RUNG
   // the same network as SCL:
   #_w1 := "HMI INTERFACE".CALIBRATION OR "HMI INTERFACE"."VIASION CALIBRATION" OR "HMI INTERFACE"."ELECTRICAL CALIBRATION";
   IF #_w1 AND NOT "HMI INTERFACE"."VIASION CALIBRATION" AND NOT "HMI INTERFACE"."ELECTRICAL CALIBRATION" THEN
       "HMI INTERFACE".MC_STATUS := 5;
   END_IF;
   "UI".CALIBRATION := #_w1;
   IF "HMI INTERFACE"."VIASION CALIBRATION" THEN "HMI INTERFACE".MC_STATUS := 6; END_IF;
   IF "HMI INTERFACE"."ELECTRICAL CALIBRATION" THEN "HMI INTERFACE".MC_STATUS := 7; END_IF;
END_REGION

REGION Network 38: ILLUMINATION_GREEN
   RUNG wire#powerrail
      Contact( #GN_ILLU1 )
      wire#w1
      Coil( #GREEN_ILLU )
   END_RUNG
   RUNG wire#powerrail
      Contact( #GN_ILLU2 )
   END_RUNG wire#w1
   // the same network as SCL:
   #GREEN_ILLU := #GN_ILLU1 OR #GN_ILLU2;
END_REGION

REGION Network 39: UI VALUE INITIALIZING AFTER CALIBRATION
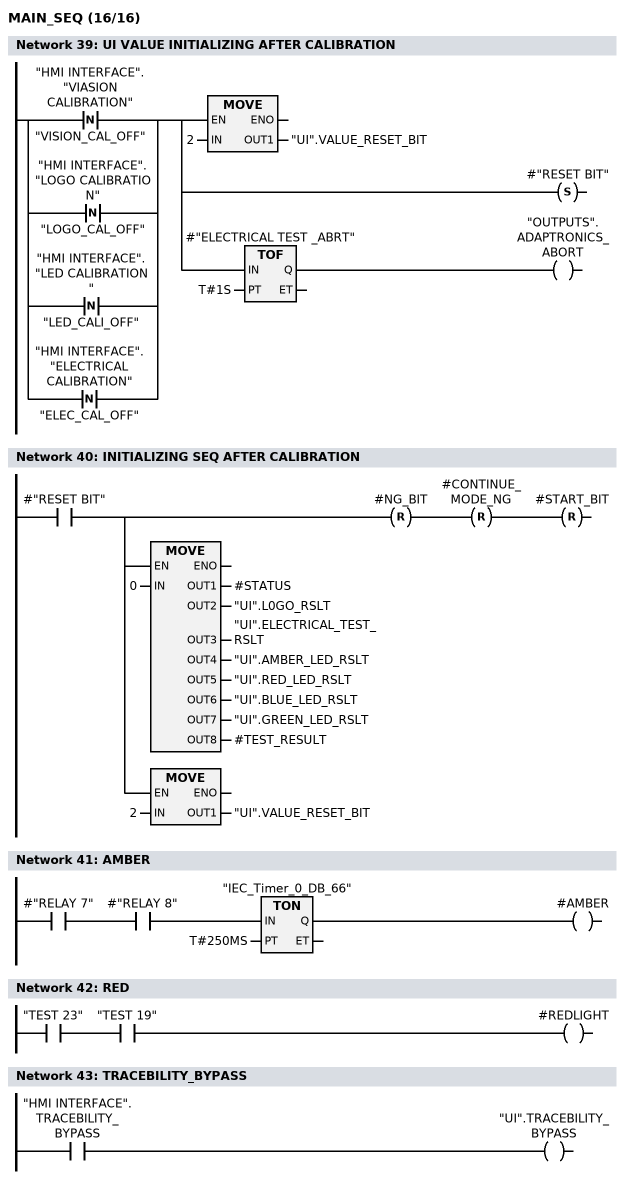
   #_w1 := NOT "HMI INTERFACE"."VIASION CALIBRATION" AND "VISION_CAL_OFF";   // falling edge of "HMI INTERFACE"."VIASION CALIBRATION"
   "VISION_CAL_OFF" := "HMI INTERFACE"."VIASION CALIBRATION";
   #_w2 := NOT "HMI INTERFACE"."LOGO CALIBRATION" AND "LOGO_CAL_OFF";   // falling edge of "HMI INTERFACE"."LOGO CALIBRATION"
   "LOGO_CAL_OFF" := "HMI INTERFACE"."LOGO CALIBRATION";
   #_w3 := NOT "HMI INTERFACE"."LED CALIBRATION" AND "LED_CALI_OFF";   // falling edge of "HMI INTERFACE"."LED CALIBRATION"
   "LED_CALI_OFF" := "HMI INTERFACE"."LED CALIBRATION";
   #_w4 := NOT "HMI INTERFACE"."ELECTRICAL CALIBRATION" AND "ELEC_CAL_OFF";   // falling edge of "HMI INTERFACE"."ELECTRICAL CALIBRATION"
   "ELEC_CAL_OFF" := "HMI INTERFACE"."ELECTRICAL CALIBRATION";
   #_w5 := #_w1 OR #_w2 OR #_w3 OR #_w4;
   IF #_w5 THEN
       "UI".VALUE_RESET_BIT := 2;
       #"RESET BIT" := TRUE;
   END_IF;
   #"ELECTRICAL TEST _ABRT"(IN := #_w5, PT := T#1S);   // TOF
   "OUTPUTS".ADAPTRONICS_ABORT := #"ELECTRICAL TEST _ABRT".Q;
END_REGION

REGION Network 40: INITIALIZING SEQ AFTER CALIBRATION
   RUNG wire#powerrail
      Contact( #"RESET BIT" )
      wire#w1
      R_Coil( #NG_BIT )
      R_Coil( #CONTINUE_MODE_NG )
      R_Coil( #START_BIT )
   END_RUNG
   RUNG wire#w1
      Move(in := 0, out1 => #STATUS, out2 => "UI".L0GO_RSLT, out3 => "UI".ELECTRICAL_TEST_RSLT, out4 => "UI".AMBER_LED_RSLT, out5 => "UI".RED_LED_RSLT, out6 => "UI".BLUE_LED_RSLT, out7 => "UI".GREEN_LED_RSLT, out8 => #TEST_RESULT)
   END_RUNG
   RUNG wire#w1
      Move(in := 2, out1 => "UI".VALUE_RESET_BIT)
   END_RUNG
   // the same network as SCL:
   IF #"RESET BIT" THEN
       #NG_BIT := FALSE;
       #CONTINUE_MODE_NG := FALSE;
       #START_BIT := FALSE;
       #STATUS := 0;
       "UI".L0GO_RSLT := 0;
       "UI".ELECTRICAL_TEST_RSLT := 0;
       "UI".AMBER_LED_RSLT := 0;
       "UI".RED_LED_RSLT := 0;
       "UI".BLUE_LED_RSLT := 0;
       "UI".GREEN_LED_RSLT := 0;
       #TEST_RESULT := 0;
       "UI".VALUE_RESET_BIT := 2;
   END_IF;
END_REGION

REGION Network 41: AMBER
   "IEC_Timer_0_DB_66".TON(IN := #"RELAY 7" AND #"RELAY 8", PT := T#250MS);
   #AMBER := "IEC_Timer_0_DB_66".Q;
END_REGION

REGION Network 42: RED
   RUNG wire#powerrail
      Contact( "TEST 23" )
      Contact( "TEST 19" )
      Coil( #REDLIGHT )
   END_RUNG
   // the same network as SCL:
   #REDLIGHT := "TEST 23" AND "TEST 19";
END_REGION

REGION Network 43: TRACEBILITY_BYPASS
   RUNG wire#powerrail
      Contact( "HMI INTERFACE".TRACEBILITY_BYPASS )
      Coil( "UI".TRACEBILITY_BYPASS )
   END_RUNG
   // the same network as SCL:
   "UI".TRACEBILITY_BYPASS := "HMI INTERFACE".TRACEBILITY_BYPASS;
END_REGION
END_FUNCTION_BLOCK

FUNCTION "INPUT_MAPPING" : Void   // FC1, LAD
{ S7_Optimized_Access := 'TRUE' }
VERSION : 0.1
   VAR_TEMP
      INC_2 : DInt;
   END_VAR
BEGIN

REGION Network 1: EMERGENCY
